Omron CX-Programmer project 新工程 (CX-Programmer 9.61)

# PLC XWD负压氦检: CJ2M CPU34
I/O table (CPU CJ2M-CPU34): rack 0 slot 11 CJ2M-EIP21

## Global symbols (name address type ; comment)
0.00 BOOL  ; #1扫码阻挡气缸缩回位
0.01 BOOL  ; #1扫码阻挡气缸伸出位
0.02 BOOL  ; #1隔离气缸缩回位
0.03 BOOL  ; 隔离气缸到位
0.04 BOOL  ; #2扫码阻挡气缸缩回位
0.05 BOOL  ; #2扫码阻挡气缸伸出位
0.06 BOOL  ; #2隔离气缸缩回位
0.08 BOOL  ; #1进料夹爪夹紧位
0.09 BOOL  ; #1进料夹爪松开位
0.10 BOOL  ; #2进料夹爪夹紧位
0.11 BOOL  ; #2进料夹爪松开位
0.12 BOOL  ; 进料夹爪变距气缸伸出位
0.13 BOOL  ; 进料夹爪变距气缸缩回位
0.14 BOOL  ; #1出料夹爪夹紧位
0.15 BOOL  ; #1出料夹爪松开位
10.00 BOOL  ; #1扫码阻挡气缸缩回
10.01 BOOL  ; #1扫码阻挡气缸伸出
10.02 BOOL  ; #1隔离气缸缩回
10.03 BOOL  ; #1隔离气缸伸出
10.04 BOOL  ; #2扫码阻挡气缸缩回
10.05 BOOL  ; #2扫码阻挡气缸伸出
10.06 BOOL  ; #2隔离气缸缩回
10.07 BOOL  ; #2隔离气缸伸出
10.08 BOOL  ; #1进料夹爪夹紧
10.09 BOOL  ; #1进料夹爪松开
10.10 BOOL  ; #2进料夹爪夹紧
10.11 BOOL  ; #2进料夹爪松开
10.12 BOOL  ; 进料夹爪变距气缸伸出
10.13 BOOL  ; 进料夹爪变距气缸缩回
10.14 BOOL  ; #1出料夹爪夹紧
10.15 BOOL  ; #1出料夹爪松开
11.00 BOOL  ; #2出料夹爪夹紧
11.01 BOOL  ; #2出料夹爪松开
11.02 BOOL  ; 出料夹爪变距气缸伸出
11.03 BOOL  ; 出料夹爪变距气缸缩回
11.04 BOOL  ; #1腔体平移一级气缸缩回
11.05 BOOL  ; #1腔体平移一级气缸伸出
11.06 BOOL  ; #1腔体平移二级气缸缩回
11.07 BOOL  ; #1腔体平移二级气缸伸出
11.08 BOOL  ; #1腔体顶伸气缸上升
11.09 BOOL  ; #1腔体顶伸气缸下降
11.10 BOOL  ; #1腔体氦检阀开
11.11 BOOL  ; 氦检仪真空阀开
11.12 BOOL  ; #1腔体抽真空阀开
11.13 BOOL  ; #1-1腔体阀开
11.14 BOOL  ; #1-2腔体阀开
11.15 BOOL  ; #1腔体破真空阀开
12.00 BOOL  ; #1腔体吹气阀开
12.01 BOOL  ; #2腔体平移一级气缸缩回
12.02 BOOL  ; #2腔体平移一级气缸伸出
12.03 BOOL  ; #2腔体平移二级气缸缩回
12.04 BOOL  ; #2腔体平移二级气缸伸出
12.05 BOOL  ; #2腔体顶伸气缸上升
12.06 BOOL  ; #2腔体顶伸气缸下降
12.07 BOOL  ; #2腔体氦检阀开
12.08 BOOL  ; 复检清洁阀开
12.09 BOOL  ; #2腔体抽真空阀开
12.10 BOOL  ; #2-1腔体阀开
12.11 BOOL  ; #2-2腔体阀开
12.12 BOOL  ; #2腔体破真空阀开
12.13 BOOL  ; #2腔体吹气阀开
12.14 BOOL  ; #3腔体平移一级气缸缩回
12.15 BOOL  ; #3腔体平移一级气缸伸出
13.00 BOOL  ; #3腔体平移二级气缸缩回
13.01 BOOL  ; #3腔体平移二级气缸伸出
13.02 BOOL  ; #3腔体顶伸气缸上升
13.03 BOOL  ; #3腔体顶伸气缸下降
13.04 BOOL  ; #3腔体氦检阀开
13.05 BOOL  ; 标漏阀开
13.06 BOOL  ; #3腔体抽真空阀开
13.07 BOOL  ; #3-1腔体阀开
13.08 BOOL  ; #3-2腔体阀开
13.09 BOOL  ; #3腔体破真空阀开
13.10 BOOL  ; #3腔体吹气阀开
13.11 BOOL  ; 进料伺服X轴使能
13.12 BOOL  ; 进料伺服X轴故障复位
13.13 BOOL  ; 进料伺服Z轴使能
13.14 BOOL  ; 进料伺服Z轴故障复位
13.15 BOOL  ; 进料伺服Z轴刹车
14.00 BOOL  ; 出料伺服X轴使能
14.01 BOOL  ; 出料伺服X轴故障复位
14.02 BOOL  ; 出料伺服Z轴使能
14.03 BOOL  ; 出料伺服Z轴故障复位
14.04 BOOL  ; 出料伺服Z轴刹车
14.05 BOOL  ; 腔体抽真空泵启动
14.07 BOOL  ; 氦检前置泵启动
14.08 BOOL  ; 氦检仪供电
14.09 BOOL  ; 启动按钮指示灯
14.10 BOOL  ; 停止按钮指示灯
14.11 BOOL  ; 复位按钮指示灯
14.12 BOOL  ; 蜂鸣器
14.13 BOOL  ; 三色灯（红）
14.14 BOOL  ; 三色灯（绿）
14.15 BOOL  ; 三色灯（黄）
1559.15 BOOL  ; SCU21_2Port#1 Protocol Macro Executing Flag
1569.15 BOOL  ; SCU21_2Port#2 Protocol Macro Executing Flag
15.00 BOOL  ; 进料拉带电机启动
15.01 BOOL  ; 扫码NG拉带电机启动
15.02 BOOL  ; 氦检NG拉带电机启动
15.03 BOOL  ; 进料对接输出
15.04 BOOL  ; 出料对接输出（TO下工站放料请求）
15.05 BOOL  ; 出料旋转气缸90度输出
15.06 BOOL  ; 出料旋转气缸0度输出
15.07 BOOL  ; 进料前段拉带输出
16.00 BOOL  ; #1-1电池抽真空阀开
16.01 BOOL  ; #1-2电池抽真空阀开
16.02 BOOL  ; #1-1电池注氦阀开
16.03 BOOL  ; #1-2电池注氦阀开
16.04 BOOL  ; #1-1电池破真空阀开
16.05 BOOL  ; #1-2电池破真空阀开
16.06 BOOL  ; #2-1电池抽真空阀开
16.07 BOOL  ; #2-2电池抽真空阀开
16.08 BOOL  ; #2-1电池注氦阀开
16.09 BOOL  ; #2-2电池注氦阀开
16.10 BOOL  ; #2-1电池破真空阀开
16.11 BOOL  ; #2-2电池破真空阀开
16.12 BOOL  ; #3-1电池抽真空阀开
16.13 BOOL  ; #3-2电池抽真空阀开
16.14 BOOL  ; #3-1电池注氦阀开
16.15 BOOL  ; #3-2电池注氦阀开
17.00 BOOL  ; #3-1电池破真空阀开
17.01 BOOL  ; #3-2电池破真空阀开
1.00 BOOL  ; #2出料夹爪夹紧位
1.01 BOOL  ; #2出料夹爪松开位
1.02 BOOL  ; 出料夹爪变距气缸伸出位
1.03 BOOL  ; 出料夹爪变距气缸缩回位
1.04 BOOL  ; #1腔体平移一级气缸缩回位
1.05 BOOL  ; #1腔体平移一级气缸伸出位
1.06 BOOL  ; #1腔体平移二级气缸缩回位
1.07 BOOL  ; #1腔体平移二级气缸伸出位
1.08 BOOL  ; #1腔体顶伸气缸上升位
1.09 BOOL  ; #1腔体顶伸气缸下降位
1.10 BOOL  ; #1腔体氦检阀开到位
1.11 BOOL  ; #1腔体氦检阀关到位
2001 CHANNEL  ; #1-1电池真空模拟量读数(AD081_1)
2002 CHANNEL  ; #1-2电池真空模拟量读数(AD081_2)
2003 CHANNEL  ; #2-1电池真空模拟量读数(AD081_3)
2004 CHANNEL  ; #2-2电池真空模拟量读数(AD081_4)
2005 CHANNEL  ; #3-1电池真空模拟量读数(AD081_5)
2006 CHANNEL  ; #3-2电池真空模拟量读数(AD081_6)
200.00 BOOL  ; PLC上电
200.01 BOOL  ; 紧急停止
200.01 BOOL  ; 急停按钮标志[0004.12]
200.02 BOOL  ; 自动启动
200.03 BOOL  ; 自动停止
200.04 BOOL  ; 报警清除
200.05 BOOL  ; 清料停止中
200.06 BOOL  ; 异常报警停止
200.08 BOOL  ; 设备待料状态（参考进料）
200.09 BOOL  ; 设备内有电池
200.10 BOOL  ; 机台有错误
200.11 BOOL  ; 报警中
200.12 BOOL  ; 三色灯-绿灯
200.13 BOOL  ; 三色灯-红灯
200.14 BOOL  ; 三色灯-黄灯
200.15 BOOL  ; 三色灯-蜂鸣器
2011 CHANNEL  ; #1腔体真空模拟量读数(AD041_1)
2012 CHANNEL  ; #2腔体真空模拟量读数(AD041_2)
2013 CHANNEL  ; #3腔体真空模拟量读数(AD041_3)
201.00 BOOL  ; 整机在初始位
205.00 BOOL  ; 整机停止中（Lamp）
205.01 BOOL  ; 清料停止中（Lamp）
205.02 BOOL  ; 整机复位（Lamp）
210.01 BOOL  ; PC系统通讯正常标志
210.02 BOOL  ; 整机机械手归零标志
210.03 BOOL  ; 安全门标志
210.04 BOOL  ; 氦检仪启动标志
221.00 BOOL  ; 整机复位（M）
221.01 BOOL  ; 进料拉带工站整机复位（M）
221.02 BOOL  ; 进料伺服工站整机复位（M）
221.03 BOOL  ; #1氦检工站整机复位（M）
221.04 BOOL  ; #2氦检工站整机复位（M）
221.05 BOOL  ; #3氦检工站整机复位（M）
221.06 BOOL  ; 出料伺服工站整机复位（M）
2960.02 BOOL  ; 进料伺服Z轴原点感应标志
2960.06 BOOL  ; 进料伺服X轴正极限
2960.07 BOOL  ; 进料伺服X轴负极限
2960.08 BOOL  ; 进料伺服Z轴正极限
2960.09 BOOL  ; 进料伺服Z轴负极限
2962.02 BOOL  ; 出料伺服Z轴原点感应标志
2962.06 BOOL  ; 出料伺服X轴正极限
2962.07 BOOL  ; 出料伺服X轴负极限
2962.08 BOOL  ; 出料伺服Z轴正极限
2962.09 BOOL  ; 出料伺服Z轴负极限
2.01 BOOL  ; #2腔体平移一级气缸缩回位
2.02 BOOL  ; #2腔体平移一级气缸伸出位
2.03 BOOL  ; #2腔体平移二级气缸缩回位
2.04 BOOL  ; #2腔体平移二级气缸伸出位
2.05 BOOL  ; #2腔体顶伸气缸上升位
2.06 BOOL  ; #2腔体顶伸气缸下降位
2.07 BOOL  ; #2腔体氦检阀开到位
2.08 BOOL  ; #2腔体氦检阀关到位
2.14 BOOL  ; #3腔体平移一级气缸缩回位
2.15 BOOL  ; #3腔体平移一级气缸伸出位
300.00 BOOL  ; #1扫码阻挡气缸缩回[Pls]
300.01 BOOL  ; #1扫码阻挡气缸伸出[Pls]
300.02 BOOL  ; #1隔离气缸缩回[Pls]
300.03 BOOL  ; #1隔离气缸伸出[Pls]
300.04 BOOL  ; #2扫码阻挡气缸缩回[Pls]
300.05 BOOL  ; #2扫码阻挡气缸伸出[Pls]
300.06 BOOL  ; #2隔离气缸缩回[Pls]
300.07 BOOL  ; #2隔离气缸伸出[Pls]
300.08 BOOL  ; #1进料夹爪夹紧[Pls]
300.09 BOOL  ; #1进料夹爪松开[Pls]
300.10 BOOL  ; #2进料夹爪夹紧[Pls]
300.11 BOOL  ; #2进料夹爪松开[Pls]
300.12 BOOL  ; 进料夹爪变距气缸伸出[Pls]
300.13 BOOL  ; 进料夹爪变距气缸缩回[Pls]
300.14 BOOL  ; #1出料夹爪夹紧[Pls]
300.15 BOOL  ; #1出料夹爪松开[Pls]
301.00 BOOL  ; #2出料夹爪夹紧[Pls]
301.01 BOOL  ; #2出料夹爪松开[Pls]
301.02 BOOL  ; 出料夹爪变距气缸伸出[Pls]
301.03 BOOL  ; 出料夹爪变距气缸缩回[Pls]
301.04 BOOL  ; #1腔体平移一级气缸缩回[Pls]
301.05 BOOL  ; #1腔体平移一级气缸伸出[Pls]
301.06 BOOL  ; #1腔体平移二级气缸缩回[Pls]
301.07 BOOL  ; #1腔体平移二级气缸伸出[Pls]
301.08 BOOL  ; #1腔体顶伸气缸上升[Pls]
301.09 BOOL  ; #1腔体顶伸气缸下降[Pls]
301.10 BOOL  ; #1腔体氦检阀开[Pls]
301.11 BOOL  ; 氦检仪真空阀开[Pls]
301.12 BOOL  ; #1腔体抽真空阀开[Pls]
301.13 BOOL  ; #1-1腔体阀开[Pls]
301.14 BOOL  ; #1-2腔体阀开[Pls]
301.15 BOOL  ; #1腔体破真空阀开[Pls]
302.00 BOOL  ; #1腔体吹气阀开[Pls]
302.01 BOOL  ; #2腔体平移一级气缸缩回[Pls]
302.02 BOOL  ; #2腔体平移一级气缸伸出[Pls]
302.03 BOOL  ; #2腔体平移二级气缸缩回[Pls]
302.04 BOOL  ; #2腔体平移二级气缸伸出[Pls]
302.05 BOOL  ; #2腔体顶伸气缸上升[Pls]
302.06 BOOL  ; #2腔体顶伸气缸下降[Pls]
302.07 BOOL  ; #2腔体氦检阀开[Pls]
302.08 BOOL  ; 复检清洁阀开[Pls]
302.09 BOOL  ; #2腔体抽真空阀开[Pls]
302.10 BOOL  ; #2-1腔体阀开[Pls]
302.11 BOOL  ; #2-2腔体阀开[Pls]
302.12 BOOL  ; #2腔体破真空阀开[Pls]
302.13 BOOL  ; #2腔体吹气阀开[Pls]
302.14 BOOL  ; #3腔体平移一级气缸缩回[Pls]
302.15 BOOL  ; #3腔体平移一级气缸伸出[Pls]
303.00 BOOL  ; #3腔体平移二级气缸缩回[Pls]
303.01 BOOL  ; #3腔体平移二级气缸伸出[Pls]
303.02 BOOL  ; #3腔体顶伸气缸上升[Pls]
303.03 BOOL  ; #3腔体顶伸气缸下降[Pls]
303.04 BOOL  ; #3腔体氦检阀开[Pls]
303.05 BOOL  ; 0[Pls]
303.06 BOOL  ; #3腔体抽真空阀开[Pls]
303.07 BOOL  ; #3-1腔体阀开[Pls]
303.08 BOOL  ; #3-2腔体阀开[Pls]
303.09 BOOL  ; #3腔体破真空阀开[Pls]
303.10 BOOL  ; #3腔体吹气阀开[Pls]
303.11 BOOL  ; 进料伺服X轴使能[Pls]
303.12 BOOL  ; 进料伺服X轴故障复位[Pls]
303.13 BOOL  ; 进料伺服Z轴使能[Pls]
303.14 BOOL  ; 进料伺服Z轴故障复位[Pls]
303.15 BOOL  ; 进料伺服Z轴刹车[Pls]
304.00 BOOL  ; 出料伺服X轴使能[Pls]
304.01 BOOL  ; 出料伺服X轴故障复位[Pls]
304.02 BOOL  ; 出料伺服Z轴使能[Pls]
304.03 BOOL  ; 出料伺服Z轴故障复位[Pls]
304.04 BOOL  ; 出料伺服Z轴刹车[Pls]
304.05 BOOL  ; 腔体抽真空泵启动[Pls]
304.06 BOOL  ; 0[Pls]
304.07 BOOL  ; 氦检前置泵启动[Pls]
304.08 BOOL  ; 氦检仪供电[Pls]
304.09 BOOL  ; 启动按钮指示灯[Pls]
304.10 BOOL  ; 停止按钮指示灯[Pls]
304.11 BOOL  ; 复位按钮指示灯[Pls]
304.12 BOOL  ; 蜂鸣器[Pls]
304.13 BOOL  ; 三色灯（红）[Pls]
304.14 BOOL  ; 三色灯（绿）[Pls]
304.15 BOOL  ; 三色灯（黄）[Pls]
305.00 BOOL  ; 进料拉带电机启动[Pls]
305.01 BOOL  ; 扫码NG拉带电机启动[Pls]
305.02 BOOL  ; 氦检NG拉带电机启动[Pls]
305.03 BOOL  ; 进料对接输出[Pls]
305.04 BOOL  ; 出料对接输出[Pls]
305.05 BOOL  ; 出料旋转气缸9O度位条件
305.06 BOOL  ; 出料旋转气缸O度位条件
305.07 BOOL  ; 0[Pls]
305.08 BOOL  ; 0[Pls]
305.09 BOOL  ; 0[Pls]
305.10 BOOL  ; 0[Pls]
305.11 BOOL  ; 0[Pls]
305.12 BOOL  ; 0[Pls]
305.13 BOOL  ; 0[Pls]
305.14 BOOL  ; 0[Pls]
305.15 BOOL  ; 0[Pls]
306.00 BOOL  ; #1-1电池抽真空阀开[Pls]
306.01 BOOL  ; #1-2电池抽真空阀开[Pls]
306.02 BOOL  ; #1-1电池注氦阀开[Pls]
306.03 BOOL  ; #1-2电池注氦阀开[Pls]
306.04 BOOL  ; #1-1电池破真空阀开[Pls]
306.05 BOOL  ; #1-2电池破真空阀开[Pls]
306.06 BOOL  ; #2-1电池抽真空阀开[Pls]
306.07 BOOL  ; #2-2电池抽真空阀开[Pls]
306.08 BOOL  ; #2-1电池注氦阀开[Pls]
306.09 BOOL  ; #2-2电池注氦阀开[Pls]
306.10 BOOL  ; #2-1电池破真空阀开[Pls]
306.11 BOOL  ; #2-2电池破真空阀开[Pls]
306.12 BOOL  ; #3-1电池抽真空阀开[Pls]
306.13 BOOL  ; #3-2电池抽真空阀开[Pls]
306.14 BOOL  ; #3-1电池注氦阀开[Pls]
306.15 BOOL  ; #3-2电池注氦阀开[Pls]
307.00 BOOL  ; #3-1电池破真空阀开[Pls]
307.01 BOOL  ; #3-2电池破真空阀开[Pls]
307.02 BOOL  ; 0[Pls]
307.03 BOOL  ; 0[Pls]
307.04 BOOL  ; 0[Pls]
307.05 BOOL  ; 0[Pls]
307.06 BOOL  ; 0[Pls]
307.07 BOOL  ; 0[Pls]
307.08 BOOL  ; 0[Pls]
307.09 BOOL  ; 0[Pls]
307.10 BOOL  ; 0[Pls]
307.11 BOOL  ; 0[Pls]
307.12 BOOL  ; 0[Pls]
307.13 BOOL  ; 0[Pls]
307.14 BOOL  ; 0[Pls]
307.15 BOOL  ; 0[Pls]
311.10 BOOL  ; #1腔体氦检阀关[Pls]
311.11 BOOL  ; 氦检仪真空阀关[Pls]
311.12 BOOL  ; #1腔体抽真空阀关[Pls]
311.13 BOOL  ; #1-1腔体阀关[Pls]
311.14 BOOL  ; #1-2腔体阀关[Pls]
311.15 BOOL  ; #1腔体破真空阀关[Pls]
312.00 BOOL  ; #1腔体吹气阀关[Pls]
312.01 BOOL  ; [Pls]
312.02 BOOL  ; [Pls]
312.03 BOOL  ; [Pls]
312.04 BOOL  ; [Pls]
312.05 BOOL  ; [Pls]
312.06 BOOL  ; [Pls]
312.07 BOOL  ; #2腔体氦检阀关[Pls]
312.08 BOOL  ; 复检清洁阀关[Pls]
312.09 BOOL  ; #2腔体抽真空阀关[Pls]
312.10 BOOL  ; #2-1腔体阀关[Pls]
312.11 BOOL  ; #2-2腔体阀关[Pls]
312.12 BOOL  ; #2腔体破真空阀关[Pls]
312.13 BOOL  ; #2腔体吹气阀关[Pls]
312.14 BOOL  ; 0[Pls]
312.15 BOOL  ; [Pls]
313.00 BOOL  ; [Pls]
313.01 BOOL  ; [Pls]
313.02 BOOL  ; [Pls]
313.03 BOOL  ; [Pls]
313.04 BOOL  ; #3腔体氦检阀关[Pls]
313.05 BOOL  ; 0[Pls]
313.06 BOOL  ; #3腔体抽真空阀关[Pls]
313.07 BOOL  ; #3-1腔体阀关[Pls]
313.08 BOOL  ; #3-2腔体阀关[Pls]
313.09 BOOL  ; #3腔体破真空阀关[Pls]
313.10 BOOL  ; #3腔体吹气阀关[Pls]
313.11 BOOL  ; [Pls]
313.12 BOOL  ; [Pls]
313.13 BOOL  ; [Pls]
313.14 BOOL  ; [Pls]
313.15 BOOL  ; [Pls]
314.00 BOOL  ; [Pls]
314.01 BOOL  ; [Pls]
314.02 BOOL  ; [Pls]
314.03 BOOL  ; [Pls]
314.04 BOOL  ; [Pls]
314.05 BOOL  ; 腔体抽真空泵停止[Pls]
314.06 BOOL  ; 0[Pls]
314.07 BOOL  ; 氦检前置泵停止[Pls]
314.08 BOOL  ; 氦检仪停电[Pls]
314.09 BOOL  ; [Pls]
314.10 BOOL  ; [Pls]
314.11 BOOL  ; [Pls]
314.12 BOOL  ; [Pls]
314.13 BOOL  ; [Pls]
314.14 BOOL  ; [Pls]
314.15 BOOL  ; [Pls]
315.00 BOOL  ; 进料拉带电机停止[Pls]
315.01 BOOL  ; 扫码NG拉带电机停止[Pls]
315.02 BOOL  ; 氦检NG拉带电机停止[Pls]
315.03 BOOL  ; 0[Pls]
315.04 BOOL  ; [Pls]
315.05 BOOL  ; [Pls]
315.06 BOOL  ; [Pls]
315.07 BOOL  ; [Pls]
315.08 BOOL  ; [Pls]
315.09 BOOL  ; [Pls]
315.10 BOOL  ; [Pls]
315.11 BOOL  ; [Pls]
315.12 BOOL  ; [Pls]
315.13 BOOL  ; [Pls]
315.14 BOOL  ; [Pls]
315.15 BOOL  ; [Pls]
316.00 BOOL  ; #1-1电池抽真空阀关[Pls]
316.01 BOOL  ; #1-2电池抽真空阀关[Pls]
316.02 BOOL  ; #1-1电池注氦阀关[Pls]
316.03 BOOL  ; #1-2电池注氦阀关[Pls]
316.04 BOOL  ; #1-1电池破真空阀关[Pls]
316.05 BOOL  ; #1-2电池破真空阀关[Pls]
316.06 BOOL  ; #2-1电池抽真空阀关[Pls]
316.07 BOOL  ; #2-2电池抽真空阀关[Pls]
316.08 BOOL  ; #2-1电池注氦阀关[Pls]
316.09 BOOL  ; #2-2电池注氦阀关[Pls]
316.10 BOOL  ; #2-1电池破真空阀关[Pls]
316.11 BOOL  ; #2-2电池破真空阀关[Pls]
316.12 BOOL  ; #3-1电池抽真空阀关[Pls]
316.13 BOOL  ; #3-2电池抽真空阀关[Pls]
316.14 BOOL  ; #3-1电池注氦阀关[Pls]
316.15 BOOL  ; #3-2电池注氦阀关[Pls]
317.00 BOOL  ; #3-1电池破真空阀关[Pls]
317.01 BOOL  ; #3-2电池破真空阀关[Pls]
3.00 BOOL  ; #3腔体平移二级气缸缩回位
3.01 BOOL  ; #3腔体平移二级气缸伸出位
3.02 BOOL  ; #3腔体顶伸气缸上升位
3.03 BOOL  ; #3腔体顶伸气缸下降位
3.04 BOOL  ; #3腔体氦检阀开到位
3.05 BOOL  ; #3腔体氦检阀关到位
3.06 BOOL  ; 氦检仪准备好了信号
3.07 BOOL  ; 氦检仪故障信号
3.11 BOOL  ; 进料伺服X轴准备好了信号
3.12 BOOL  ; 进料伺服X轴故障信号
3.13 BOOL  ; 进料伺服Z轴准备好了信号
3.14 BOOL  ; 进料伺服Z轴故障信号
400.00 BOOL  ; #1扫码阻挡气缸缩回[M]
400.01 BOOL  ; #1扫码阻挡气缸伸出[M]
400.02 BOOL  ; #1隔离气缸缩回[M]
400.03 BOOL  ; #1隔离气缸伸出[M]
400.04 BOOL  ; #2扫码阻挡气缸缩回[M]
400.05 BOOL  ; #2扫码阻挡气缸伸出[M]
400.06 BOOL  ; #2隔离气缸缩回[M]
400.07 BOOL  ; #2隔离气缸伸出[M]
400.08 BOOL  ; #1进料夹爪夹紧[M]
400.09 BOOL  ; #1进料夹爪松开[M]
400.10 BOOL  ; #2进料夹爪夹紧[M]
400.11 BOOL  ; #2进料夹爪松开[M]
400.12 BOOL  ; 进料夹爪变距气缸伸出[M]
400.13 BOOL  ; 进料夹爪变距气缸缩回[M]
400.14 BOOL  ; #1出料夹爪夹紧[M]
400.15 BOOL  ; #1出料夹爪松开[M]
401.00 BOOL  ; #2出料夹爪夹紧[M]
401.01 BOOL  ; #2出料夹爪松开[M]
401.02 BOOL  ; 出料夹爪变距气缸伸出[M]
401.03 BOOL  ; 出料夹爪变距气缸缩回[M]
401.04 BOOL  ; #1腔体平移一级气缸缩回[M]
401.05 BOOL  ; #1腔体平移一级气缸伸出[M]
401.06 BOOL  ; #1腔体平移二级气缸缩回[M]
401.07 BOOL  ; #1腔体平移二级气缸伸出[M]
401.08 BOOL  ; #1腔体顶伸气缸上升[M]
401.09 BOOL  ; #1腔体顶伸气缸下降[M]
401.10 BOOL  ; #1腔体氦检阀开[M]
401.11 BOOL  ; 氦检仪真空阀开[M]
401.12 BOOL  ; #1腔体抽真空阀开[M]
401.13 BOOL  ; #1-1腔体阀开[M]
401.14 BOOL  ; #1-2腔体阀开[M]
401.15 BOOL  ; #1腔体破真空阀开[M]
402.00 BOOL  ; #1腔体吹气阀开[M]
402.01 BOOL  ; #2腔体平移一级气缸缩回[M]
402.02 BOOL  ; #2腔体平移一级气缸伸出[M]
402.03 BOOL  ; #2腔体平移二级气缸缩回[M]
402.04 BOOL  ; #2腔体平移二级气缸伸出[M]
402.05 BOOL  ; #2腔体顶伸气缸上升[M]
402.06 BOOL  ; #2腔体顶伸气缸下降[M]
402.07 BOOL  ; #2腔体氦检阀开[M]
402.08 BOOL  ; 复检清洁阀开[M]
402.09 BOOL  ; #2腔体抽真空阀开[M]
402.10 BOOL  ; #2-1腔体阀开[M]
402.11 BOOL  ; #2-2腔体阀开[M]
402.12 BOOL  ; #2腔体破真空阀开[M]
402.13 BOOL  ; #2腔体吹气阀开[M]
402.14 BOOL  ; #3腔体平移一级气缸缩回[M]
402.15 BOOL  ; #3腔体平移一级气缸伸出[M]
403.00 BOOL  ; #3腔体平移二级气缸缩回[M]
403.01 BOOL  ; #3腔体平移二级气缸伸出[M]
403.02 BOOL  ; #3腔体顶伸气缸上升[M]
403.03 BOOL  ; #3腔体顶伸气缸下降[M]
403.04 BOOL  ; #3腔体氦检阀开[M]
403.05 BOOL  ; 0[M]
403.06 BOOL  ; #3腔体抽真空阀开[M]
403.07 BOOL  ; #3-1腔体阀开[M]
403.08 BOOL  ; #3-2腔体阀开[M]
403.09 BOOL  ; #3腔体破真空阀开[M]
403.10 BOOL  ; #3腔体吹气阀开[M]
403.11 BOOL  ; 进料伺服X轴使能[M]
403.12 BOOL  ; 进料伺服X轴故障复位[M]
403.13 BOOL  ; 进料伺服Z轴使能[M]
403.14 BOOL  ; 进料伺服Z轴故障复位[M]
403.15 BOOL  ; 进料伺服Z轴刹车[M]
404.00 BOOL  ; 出料伺服X轴使能[M]
404.01 BOOL  ; 出料伺服X轴故障复位[M]
404.02 BOOL  ; 出料伺服Z轴使能[M]
404.03 BOOL  ; 出料伺服Z轴故障复位[M]
404.04 BOOL  ; 出料伺服Z轴刹车[M]
404.05 BOOL  ; 腔体抽真空泵启动[M]
404.06 BOOL  ; 0[M]
404.07 BOOL  ; 氦检前置泵启动[M]
404.08 BOOL  ; 氦检仪供电[M]
404.09 BOOL  ; 启动按钮指示灯[M]
404.10 BOOL  ; 停止按钮指示灯[M]
404.11 BOOL  ; 复位按钮指示灯[M]
404.12 BOOL  ; 蜂鸣器[M]
404.13 BOOL  ; 三色灯（红）[M]
404.14 BOOL  ; 三色灯（绿）[M]
404.15 BOOL  ; 三色灯（黄）[M]
405.00 BOOL  ; 进料拉带电机启动[M]
405.01 BOOL  ; 扫码NG拉带电机启动[M]
405.02 BOOL  ; 氦检NG拉带电机启动[M]
405.03 BOOL  ; 进料对接输出[M]
405.04 BOOL  ; 出料对接输出[M]
405.05 BOOL  ; 出料旋转气缸90度输出[M]
405.06 BOOL  ; 出料旋转气缸0度输出[M]
405.07 BOOL  ; 0[M]
405.08 BOOL  ; 0[M]
405.09 BOOL  ; 0[M]
405.10 BOOL  ; 0[M]
405.11 BOOL  ; 0[M]
405.12 BOOL  ; 0[M]
405.13 BOOL  ; 0[M]
405.14 BOOL  ; 0[M]
405.15 BOOL  ; 0[M]
406.00 BOOL  ; #1-1电池抽真空阀开[M]
406.01 BOOL  ; #1-2电池抽真空阀开[M]
406.02 BOOL  ; #1-1电池注氦阀开[M]
406.03 BOOL  ; #1-2电池注氦阀开[M]
406.04 BOOL  ; #1-1电池破真空阀开[M]
406.05 BOOL  ; #1-2电池破真空阀开[M]
406.06 BOOL  ; #2-1电池抽真空阀开[M]
406.07 BOOL  ; #2-2电池抽真空阀开[M]
406.08 BOOL  ; #2-1电池注氦阀开[M]
406.09 BOOL  ; #2-2电池注氦阀开[M]
406.10 BOOL  ; #2-1电池破真空阀开[M]
406.11 BOOL  ; #2-2电池破真空阀开[M]
406.12 BOOL  ; #3-1电池抽真空阀开[M]
406.13 BOOL  ; #3-2电池抽真空阀开[M]
406.14 BOOL  ; #3-1电池注氦阀开[M]
406.15 BOOL  ; #3-2电池注氦阀开[M]
407.00 BOOL  ; #3-1电池破真空阀开[M]
407.01 BOOL  ; #3-2电池破真空阀开[M]
407.02 BOOL  ; 0[M]
407.03 BOOL  ; 0[M]
407.04 BOOL  ; 0[M]
407.05 BOOL  ; 0[M]
407.06 BOOL  ; 0[M]
407.07 BOOL  ; 0[M]
407.08 BOOL  ; 0[M]
407.09 BOOL  ; 0[M]
407.10 BOOL  ; 0[M]
407.11 BOOL  ; 0[M]
407.12 BOOL  ; 0[M]
407.13 BOOL  ; 0[M]
407.14 BOOL  ; 0[M]
407.15 BOOL  ; 0[M]
411.10 BOOL  ; #1腔体氦检阀关[M]
411.11 BOOL  ; 氦检仪真空阀关[M]
411.12 BOOL  ; #1腔体抽真空阀关[M]
411.13 BOOL  ; #1-1腔体阀关[M]
411.14 BOOL  ; #1-2腔体阀关[M]
411.15 BOOL  ; #1腔体破真空阀关[M]
412.00 BOOL  ; #1腔体吹气阀关[M]
412.01 BOOL  ; [M]
412.02 BOOL  ; [M]
412.03 BOOL  ; [M]
412.04 BOOL  ; [M]
412.05 BOOL  ; [M]
412.06 BOOL  ; [M]
412.07 BOOL  ; #2腔体氦检阀关[M]
412.08 BOOL  ; 复检清洁阀关[M]
412.09 BOOL  ; #2腔体抽真空阀关[M]
412.10 BOOL  ; #2-1腔体阀关[M]
412.11 BOOL  ; #2-2腔体阀关[M]
412.12 BOOL  ; #2腔体破真空阀关[M]
412.13 BOOL  ; #2腔体吹气阀关[M]
412.14 BOOL  ; 0[M]
412.15 BOOL  ; [M]
413.00 BOOL  ; [M]
413.01 BOOL  ; [M]
413.02 BOOL  ; [M]
413.03 BOOL  ; [M]
413.04 BOOL  ; #3腔体氦检阀关[M]
413.05 BOOL  ; 0[M]
413.06 BOOL  ; #3腔体抽真空阀关[M]
413.07 BOOL  ; #3-1腔体阀关[M]
413.08 BOOL  ; #3-2腔体阀关[M]
413.09 BOOL  ; #3腔体破真空阀关[M]
413.10 BOOL  ; #3腔体吹气阀关[M]
413.11 BOOL  ; [M]
413.12 BOOL  ; [M]
413.13 BOOL  ; [M]
413.14 BOOL  ; [M]
413.15 BOOL  ; [M]
414.00 BOOL  ; [M]
414.01 BOOL  ; [M]
414.02 BOOL  ; [M]
414.03 BOOL  ; [M]
414.04 BOOL  ; [M]
414.05 BOOL  ; 腔体抽真空泵停止[M]
414.06 BOOL  ; 0[M]
414.07 BOOL  ; 氦检前置泵停止[M]
414.08 BOOL  ; 氦检仪停电[M]
414.09 BOOL  ; [M]
414.10 BOOL  ; [M]
414.11 BOOL  ; [M]
414.12 BOOL  ; [M]
414.13 BOOL  ; [M]
414.14 BOOL  ; [M]
414.15 BOOL  ; [M]
415.00 BOOL  ; 进料拉带电机停止[M]
415.01 BOOL  ; 扫码NG拉带电机停止[M]
415.02 BOOL  ; 氦检NG拉带电机停止[M]
415.03 BOOL  ; 0[M]
415.04 BOOL  ; [M]
415.05 BOOL  ; [M]
415.06 BOOL  ; [M]
415.07 BOOL  ; [M]
415.08 BOOL  ; [M]
415.09 BOOL  ; [M]
415.10 BOOL  ; [M]
415.11 BOOL  ; [M]
415.12 BOOL  ; [M]
415.13 BOOL  ; [M]
415.14 BOOL  ; [M]
415.15 BOOL  ; [M]
416.00 BOOL  ; #1-1电池抽真空阀关[M]
416.01 BOOL  ; #1-2电池抽真空阀关[M]
416.02 BOOL  ; #1-1电池注氦阀关[M]
416.03 BOOL  ; #1-2电池注氦阀关[M]
416.04 BOOL  ; #1-1电池破真空阀关[M]
416.05 BOOL  ; #1-2电池破真空阀关[M]
416.06 BOOL  ; #2-1电池抽真空阀关[M]
416.07 BOOL  ; #2-2电池抽真空阀关[M]
416.08 BOOL  ; #2-1电池注氦阀关[M]
416.09 BOOL  ; #2-2电池注氦阀关[M]
416.10 BOOL  ; #2-1电池破真空阀关[M]
416.11 BOOL  ; #2-2电池破真空阀关[M]
416.12 BOOL  ; #3-1电池抽真空阀关[M]
416.13 BOOL  ; #3-2电池抽真空阀关[M]
416.14 BOOL  ; #3-1电池注氦阀关[M]
416.15 BOOL  ; #3-2电池注氦阀关[M]
417.00 BOOL  ; #3-1电池破真空阀关[M]
417.01 BOOL  ; #3-2电池破真空阀关[M]
449.00 BOOL  ; 进料#1扫码测试[M]
449.01 BOOL  ; 进料#2扫码测试[M]
450.00 BOOL  ; 进料伺服X轴JOG+[M]
450.01 BOOL  ; 进料伺服X轴JOG-[M]
450.02 BOOL  ; 进料伺服X轴回原点[M]
450.03 BOOL  ; 进料伺服X轴取料位[M]
450.04 BOOL  ; 进料伺服X轴#1腔放料位[M]
450.05 BOOL  ; 进料伺服X轴#2腔放料位[M]
450.06 BOOL  ; 进料伺服X轴#3腔放料位[M]
450.07 BOOL  ; 进料伺服X轴#1夹爪扫码NG放料位[M]
450.08 BOOL  ; 进料伺服X轴#2夹爪扫码NG放料位[M]
450.09 BOOL  ; 进料伺服X轴#1夹爪配对取放料位[M]
450.10 BOOL  ; 进料伺服X轴#2夹爪配对取放料位[M]
450.11 BOOL  ; 进料伺服X轴#1腔有料检测位[M]
450.12 BOOL  ; 进料伺服X轴#2腔有料检测位[M]
450.13 BOOL  ; 进料伺服X轴#3腔有料检测位[M]
450.14 BOOL  ; 0[M]
450.15 BOOL  ; 0[M]
451.00 BOOL  ; 进料伺服Z轴JOG+[M]
451.01 BOOL  ; 进料伺服Z轴JOG-[M]
451.02 BOOL  ; 进料伺服Z轴回原点[M]
451.03 BOOL  ; 进料伺服Z轴待机位[M]
451.04 BOOL  ; 进料伺服Z轴取料位[M]
451.05 BOOL  ; 进料伺服Z轴#1腔放料位[M]
451.06 BOOL  ; 进料伺服Z轴#2腔放料位[M]
451.07 BOOL  ; 进料伺服Z轴#3腔放料位[M]
451.08 BOOL  ; 进料伺服Z轴#1夹爪扫码NG放料位[M]
451.09 BOOL  ; 进料伺服Z轴#2夹爪扫码NG放料位[M]
451.10 BOOL  ; 进料伺服Z轴#1夹爪配对取放料位[M]
451.11 BOOL  ; 进料伺服Z轴#2夹爪配对取放料位[M]
451.12 BOOL  ; 0[M]
451.13 BOOL  ; 0[M]
451.14 BOOL  ; 0[M]
451.15 BOOL  ; 0[M]
452.00 BOOL  ; 出料伺服X轴JOG+[M]
452.01 BOOL  ; 出料伺服X轴JOG-[M]
452.02 BOOL  ; 出料伺服X轴回原点[M]
452.03 BOOL  ; 出料伺服X轴放料位[M]
452.04 BOOL  ; 出料伺服X轴#1腔取料位[M]
452.05 BOOL  ; 出料伺服X轴#2腔取料位[M]
452.06 BOOL  ; 出料伺服X轴#3腔取料位[M]
452.07 BOOL  ; 出料伺服X轴#1夹爪氦检NG放料位[M]
452.08 BOOL  ; 出料伺服X轴#2夹爪氦检NG放料位[M]
452.09 BOOL  ; 出料伺服X轴#1夹爪配对取放料位[M]
452.10 BOOL  ; 出料伺服X轴#2夹爪配对取放料位[M]
452.11 BOOL  ; 0[M]
452.12 BOOL  ; 0[M]
452.13 BOOL  ; 0[M]
452.14 BOOL  ; 0[M]
452.15 BOOL  ; 0[M]
453.00 BOOL  ; 出料伺服Z轴JOG+[M]
453.01 BOOL  ; 出料伺服Z轴JOG-[M]
453.02 BOOL  ; 出料伺服Z轴回原点[M]
453.03 BOOL  ; 出料伺服Z轴待机位[M]
453.04 BOOL  ; 出料伺服Z轴放料位[M]
453.05 BOOL  ; 出料伺服Z轴#1腔取料位[M]
453.06 BOOL  ; 出料伺服Z轴#2腔取料位[M]
453.07 BOOL  ; 出料伺服Z轴#3腔取料位[M]
453.08 BOOL  ; 出料伺服Z轴#1夹爪氦检NG放料位[M]
453.09 BOOL  ; 出料伺服Z轴#2夹爪氦检NG放料位[M]
453.10 BOOL  ; 出料伺服Z轴#1夹爪配对取放料位[M]
453.11 BOOL  ; 出料伺服Z轴#2夹爪配对取放料位[M]
480.00 BOOL  ; 进料伺服X轴定位目标位置设定OK
480.01 BOOL  ; 进料伺服X轴定位条件
480.10 BOOL  ; 进料伺服Z轴定位目标位置设定OK
480.11 BOOL  ; 进料伺服Z轴定位条件
481.00 BOOL  ; 进料伺服X轴手动定位触发（M）
481.01 BOOL  ; 进料伺服X轴单步/自动循环定位触发（A）
481.10 BOOL  ; 进料伺服Z轴手动定位触发（M）
481.11 BOOL  ; 进料伺服Z轴单步/自动循环定位触发（A）
4.00 BOOL  ; 出料伺服X轴准备好了信号
4.01 BOOL  ; 出料伺服X轴故障信号
4.02 BOOL  ; 出料伺服Z轴准备好了信号
4.03 BOOL  ; 出料伺服Z轴故障信号
4.05 BOOL  ; 腔体抽真空泵运行信号
4.06 BOOL  ; 腔体抽真空泵过载信号
4.07 BOOL  ; 氦检前置泵运行信号
4.08 BOOL  ; 氦检前置泵过载信号
4.09 BOOL  ; 启动按钮
4.10 BOOL  ; 停止按钮
4.11 BOOL  ; 复位按钮
4.12 BOOL  ; 急停按钮
4.13 BOOL  ; 手自动选择
4.14 BOOL  ; #1进料夹爪防下坠感应
4.15 BOOL  ; #2进料夹爪防下坠感应
500.00 BOOL  ; #1扫码阻挡气缸缩回条件
500.01 BOOL  ; #1扫码阻挡气缸伸出条件
500.02 BOOL  ; #1隔离气缸缩回条件
500.03 BOOL  ; #1隔离气缸伸出条件
500.04 BOOL  ; #2扫码阻挡气缸缩回条件
500.05 BOOL  ; #2扫码阻挡气缸伸出条件
500.06 BOOL  ; #2隔离气缸缩回条件
500.07 BOOL  ; #2隔离气缸伸出条件
500.08 BOOL  ; #1进料夹爪夹紧条件
500.09 BOOL  ; #1进料夹爪松开条件
500.10 BOOL  ; #2进料夹爪夹紧条件
500.11 BOOL  ; #2进料夹爪松开条件
500.12 BOOL  ; 进料夹爪变距气缸伸出条件
500.13 BOOL  ; 进料夹爪变距气缸缩回条件
500.14 BOOL  ; #1出料夹爪夹紧条件
500.15 BOOL  ; #1出料夹爪松开条件
501.00 BOOL  ; #2出料夹爪夹紧条件
501.01 BOOL  ; #2出料夹爪松开条件
501.02 BOOL  ; 出料夹爪变距气缸伸出条件
501.03 BOOL  ; 出料夹爪变距气缸缩回条件
501.04 BOOL  ; #1腔体平移一级气缸缩回条件
501.05 BOOL  ; #1腔体平移一级气缸伸出条件
501.06 BOOL  ; #1腔体平移二级气缸缩回条件
501.07 BOOL  ; #1腔体平移二级气缸伸出条件
501.08 BOOL  ; #1腔体顶伸气缸上升条件
501.09 BOOL  ; #1腔体顶伸气缸下降条件
501.10 BOOL  ; #1腔体氦检阀开条件
501.11 BOOL  ; 氦检仪真空阀开条件
501.12 BOOL  ; #1腔体抽真空阀开条件
501.13 BOOL  ; #1-1腔体阀开条件
501.14 BOOL  ; #1-2腔体阀开条件
501.15 BOOL  ; #1腔体破真空阀开条件
502.00 BOOL  ; #1腔体吹气阀开条件
502.01 BOOL  ; #2腔体平移一级气缸缩回条件
502.02 BOOL  ; #2腔体平移一级气缸伸出条件
502.03 BOOL  ; #2腔体平移二级气缸缩回条件
502.04 BOOL  ; #2腔体平移二级气缸伸出条件
502.05 BOOL  ; #2腔体顶伸气缸上升条件
502.06 BOOL  ; #2腔体顶伸气缸下降条件
502.07 BOOL  ; #2腔体氦检阀开条件
502.08 BOOL  ; 复检清洁阀开条件
502.09 BOOL  ; #2腔体抽真空阀开条件
502.10 BOOL  ; #2-1腔体阀开条件
502.11 BOOL  ; #2-2腔体阀开条件
502.12 BOOL  ; #2腔体破真空阀开条件
502.13 BOOL  ; #2腔体吹气阀开条件
502.14 BOOL  ; #3腔体平移一级气缸缩回条件
502.15 BOOL  ; #3腔体平移一级气缸伸出条件
503.00 BOOL  ; #3腔体平移二级气缸缩回条件
503.01 BOOL  ; #3腔体平移二级气缸伸出条件
503.02 BOOL  ; #3腔体顶伸气缸上升条件
503.03 BOOL  ; #3腔体顶伸气缸下降条件
503.04 BOOL  ; #3腔体氦检阀开条件
503.05 BOOL  ; 0条件
503.06 BOOL  ; #3腔体抽真空阀开条件
503.07 BOOL  ; #3-1腔体阀开条件
503.08 BOOL  ; #3-2腔体阀开条件
503.09 BOOL  ; #3腔体破真空阀开条件
503.10 BOOL  ; #3腔体吹气阀开条件
503.11 BOOL  ; 进料伺服X轴使能条件
503.12 BOOL  ; 进料伺服X轴故障复位条件
503.13 BOOL  ; 进料伺服Z轴使能条件
503.14 BOOL  ; 进料伺服Z轴故障复位条件
503.15 BOOL  ; 进料伺服Z轴刹车条件
504.00 BOOL  ; 出料伺服X轴使能条件
504.01 BOOL  ; 出料伺服X轴故障复位条件
504.02 BOOL  ; 出料伺服Z轴使能条件
504.03 BOOL  ; 出料伺服Z轴故障复位条件
504.04 BOOL  ; 出料伺服Z轴刹车条件
504.05 BOOL  ; 腔体抽真空泵启动条件
504.06 BOOL  ; 0条件
504.07 BOOL  ; 氦检前置泵启动条件
504.08 BOOL  ; 氦检仪供电条件
504.09 BOOL  ; 启动按钮指示灯条件
504.10 BOOL  ; 停止按钮指示灯条件
504.11 BOOL  ; 复位按钮指示灯条件
504.12 BOOL  ; 蜂鸣器条件
504.13 BOOL  ; 三色灯（红）条件
504.14 BOOL  ; 三色灯（绿）条件
504.15 BOOL  ; 三色灯（黄）条件
505.00 BOOL  ; 进料拉带电机启动条件
505.01 BOOL  ; 扫码NG拉带电机启动条件
505.02 BOOL  ; 氦检NG拉带电机启动条件
505.03 BOOL  ; 进料对接输出条件
505.04 BOOL  ; 出料对接输出条件
505.05 BOOL  ; 出料旋转气缸9O度位条件
505.06 BOOL  ; 出料旋转气缸O度位条件
505.07 BOOL  ; 0条件
505.08 BOOL  ; 0条件
505.09 BOOL  ; 0条件
505.10 BOOL  ; 0条件
505.11 BOOL  ; 0条件
505.12 BOOL  ; 0条件
505.13 BOOL  ; 0条件
505.14 BOOL  ; 0条件
505.15 BOOL  ; 0条件
506.00 BOOL  ; #1-1电池抽真空阀开条件
506.01 BOOL  ; #1-2电池抽真空阀开条件
506.02 BOOL  ; #1-1电池注氦阀开条件
506.03 BOOL  ; #1-2电池注氦阀开条件
506.04 BOOL  ; #1-1电池破真空阀开条件
506.05 BOOL  ; #1-2电池破真空阀开条件
506.06 BOOL  ; #2-1电池抽真空阀开条件
506.07 BOOL  ; #2-2电池抽真空阀开条件
506.08 BOOL  ; #2-1电池注氦阀开条件
506.09 BOOL  ; #2-2电池注氦阀开条件
506.10 BOOL  ; #2-1电池破真空阀开条件
506.11 BOOL  ; #2-2电池破真空阀开条件
506.12 BOOL  ; #3-1电池抽真空阀开条件
506.13 BOOL  ; #3-2电池抽真空阀开条件
506.14 BOOL  ; #3-1电池注氦阀开条件
506.15 BOOL  ; #3-2电池注氦阀开条件
507.00 BOOL  ; #3-1电池破真空阀开条件
507.01 BOOL  ; #3-2电池破真空阀开条件
507.02 BOOL  ; 0条件
507.03 BOOL  ; 0条件
507.04 BOOL  ; 0条件
507.05 BOOL  ; 0条件
507.06 BOOL  ; 0条件
507.07 BOOL  ; 0条件
507.08 BOOL  ; 0条件
507.09 BOOL  ; 0条件
507.10 BOOL  ; 0条件
507.11 BOOL  ; 0条件
507.12 BOOL  ; 0条件
507.13 BOOL  ; 0条件
507.14 BOOL  ; 0条件
507.15 BOOL  ; 0条件
511.10 BOOL  ; #1腔体氦检阀关条件
511.11 BOOL  ; 氦检仪真空阀关条件
511.12 BOOL  ; #1腔体抽真空阀关条件
511.13 BOOL  ; #1-1腔体阀关条件
511.14 BOOL  ; #1-2腔体阀关条件
511.15 BOOL  ; #1腔体破真空阀关条件
512.00 BOOL  ; #1腔体吹气阀关条件
512.01 BOOL  ; 条件
512.02 BOOL  ; 条件
512.03 BOOL  ; 条件
512.04 BOOL  ; 条件
512.05 BOOL  ; 条件
512.06 BOOL  ; 条件
512.07 BOOL  ; #2腔体氦检阀关条件
512.08 BOOL  ; 复检清洁阀关条件
512.09 BOOL  ; #2腔体抽真空阀关条件
512.10 BOOL  ; #2-1腔体阀关条件
512.11 BOOL  ; #2-2腔体阀关条件
512.12 BOOL  ; #2腔体破真空阀关条件
512.13 BOOL  ; #2腔体吹气阀关条件
512.14 BOOL  ; 0条件
512.15 BOOL  ; 条件
513.00 BOOL  ; 条件
513.01 BOOL  ; 条件
513.02 BOOL  ; 条件
513.03 BOOL  ; 条件
513.04 BOOL  ; #3腔体氦检阀关条件
513.05 BOOL  ; 0条件
513.06 BOOL  ; #3腔体抽真空阀关条件
513.07 BOOL  ; #3-1腔体阀关条件
513.08 BOOL  ; #3-2腔体阀关条件
513.09 BOOL  ; #3腔体破真空阀关条件
513.10 BOOL  ; #3腔体吹气阀关条件
513.11 BOOL  ; 条件
513.12 BOOL  ; 条件
513.13 BOOL  ; 条件
513.14 BOOL  ; 条件
513.15 BOOL  ; 条件
514.00 BOOL  ; 条件
514.01 BOOL  ; 条件
514.02 BOOL  ; 条件
514.03 BOOL  ; 条件
514.04 BOOL  ; 条件
514.05 BOOL  ; 腔体抽真空泵停止条件
514.06 BOOL  ; 0条件
514.07 BOOL  ; 氦检前置泵停止条件
514.08 BOOL  ; 氦检仪停电条件
514.09 BOOL  ; 条件
514.10 BOOL  ; 条件
514.11 BOOL  ; 条件
514.12 BOOL  ; 条件
514.13 BOOL  ; 条件
514.14 BOOL  ; 条件
514.15 BOOL  ; 条件
515.00 BOOL  ; 进料拉带电机停止条件
515.01 BOOL  ; 扫码NG拉带电机停止条件
515.02 BOOL  ; 氦检NG拉带电机停止条件
515.03 BOOL  ; 0条件
515.04 BOOL  ; 条件
515.05 BOOL  ; 条件
515.06 BOOL  ; 条件
515.07 BOOL  ; 条件
515.08 BOOL  ; 条件
515.09 BOOL  ; 条件
515.10 BOOL  ; 条件
515.11 BOOL  ; 条件
515.12 BOOL  ; 条件
515.13 BOOL  ; 条件
515.14 BOOL  ; 条件
515.15 BOOL  ; 条件
516.00 BOOL  ; #1-1电池抽真空阀关条件
516.01 BOOL  ; #1-2电池抽真空阀关条件
516.02 BOOL  ; #1-1电池注氦阀关条件
516.03 BOOL  ; #1-2电池注氦阀关条件
516.04 BOOL  ; #1-1电池破真空阀关条件
516.05 BOOL  ; #1-2电池破真空阀关条件
516.06 BOOL  ; #2-1电池抽真空阀关条件
516.07 BOOL  ; #2-2电池抽真空阀关条件
516.08 BOOL  ; #2-1电池注氦阀关条件
516.09 BOOL  ; #2-2电池注氦阀关条件
516.10 BOOL  ; #2-1电池破真空阀关条件
516.11 BOOL  ; #2-2电池破真空阀关条件
516.12 BOOL  ; #3-1电池抽真空阀关条件
516.13 BOOL  ; #3-2电池抽真空阀关条件
516.14 BOOL  ; #3-1电池注氦阀关条件
516.15 BOOL  ; #3-2电池注氦阀关条件
517.00 BOOL  ; #3-1电池破真空阀关条件
517.01 BOOL  ; #3-2电池破真空阀关条件
5.00 BOOL  ; #1出料夹爪防下坠感应
5.01 BOOL  ; #2出料夹爪防下坠感应
5.03 BOOL  ; 进料对接输入(停止)
5.04 BOOL  ; 出料对接输入
5.05 BOOL  ; $?St$Bk?_#[5] / 出料旋转气缸9O度位 / $?St$Bk?_#[5]
5.06 BOOL  ; $?St$Bk?_#[6] / 出料旋转气缸O度位 / $?St$Bk?_#[6]
5.07 BOOL  ; 设备总气压信号
5.08 BOOL  ; #1来料位有料感应
5.09 BOOL  ; #2来料位有料感应
5.10 BOOL  ; #1隔离位有料感应
5.11 BOOL  ; #2隔离位有料感应
5.12 BOOL  ; #1扫码位有料感应
5.13 BOOL  ; #2扫码位有料感应
5.14 BOOL  ; #1-1进料位有料感应（光电开关）
5.15 BOOL  ; #1-2进料位有料感应（接近开关）
600.00 BOOL  ; #1扫码阻挡气缸缩回[A]
600.01 BOOL  ; #1扫码阻挡气缸伸出[A]
600.02 BOOL  ; #1隔离气缸缩回[A]
600.03 BOOL  ; #1隔离气缸伸出[A]
600.04 BOOL  ; #2扫码阻挡气缸缩回[A]
600.05 BOOL  ; #2扫码阻挡气缸伸出[A]
600.06 BOOL  ; #2隔离气缸缩回[A]
600.07 BOOL  ; #2隔离气缸伸出[A]
600.08 BOOL  ; #1进料夹爪夹紧[A]
600.09 BOOL  ; #1进料夹爪松开[A]
600.10 BOOL  ; #2进料夹爪夹紧[A]
600.11 BOOL  ; #2进料夹爪松开[A]
600.12 BOOL  ; 进料夹爪变距气缸伸出[A]
600.13 BOOL  ; 进料夹爪变距气缸缩回[A]
600.14 BOOL  ; #1出料夹爪夹紧[A]
600.15 BOOL  ; #1出料夹爪松开[A]
601.00 BOOL  ; #2出料夹爪夹紧[A]
601.01 BOOL  ; #2出料夹爪松开[A]
601.02 BOOL  ; 出料夹爪变距气缸伸出[A]
601.03 BOOL  ; 出料夹爪变距气缸缩回[A]
601.04 BOOL  ; #1腔体平移一级气缸缩回[A]
601.05 BOOL  ; #1腔体平移一级气缸伸出[A]
601.06 BOOL  ; #1腔体平移二级气缸缩回[A]
601.07 BOOL  ; #1腔体平移二级气缸伸出[A]
601.08 BOOL  ; #1腔体顶伸气缸上升[A]
601.09 BOOL  ; #1腔体顶伸气缸下降[A]
601.10 BOOL  ; #1腔体氦检阀开[A]
601.11 BOOL  ; 氦检仪真空阀开[A]
601.12 BOOL  ; #1腔体抽真空阀开[A]
601.13 BOOL  ; #1-1腔体阀开[A]
601.14 BOOL  ; #1-2腔体阀开[A]
601.15 BOOL  ; #1腔体破真空阀开[A]
602.00 BOOL  ; #1腔体吹气阀开[A]
602.01 BOOL  ; #2腔体平移一级气缸缩回[A]
602.02 BOOL  ; #2腔体平移一级气缸伸出[A]
602.03 BOOL  ; #2腔体平移二级气缸缩回[A]
602.04 BOOL  ; #2腔体平移二级气缸伸出[A]
602.05 BOOL  ; #2腔体顶伸气缸上升[A]
602.06 BOOL  ; #2腔体顶伸气缸下降[A]
602.07 BOOL  ; #2腔体氦检阀开[A]
602.08 BOOL  ; 复检清洁阀开[A]
602.09 BOOL  ; #2腔体抽真空阀开[A]
602.10 BOOL  ; #2-1腔体阀开[A]
602.11 BOOL  ; #2-2腔体阀开[A]
602.12 BOOL  ; #2腔体破真空阀开[A]
602.13 BOOL  ; #2腔体吹气阀开[A]
602.14 BOOL  ; #3腔体平移一级气缸缩回[A]
602.15 BOOL  ; #3腔体平移一级气缸伸出[A]
603.00 BOOL  ; #3腔体平移二级气缸缩回[A]
603.01 BOOL  ; #3腔体平移二级气缸伸出[A]
603.02 BOOL  ; #3腔体顶伸气缸上升[A]
603.03 BOOL  ; #3腔体顶伸气缸下降[A]
603.04 BOOL  ; #3腔体氦检阀开[A]
603.05 BOOL  ; 0[A]
603.06 BOOL  ; #3腔体抽真空阀开[A]
603.07 BOOL  ; #3-1腔体阀开[A]
603.08 BOOL  ; #3-2腔体阀开[A]
603.09 BOOL  ; #3腔体破真空阀开[A]
603.10 BOOL  ; #3腔体吹气阀开[A]
603.11 BOOL  ; 进料伺服X轴使能[A]
603.12 BOOL  ; 进料伺服X轴故障复位[A]
603.13 BOOL  ; 进料伺服Z轴使能[A]
603.14 BOOL  ; 进料伺服Z轴故障复位[A]
603.15 BOOL  ; 进料伺服Z轴刹车[A]
604.00 BOOL  ; 出料伺服X轴使能[A]
604.01 BOOL  ; 出料伺服X轴故障复位[A]
604.02 BOOL  ; 出料伺服Z轴使能[A]
604.03 BOOL  ; 出料伺服Z轴故障复位[A]
604.04 BOOL  ; 出料伺服Z轴刹车[A]
604.05 BOOL  ; 腔体抽真空泵启动[A]
604.06 BOOL  ; 0[A]
604.07 BOOL  ; 氦检前置泵启动[A]
604.08 BOOL  ; 氦检仪供电[A]
604.09 BOOL  ; 启动按钮指示灯[A]
604.10 BOOL  ; 停止按钮指示灯[A]
604.11 BOOL  ; 复位按钮指示灯[A]
604.12 BOOL  ; 蜂鸣器[A]
604.13 BOOL  ; 三色灯（红）[A]
604.14 BOOL  ; 三色灯（绿）[A]
604.15 BOOL  ; 三色灯（黄）[A]
605.00 BOOL  ; 进料拉带电机启动[A]
605.01 BOOL  ; 扫码NG拉带电机启动[A]
605.02 BOOL  ; 氦检NG拉带电机启动[A]
605.03 BOOL  ; 进料对接输出[A]
605.04 BOOL  ; 出料对接输出[A]
605.05 BOOL  ; 出料旋转气缸9O度位条件
605.06 BOOL  ; 出料旋转气缸O度位条件
605.07 BOOL  ; 0[A]
605.08 BOOL  ; 0[A]
605.09 BOOL  ; 0[A]
605.10 BOOL  ; 0[A]
605.11 BOOL  ; 0[A]
605.12 BOOL  ; 0[A]
605.13 BOOL  ; 0[A]
605.14 BOOL  ; 0[A]
605.15 BOOL  ; 0[A]
606.00 BOOL  ; #1-1电池抽真空阀开[A]
606.01 BOOL  ; #1-2电池抽真空阀开[A]
606.02 BOOL  ; #1-1电池注氦阀开[A]
606.03 BOOL  ; #1-2电池注氦阀开[A]
606.04 BOOL  ; #1-1电池破真空阀开[A]
606.05 BOOL  ; #1-2电池破真空阀开[A]
606.06 BOOL  ; #2-1电池抽真空阀开[A]
606.07 BOOL  ; #2-2电池抽真空阀开[A]
606.08 BOOL  ; #2-1电池注氦阀开[A]
606.09 BOOL  ; #2-2电池注氦阀开[A]
606.10 BOOL  ; #2-1电池破真空阀开[A]
606.11 BOOL  ; #2-2电池破真空阀开[A]
606.12 BOOL  ; #3-1电池抽真空阀开[A]
606.13 BOOL  ; #3-2电池抽真空阀开[A]
606.14 BOOL  ; #3-1电池注氦阀开[A]
606.15 BOOL  ; #3-2电池注氦阀开[A]
607.00 BOOL  ; #3-1电池破真空阀开[A]
607.01 BOOL  ; #3-2电池破真空阀开[A]
607.02 BOOL  ; 0[A]
607.03 BOOL  ; 0[A]
607.04 BOOL  ; 0[A]
607.05 BOOL  ; 0[A]
607.06 BOOL  ; 0[A]
607.07 BOOL  ; 0[A]
607.08 BOOL  ; 0[A]
607.09 BOOL  ; 0[A]
607.10 BOOL  ; 0[A]
607.11 BOOL  ; 0[A]
607.12 BOOL  ; 0[A]
607.13 BOOL  ; 0[A]
607.14 BOOL  ; 0[A]
607.15 BOOL  ; 0[A]
6100.00 BOOL  ; 出料调试
6100.01 BOOL  ; 出料取料单步
6100.02 BOOL  ; 出料全NG单步
6100.14 BOOL  ; 全NG单步
611.10 BOOL  ; #1腔体氦检阀关[A]
611.11 BOOL  ; 氦检仪真空阀关[A]
611.12 BOOL  ; #1腔体抽真空阀关[A]
611.13 BOOL  ; #1-1腔体阀关[A]
611.14 BOOL  ; #1-2腔体阀关[A]
611.15 BOOL  ; #1腔体破真空阀关[A]
612.00 BOOL  ; #1腔体吹气阀关[A]
612.01 BOOL  ; [A]
612.02 BOOL  ; [A]
612.03 BOOL  ; [A]
612.04 BOOL  ; [A]
612.05 BOOL  ; [A]
612.06 BOOL  ; [A]
612.07 BOOL  ; #2腔体氦检阀关[A]
612.08 BOOL  ; 复检清洁阀关[A]
612.09 BOOL  ; #2腔体抽真空阀关[A]
612.10 BOOL  ; #2-1腔体阀关[A]
612.11 BOOL  ; #2-2腔体阀关[A]
612.12 BOOL  ; #2腔体破真空阀关[A]
612.13 BOOL  ; #2腔体吹气阀关[A]
612.14 BOOL  ; 0[A]
612.15 BOOL  ; [A]
613.00 BOOL  ; [A]
613.01 BOOL  ; [A]
613.02 BOOL  ; [A]
613.03 BOOL  ; [A]
613.04 BOOL  ; #3腔体氦检阀关[A]
613.05 BOOL  ; 0[A]
613.06 BOOL  ; #3腔体抽真空阀关[A]
613.07 BOOL  ; #3-1腔体阀关[A]
613.08 BOOL  ; #3-2腔体阀关[A]
613.09 BOOL  ; #3腔体破真空阀关[A]
613.10 BOOL  ; #3腔体吹气阀关[A]
613.11 BOOL  ; [A]
613.12 BOOL  ; [A]
613.13 BOOL  ; [A]
613.14 BOOL  ; [A]
613.15 BOOL  ; [A]
614.00 BOOL  ; [A]
614.01 BOOL  ; [A]
614.02 BOOL  ; [A]
614.03 BOOL  ; [A]
614.04 BOOL  ; [A]
614.05 BOOL  ; 腔体抽真空泵停止[A]
614.06 BOOL  ; 0[A]
614.07 BOOL  ; 氦检前置泵停止[A]
614.08 BOOL  ; 氦检仪停电[A]
614.09 BOOL  ; [A]
614.10 BOOL  ; [A]
614.11 BOOL  ; [A]
614.12 BOOL  ; [A]
614.13 BOOL  ; [A]
614.14 BOOL  ; [A]
614.15 BOOL  ; [A]
615.00 BOOL  ; 进料拉带电机停止[A]
615.01 BOOL  ; 扫码NG拉带电机停止[A]
615.02 BOOL  ; 氦检NG拉带电机停止[A]
615.03 BOOL  ; 0[A]
615.04 BOOL  ; [A]
615.05 BOOL  ; [A]
615.06 BOOL  ; [A]
615.07 BOOL  ; [A]
615.08 BOOL  ; [A]
615.09 BOOL  ; [A]
615.10 BOOL  ; [A]
615.11 BOOL  ; [A]
615.12 BOOL  ; [A]
615.13 BOOL  ; [A]
615.14 BOOL  ; [A]
615.15 BOOL  ; [A]
616.00 BOOL  ; #1-1电池抽真空阀关[A]
616.01 BOOL  ; #1-2电池抽真空阀关[A]
616.02 BOOL  ; #1-1电池注氦阀关[A]
616.03 BOOL  ; #1-2电池注氦阀关[A]
616.04 BOOL  ; #1-1电池破真空阀关[A]
616.05 BOOL  ; #1-2电池破真空阀关[A]
616.06 BOOL  ; #2-1电池抽真空阀关[A]
616.07 BOOL  ; #2-2电池抽真空阀关[A]
616.08 BOOL  ; #2-1电池注氦阀关[A]
616.09 BOOL  ; #2-2电池注氦阀关[A]
616.10 BOOL  ; #2-1电池破真空阀关[A]
616.11 BOOL  ; #2-2电池破真空阀关[A]
616.12 BOOL  ; #3-1电池抽真空阀关[A]
616.13 BOOL  ; #3-2电池抽真空阀关[A]
616.14 BOOL  ; #3-1电池注氦阀关[A]
616.15 BOOL  ; #3-2电池注氦阀关[A]
617.00 BOOL  ; #3-1电池破真空阀关[A]
617.01 BOOL  ; #3-2电池破真空阀关[A]
650.00 BOOL  ; 进料伺服X轴JOG+[A]
650.01 BOOL  ; 进料伺服X轴JOG-[A]
650.02 BOOL  ; 进料伺服X轴回原点[A]
650.03 BOOL  ; 进料伺服X轴取料位[A]
650.04 BOOL  ; 进料伺服X轴#1腔放料位[A]
650.05 BOOL  ; 进料伺服X轴#2腔放料位[A]
650.06 BOOL  ; 进料伺服X轴#3腔放料位[A]
650.07 BOOL  ; 进料伺服X轴#1夹爪扫码NG放料位[A]
650.08 BOOL  ; 进料伺服X轴#2夹爪扫码NG放料位[A]
650.09 BOOL  ; 进料伺服X轴#1夹爪配对取放料位[A]
650.10 BOOL  ; 进料伺服X轴#2夹爪配对取放料位[A]
650.11 BOOL  ; 进料伺服X轴#1腔有料检测位[A]
650.12 BOOL  ; 进料伺服X轴#2腔有料检测位[A]
650.13 BOOL  ; 进料伺服X轴#3腔有料检测位[A]
650.14 BOOL  ; 0[A]
650.15 BOOL  ; 0[A]
651.00 BOOL  ; 进料伺服Z轴JOG+[A]
651.01 BOOL  ; 进料伺服Z轴JOG-[A]
651.02 BOOL  ; 进料伺服Z轴回原点[A]
651.03 BOOL  ; 进料伺服Z轴待机位[A]
651.04 BOOL  ; 进料伺服Z轴取料位[A]
651.05 BOOL  ; 进料伺服Z轴#1腔放料位[A]
651.06 BOOL  ; 进料伺服Z轴#2腔放料位[A]
651.07 BOOL  ; 进料伺服Z轴#3腔放料位[A]
651.08 BOOL  ; 进料伺服Z轴#1夹爪扫码NG放料位[A]
651.09 BOOL  ; 进料伺服Z轴#2夹爪扫码NG放料位[A]
651.10 BOOL  ; 进料伺服Z轴#1夹爪配对取放料位[A]
651.11 BOOL  ; 进料伺服Z轴#2夹爪配对取放料位[A]
651.12 BOOL  ; 0[A]
651.13 BOOL  ; 0[A]
651.14 BOOL  ; 0[A]
651.15 BOOL  ; 0[A]
652.00 BOOL  ; 出料伺服X轴JOG+[A]
652.01 BOOL  ; 出料伺服X轴JOG-[A]
652.02 BOOL  ; 出料伺服X轴回原点[A]
652.03 BOOL  ; 出料伺服X轴放料位[A]
652.04 BOOL  ; 出料伺服X轴#1腔取料位[A]
652.05 BOOL  ; 出料伺服X轴#2腔取料位[A]
652.06 BOOL  ; 出料伺服X轴#3腔取料位[A]
652.07 BOOL  ; 出料伺服X轴#1夹爪氦检NG放料位[A]
652.08 BOOL  ; 出料伺服X轴#2夹爪氦检NG放料位[A]
652.09 BOOL  ; 出料伺服X轴#1夹爪配对取放料位[A]
652.10 BOOL  ; 出料伺服X轴#2夹爪配对取放料位[A]
652.11 BOOL  ; 0[A]
652.12 BOOL  ; 0[A]
652.13 BOOL  ; 0[A]
652.14 BOOL  ; 0[A]
652.15 BOOL  ; 0[A]
653.00 BOOL  ; 出料伺服Z轴JOG+[A]
653.01 BOOL  ; 出料伺服Z轴JOG-[A]
653.02 BOOL  ; 出料伺服Z轴回原点[A]
653.03 BOOL  ; 出料伺服Z轴待机位[A]
653.04 BOOL  ; 出料伺服Z轴放料位[A]
653.05 BOOL  ; 出料伺服Z轴#1腔取料位[A]
653.06 BOOL  ; 出料伺服Z轴#2腔取料位[A]
653.07 BOOL  ; 出料伺服Z轴#3腔取料位[A]
653.08 BOOL  ; 出料伺服Z轴#1夹爪氦检NG放料位[A]
653.09 BOOL  ; 出料伺服Z轴#2夹爪氦检NG放料位[A]
653.10 BOOL  ; 出料伺服Z轴#1夹爪配对取放料位[A]
653.11 BOOL  ; 出料伺服Z轴#2夹爪配对取放料位[A]
6.00 BOOL  ; #2-1进料位有料感应（光电开关）
6.01 BOOL  ; #2-2进料位有料感应（接近开关）
6.02 BOOL  ; 进料夹爪柔性感应
6.03 BOOL  ; 出料夹爪柔性感应
6.04 BOOL  ; #1进料夹爪对应腔体有料感应
6.05 BOOL  ; #2进料夹爪对应腔体有料感应
6.06 BOOL  ; 扫码NG放料#1位有料感应
6.07 BOOL  ; 扫码NG放料#2位有料感应
6.08 BOOL  ; 扫码NG料满位有料感应
6.09 BOOL  ; 进料配对位有料感应
6.10 BOOL  ; 出料配对位有料感应
6.11 BOOL  ; 氦检NG放料#1位有料感应
6.12 BOOL  ; 氦检NG放料#2位有料感应
6.13 BOOL  ; 氦检NG料满位有料感应
6.14 BOOL  ; #1-1出料位有料感应
6.15 BOOL  ; #1-2出料位有料感应
700 CHANNEL  ; 手动按钮操作字
700.00 BOOL  ; #1扫码阻挡气缸缩回[SW]
700.01 BOOL  ; #1扫码阻挡气缸伸出[SW]
700.02 BOOL  ; #1隔离气缸缩回[SW]
700.03 BOOL  ; #1隔离气缸伸出[SW]
700.04 BOOL  ; #2扫码阻挡气缸缩回[SW]
700.05 BOOL  ; #2扫码阻挡气缸伸出[SW]
700.06 BOOL  ; #2隔离气缸缩回[SW]
700.07 BOOL  ; #2隔离气缸伸出[SW]
700.08 BOOL  ; #1进料夹爪夹紧[SW]
700.09 BOOL  ; #1进料夹爪松开[SW]
700.10 BOOL  ; #2进料夹爪夹紧[SW]
700.11 BOOL  ; #2进料夹爪松开[SW]
700.12 BOOL  ; 进料夹爪变距气缸伸出[SW]
700.13 BOOL  ; 进料夹爪变距气缸缩回[SW]
700.14 BOOL  ; #1出料夹爪夹紧[SW]
700.15 BOOL  ; #1出料夹爪松开[SW]
701.00 BOOL  ; #2出料夹爪夹紧[SW]
701.01 BOOL  ; #2出料夹爪松开[SW]
701.02 BOOL  ; 出料夹爪变距气缸伸出[SW]
701.03 BOOL  ; 出料夹爪变距气缸缩回[SW]
701.04 BOOL  ; #1腔体平移一级气缸缩回[SW]
701.05 BOOL  ; #1腔体平移一级气缸伸出[SW]
701.06 BOOL  ; #1腔体平移二级气缸缩回[SW]
701.07 BOOL  ; #1腔体平移二级气缸伸出[SW]
701.08 BOOL  ; #1腔体顶伸气缸上升[SW]
701.09 BOOL  ; #1腔体顶伸气缸下降[SW]
701.10 BOOL  ; #1腔体氦检阀开[SW]
701.11 BOOL  ; 氦检仪真空阀开[SW]
701.12 BOOL  ; #1腔体抽真空阀开[SW]
701.13 BOOL  ; #1-1腔体阀开[SW]
701.14 BOOL  ; #1-2腔体阀开[SW]
701.15 BOOL  ; #1腔体破真空阀开[SW]
702.00 BOOL  ; #1腔体吹气阀开[SW]
702.01 BOOL  ; #2腔体平移一级气缸缩回[SW]
702.02 BOOL  ; #2腔体平移一级气缸伸出[SW]
702.03 BOOL  ; #2腔体平移二级气缸缩回[SW]
702.04 BOOL  ; #2腔体平移二级气缸伸出[SW]
702.05 BOOL  ; #2腔体顶伸气缸上升[SW]
702.06 BOOL  ; #2腔体顶伸气缸下降[SW]
702.07 BOOL  ; #2腔体氦检阀开[SW]
702.08 BOOL  ; 复检清洁阀开[SW]
702.09 BOOL  ; #2腔体抽真空阀开[SW]
702.10 BOOL  ; #2-1腔体阀开[SW]
702.11 BOOL  ; #2-2腔体阀开[SW]
702.12 BOOL  ; #2腔体破真空阀开[SW]
702.13 BOOL  ; #2腔体吹气阀开[SW]
702.14 BOOL  ; #3腔体平移一级气缸缩回[SW]
702.15 BOOL  ; #3腔体平移一级气缸伸出[SW]
703.00 BOOL  ; #3腔体平移二级气缸缩回[SW]
703.01 BOOL  ; #3腔体平移二级气缸伸出[SW]
703.02 BOOL  ; #3腔体顶伸气缸上升[SW]
703.03 BOOL  ; #3腔体顶伸气缸下降[SW]
703.04 BOOL  ; #3腔体氦检阀开[SW]
703.05 BOOL  ; 0[SW]
703.06 BOOL  ; #3腔体抽真空阀开[SW]
703.07 BOOL  ; #3-1腔体阀开[SW]
703.08 BOOL  ; #3-2腔体阀开[SW]
703.09 BOOL  ; #3腔体破真空阀开[SW]
703.10 BOOL  ; #3腔体吹气阀开[SW]
703.11 BOOL  ; 进料伺服X轴使能[SW]
703.12 BOOL  ; 进料伺服X轴故障复位[SW]
703.13 BOOL  ; 进料伺服Z轴使能[SW]
703.14 BOOL  ; 进料伺服Z轴故障复位[SW]
703.15 BOOL  ; 进料伺服Z轴刹车[SW]
704.00 BOOL  ; 出料伺服X轴使能[SW]
704.01 BOOL  ; 出料伺服X轴故障复位[SW]
704.02 BOOL  ; 出料伺服Z轴使能[SW]
704.03 BOOL  ; 出料伺服Z轴故障复位[SW]
704.04 BOOL  ; 出料伺服Z轴刹车[SW]
704.05 BOOL  ; 腔体抽真空泵启动[SW]
704.06 BOOL  ; 0[SW]
704.07 BOOL  ; 氦检前置泵启动[SW]
704.08 BOOL  ; 氦检仪供电[SW]
704.09 BOOL  ; 启动按钮指示灯[SW]
704.10 BOOL  ; 停止按钮指示灯[SW]
704.11 BOOL  ; 复位按钮指示灯[SW]
704.12 BOOL  ; 蜂鸣器[SW]
704.13 BOOL  ; 三色灯（红）[SW]
704.14 BOOL  ; 三色灯（绿）[SW]
704.15 BOOL  ; 三色灯（黄）[SW]
705 CHANNEL  ; 手动按钮操作字
705.00 BOOL  ; 进料拉带电机启动[SW]
705.01 BOOL  ; 扫码NG拉带电机启动[SW]
705.02 BOOL  ; 氦检NG拉带电机启动[SW]
705.03 BOOL  ; 进料对接输出[SW]
705.04 BOOL  ; 出料对接输出[SW]
705.05 BOOL  ; 出料旋转气缸9O度位条件
705.06 BOOL  ; 出料旋转气缸O度位条件
705.07 BOOL  ; 0[SW]
705.08 BOOL  ; 0[SW]
705.09 BOOL  ; 0[SW]
705.10 BOOL  ; 0[SW]
705.11 BOOL  ; 0[SW]
705.12 BOOL  ; 0[SW]
705.13 BOOL  ; 0[SW]
705.14 BOOL  ; 0[SW]
705.15 BOOL  ; 0[SW]
706 CHANNEL  ; 手动按钮操作字
706.00 BOOL  ; #1-1电池抽真空阀开[SW]
706.01 BOOL  ; #1-2电池抽真空阀开[SW]
706.02 BOOL  ; #1-1电池注氦阀开[SW]
706.03 BOOL  ; #1-2电池注氦阀开[SW]
706.04 BOOL  ; #1-1电池破真空阀开[SW]
706.05 BOOL  ; #1-2电池破真空阀开[SW]
706.06 BOOL  ; #2-1电池抽真空阀开[SW]
706.07 BOOL  ; #2-2电池抽真空阀开[SW]
706.08 BOOL  ; #2-1电池注氦阀开[SW]
706.09 BOOL  ; #2-2电池注氦阀开[SW]
706.10 BOOL  ; #2-1电池破真空阀开[SW]
706.11 BOOL  ; #2-2电池破真空阀开[SW]
706.12 BOOL  ; #3-1电池抽真空阀开[SW]
706.13 BOOL  ; #3-2电池抽真空阀开[SW]
706.14 BOOL  ; #3-1电池注氦阀开[SW]
706.15 BOOL  ; #3-2电池注氦阀开[SW]
707.00 BOOL  ; #3-1电池破真空阀开[SW]
707.01 BOOL  ; #3-2电池破真空阀开[SW]
707.02 BOOL  ; 0[SW]
707.03 BOOL  ; 0[SW]
707.04 BOOL  ; 0[SW]
707.05 BOOL  ; 0[SW]
707.06 BOOL  ; 0[SW]
707.07 BOOL  ; 0[SW]
707.08 BOOL  ; 0[SW]
707.09 BOOL  ; 0[SW]
707.10 BOOL  ; 0[SW]
707.11 BOOL  ; 0[SW]
707.12 BOOL  ; 0[SW]
707.13 BOOL  ; 0[SW]
707.14 BOOL  ; 0[SW]
707.15 BOOL  ; 0[SW]
711 CHANNEL  ; 手动按钮操作字
711.10 BOOL  ; #1腔体氦检阀关[SW]
711.11 BOOL  ; 氦检仪真空阀关[SW]
711.12 BOOL  ; #1腔体抽真空阀关[SW]
711.13 BOOL  ; #1-1腔体阀关[SW]
711.14 BOOL  ; #1-2腔体阀关[SW]
711.15 BOOL  ; #1腔体破真空阀关[SW]
712.00 BOOL  ; #1腔体吹气阀关[SW]
712.01 BOOL  ; [SW]
712.02 BOOL  ; [SW]
712.03 BOOL  ; [SW]
712.04 BOOL  ; [SW]
712.05 BOOL  ; [SW]
712.06 BOOL  ; [SW]
712.07 BOOL  ; #2腔体氦检阀关[SW]
712.08 BOOL  ; 复检清洁阀关[SW]
712.09 BOOL  ; #2腔体抽真空阀关[SW]
712.10 BOOL  ; #2-1腔体阀关[SW]
712.11 BOOL  ; #2-2腔体阀关[SW]
712.12 BOOL  ; #2腔体破真空阀关[SW]
712.13 BOOL  ; #2腔体吹气阀关[SW]
712.14 BOOL  ; 0[SW]
712.15 BOOL  ; [SW]
713.00 BOOL  ; [SW]
713.01 BOOL  ; [SW]
713.02 BOOL  ; [SW]
713.03 BOOL  ; [SW]
713.04 BOOL  ; #3腔体氦检阀关[SW]
713.05 BOOL  ; 0[SW]
713.06 BOOL  ; #3腔体抽真空阀关[SW]
713.07 BOOL  ; #3-1腔体阀关[SW]
713.08 BOOL  ; #3-2腔体阀关[SW]
713.09 BOOL  ; #3腔体破真空阀关[SW]
713.10 BOOL  ; #3腔体吹气阀关[SW]
713.11 BOOL  ; [SW]
713.12 BOOL  ; [SW]
713.13 BOOL  ; [SW]
713.14 BOOL  ; [SW]
713.15 BOOL  ; [SW]
714.00 BOOL  ; [SW]
714.01 BOOL  ; [SW]
714.02 BOOL  ; [SW]
714.03 BOOL  ; [SW]
714.04 BOOL  ; [SW]
714.05 BOOL  ; 腔体抽真空泵停止[SW]
714.06 BOOL  ; 0[SW]
714.07 BOOL  ; 氦检前置泵停止[SW]
714.08 BOOL  ; 氦检仪停电[SW]
714.09 BOOL  ; [SW]
714.10 BOOL  ; [SW]
714.11 BOOL  ; [SW]
714.12 BOOL  ; [SW]
714.13 BOOL  ; [SW]
714.14 BOOL  ; [SW]
714.15 BOOL  ; [SW]
715 CHANNEL  ; 手动按钮操作字
715.00 BOOL  ; 进料拉带电机停止[SW]
715.01 BOOL  ; 扫码NG拉带电机停止[SW]
715.02 BOOL  ; 氦检NG拉带电机停止[SW]
715.03 BOOL  ; 0[SW]
715.04 BOOL  ; [SW]
715.05 BOOL  ; [SW]
715.06 BOOL  ; [SW]
715.07 BOOL  ; [SW]
715.08 BOOL  ; [SW]
715.09 BOOL  ; [SW]
715.10 BOOL  ; [SW]
715.11 BOOL  ; [SW]
715.12 BOOL  ; [SW]
715.13 BOOL  ; [SW]
715.14 BOOL  ; [SW]
715.15 BOOL  ; [SW]
716 CHANNEL  ; 手动按钮操作字
716.00 BOOL  ; #1-1电池抽真空阀关[SW]
716.01 BOOL  ; #1-2电池抽真空阀关[SW]
716.02 BOOL  ; #1-1电池注氦阀关[SW]
716.03 BOOL  ; #1-2电池注氦阀关[SW]
716.04 BOOL  ; #1-1电池破真空阀关[SW]
716.05 BOOL  ; #1-2电池破真空阀关[SW]
716.06 BOOL  ; #2-1电池抽真空阀关[SW]
716.07 BOOL  ; #2-2电池抽真空阀关[SW]
716.08 BOOL  ; #2-1电池注氦阀关[SW]
716.09 BOOL  ; #2-2电池注氦阀关[SW]
716.10 BOOL  ; #2-1电池破真空阀关[SW]
716.11 BOOL  ; #2-2电池破真空阀关[SW]
716.12 BOOL  ; #3-1电池抽真空阀关[SW]
716.13 BOOL  ; #3-2电池抽真空阀关[SW]
716.14 BOOL  ; #3-1电池注氦阀关[SW]
716.15 BOOL  ; #3-2电池注氦阀关[SW]
717.00 BOOL  ; #3-1电池破真空阀关[SW]
717.01 BOOL  ; #3-2电池破真空阀关[SW]
750.00 BOOL  ; 进料伺服X轴JOG+[SW]
750.01 BOOL  ; 进料伺服X轴JOG-[SW]
750.02 BOOL  ; 进料伺服X轴回原点[SW]
750.03 BOOL  ; 进料伺服X轴取料位[SW]
750.04 BOOL  ; 进料伺服X轴#1腔放料位[SW]
750.05 BOOL  ; 进料伺服X轴#2腔放料位[SW]
750.06 BOOL  ; 进料伺服X轴#3腔放料位[SW]
750.07 BOOL  ; 进料伺服X轴#1夹爪扫码NG放料位[SW]
750.08 BOOL  ; 进料伺服X轴#2夹爪扫码NG放料位[SW]
750.09 BOOL  ; 进料伺服X轴#1夹爪配对取放料位[SW]
750.10 BOOL  ; 进料伺服X轴#2夹爪配对取放料位[SW]
750.11 BOOL  ; 进料伺服X轴#1腔有料检测位[SW]
750.12 BOOL  ; 进料伺服X轴#2腔有料检测位[SW]
750.13 BOOL  ; 进料伺服X轴#3腔有料检测位[SW]
750.14 BOOL  ; 0[SW]
750.15 BOOL  ; 0[SW]
751.00 BOOL  ; 进料伺服Z轴JOG+[SW]
751.01 BOOL  ; 进料伺服Z轴JOG-[SW]
751.02 BOOL  ; 进料伺服Z轴回原点[SW]
751.03 BOOL  ; 进料伺服Z轴待机位[SW]
751.04 BOOL  ; 进料伺服Z轴取料位[SW]
751.05 BOOL  ; 进料伺服Z轴#1腔放料位[SW]
751.06 BOOL  ; 进料伺服Z轴#2腔放料位[SW]
751.07 BOOL  ; 进料伺服Z轴#3腔放料位[SW]
751.08 BOOL  ; 进料伺服Z轴#1夹爪扫码NG放料位[SW]
751.09 BOOL  ; 进料伺服Z轴#2夹爪扫码NG放料位[SW]
751.10 BOOL  ; 进料伺服Z轴#1夹爪配对取放料位[SW]
751.11 BOOL  ; 进料伺服Z轴#2夹爪配对取放料位[SW]
751.12 BOOL  ; 0[SW]
751.13 BOOL  ; 0[SW]
751.14 BOOL  ; 0[SW]
751.15 BOOL  ; 进料伺服Z轴跟踪开选择（跟踪=1）[SW]
752 CHANNEL  ; 出料模组X/Z联动需求
752.00 BOOL  ; 出料伺服X轴JOG+[SW]
752.01 BOOL  ; 出料伺服X轴JOG-[SW]
752.02 BOOL  ; 出料伺服X轴回原点[SW]
752.03 BOOL  ; 出料伺服X轴放料位[SW]
752.04 BOOL  ; 出料伺服X轴#1腔取料位[SW]
752.05 BOOL  ; 出料伺服X轴#2腔取料位[SW]
752.06 BOOL  ; 出料伺服X轴#3腔取料位[SW]
752.07 BOOL  ; 出料伺服X轴#1夹爪氦检NG放料位[SW]
752.08 BOOL  ; 出料伺服X轴#2夹爪氦检NG放料位[SW]
752.09 BOOL  ; 出料伺服X轴#1夹爪配对取放料位[SW]
752.10 BOOL  ; 出料伺服X轴#2夹爪配对取放料位[SW]
752.11 BOOL  ; 0[SW]
752.12 BOOL  ; 0[SW]
752.13 BOOL  ; 0[SW]
752.14 BOOL  ; 0[SW]
752.15 BOOL  ; 0[SW]
753.00 BOOL  ; 出料伺服Z轴JOG+[SW]
753.01 BOOL  ; 出料伺服Z轴JOG-[SW]
753.02 BOOL  ; 出料伺服Z轴回原点[SW]
753.03 BOOL  ; 出料伺服Z轴待机位[SW]
753.04 BOOL  ; 出料伺服Z轴放料位[SW]
753.05 BOOL  ; 出料伺服Z轴#1腔取料位[SW]
753.06 BOOL  ; 出料伺服Z轴#2腔取料位[SW]
753.07 BOOL  ; 出料伺服Z轴#3腔取料位[SW]
753.08 BOOL  ; 出料伺服Z轴#1夹爪氦检NG放料位[SW]
753.09 BOOL  ; 出料伺服Z轴#2夹爪氦检NG放料位[SW]
753.10 BOOL  ; 出料伺服Z轴#1夹爪配对取放料位[SW]
753.11 BOOL  ; 出料伺服Z轴#2夹爪配对取放料位[SW]
753.15 BOOL  ; 出料伺服Z轴跟踪开选择[SW]
7.00 BOOL  ; #2-1出料位有料感应
7.01 BOOL  ; #2-2出料位有料感应
7.02 BOOL  ; #1门磁开关
7.03 BOOL  ; #2门磁开关
7.04 BOOL  ; #3门磁开关
7.05 BOOL  ; #4门磁开关
7.06 BOOL  ; #5门磁开关
7.07 BOOL  ; #6门磁开关
7.08 BOOL  ; #7门磁开关
7.09 BOOL  ; #8门磁开关
7.10 BOOL  ; #9门磁开关
7.11 BOOL  ; #10门磁开关
7.12 BOOL  ; #11门磁开关
7.13 BOOL  ; 设备真空压力信号
7.14 BOOL  ; 设备氦气压力信号
7.15 BOOL  ; 精密调压阀信号
800.00 BOOL  ; #1扫码阻挡气缸缩回位标志[0000.00]
800.01 BOOL  ; #1扫码阻挡气缸伸出位标志[0000.01]
800.02 BOOL  ; #1隔离气缸缩回位标志[0000.02]
800.03 BOOL  ; 0标志[0000.03]
800.04 BOOL  ; #2扫码阻挡气缸缩回位标志[0000.04]
800.05 BOOL  ; #2扫码阻挡气缸伸出位标志[0000.05]
800.06 BOOL  ; #2隔离气缸缩回位标志[0000.06]
800.07 BOOL  ; 0标志[0000.07]
800.08 BOOL  ; #1进料夹爪夹紧位标志[0000.08]
800.09 BOOL  ; #1进料夹爪松开位标志[0000.09]
800.10 BOOL  ; #2进料夹爪夹紧位标志[0000.10]
800.11 BOOL  ; #2进料夹爪松开位标志[0000.11]
800.12 BOOL  ; 进料夹爪变距气缸伸出位标志[0000.12]
800.13 BOOL  ; 进料夹爪变距气缸缩回位标志[0000.13]
800.14 BOOL  ; #1出料夹爪夹紧位标志[0000.14]
800.15 BOOL  ; #1出料夹爪松开位标志[0000.15]
801.00 BOOL  ; #2出料夹爪夹紧位标志[0001.00]
801.01 BOOL  ; #2出料夹爪松开位标志[0001.01]
801.02 BOOL  ; 出料夹爪变距气缸伸出位标志[0001.02]
801.03 BOOL  ; 出料夹爪变距气缸缩回位标志[0001.03]
801.04 BOOL  ; #1腔体平移一级气缸缩回位标志[0001.04]
801.05 BOOL  ; #1腔体平移一级气缸伸出位标志[0001.05]
801.06 BOOL  ; #1腔体平移二级气缸缩回位标志[0001.06]
801.07 BOOL  ; #1腔体平移二级气缸伸出位标志[0001.07]
801.08 BOOL  ; #1腔体顶伸气缸上升位标志[0001.08]
801.09 BOOL  ; #1腔体顶伸气缸下降位标志[0001.09]
801.10 BOOL  ; #1腔体氦检阀开到位标志[0001.10]
801.11 BOOL  ; #1腔体氦检阀关到位标志[0001.11]
801.12 BOOL  ; 0标志[0001.12]
801.13 BOOL  ; 0标志[0001.13]
801.14 BOOL  ; 0标志[0001.14]
801.15 BOOL  ; 0标志[0001.15]
802.00 BOOL  ; 0标志[0002.00]
802.01 BOOL  ; #2腔体平移一级气缸缩回位标志[0002.01]
802.02 BOOL  ; #2腔体平移一级气缸伸出位标志[0002.02]
802.03 BOOL  ; #2腔体平移二级气缸缩回位标志[0002.03]
802.04 BOOL  ; #2腔体平移二级气缸伸出位标志[0002.04]
802.05 BOOL  ; #2腔体顶伸气缸上升位标志[0002.05]
802.06 BOOL  ; #2腔体顶伸气缸下降位标志[0002.06]
802.07 BOOL  ; #2腔体氦检阀开到位标志[0002.07]
802.08 BOOL  ; #2腔体氦检阀关到位标志[0002.08]
802.09 BOOL  ; 0标志[0002.09]
802.10 BOOL  ; 0标志[0002.10]
802.11 BOOL  ; 0标志[0002.11]
802.12 BOOL  ; 0标志[0002.12]
802.13 BOOL  ; 0标志[0002.13]
802.14 BOOL  ; #3腔体平移一级气缸缩回位标志[0002.14]
802.15 BOOL  ; #3腔体平移一级气缸伸出位标志[0002.15]
803.00 BOOL  ; #3腔体平移二级气缸缩回位标志[0003.00]
803.01 BOOL  ; #3腔体平移二级气缸伸出位标志[0003.01]
803.02 BOOL  ; #3腔体顶伸气缸上升位标志[0003.02]
803.03 BOOL  ; #3腔体顶伸气缸下降位标志[0003.03]
803.04 BOOL  ; #3腔体氦检阀开到位标志[0003.04]
803.05 BOOL  ; #3腔体氦检阀关到位标志[0003.05]
803.06 BOOL  ; 氦检仪准备好了信号标志[0003.06]
803.07 BOOL  ; 氦检仪故障信号标志[0003.07]
803.08 BOOL  ; 0标志[0003.08]
803.09 BOOL  ; 0标志[0003.09]
803.10 BOOL  ; 0标志[0003.10]
803.11 BOOL  ; 进料伺服X轴准备好了信号标志[0003.11]
803.12 BOOL  ; 进料伺服X轴故障信号标志[0003.12]
803.13 BOOL  ; 进料伺服Z轴准备好了信号标志[0003.13]
803.14 BOOL  ; 进料伺服Z轴故障信号标志[0003.14]
803.15 BOOL  ; 0标志[0003.15]
804.00 BOOL  ; 出料伺服X轴准备好了信号标志[0004.00]
804.01 BOOL  ; 出料伺服X轴故障信号标志[0004.01]
804.02 BOOL  ; 出料伺服Z轴准备好了信号标志[0004.02]
804.03 BOOL  ; 出料伺服Z轴故障信号标志[0004.03]
804.04 BOOL  ; 0标志[0004.04]
804.05 BOOL  ; 腔体抽真空泵运行信号标志[0004.05]
804.06 BOOL  ; 腔体抽真空泵过载信号标志[0004.06]
804.07 BOOL  ; 氦检前置泵运行信号标志[0004.07]
804.08 BOOL  ; 氦检前置泵过载信号标志[0004.08]
804.09 BOOL  ; 启动按钮标志[0004.09]
804.10 BOOL  ; 停止按钮标志[0004.10]
804.11 BOOL  ; 复位按钮标志[0004.11]
804.12 BOOL  ; $?St$Bk?_#[7] / 急停按钮标志[0004.12] / $?St$Bk?_#[7]
804.13 BOOL  ; 手自动选择标志[0004.13]
804.14 BOOL  ; #1进料夹爪防下坠感应标志[0004.14]
804.15 BOOL  ; #2进料夹爪防下坠感应标志[0004.15]
805.00 BOOL  ; #1出料夹爪防下坠感应标志[0005.00]
805.01 BOOL  ; #2出料夹爪防下坠感应标志[0005.01]
805.02 BOOL  ; 0标志[0005.02]
805.03 BOOL  ; 进料对接输入(停止)标志[0005.03]
805.04 BOOL  ; 出料对接输入标志（1-允许放料）[0005.04]
805.05 BOOL  ; 出料旋转气缸9O度位条件
805.06 BOOL  ; 出料旋转气缸O度位条件
805.07 BOOL  ; 设备总气压信号标志[0005.07]
805.08 BOOL  ; #1来料位有料感应标志[0005.08]
805.09 BOOL  ; #2来料位有料感应标志[0005.09]
805.10 BOOL  ; #1隔离位有料感应标志[0005.10]
805.11 BOOL  ; #2隔离位有料感应标志[0005.11]
805.12 BOOL  ; #1扫码位有料感应标志[0005.12]
805.13 BOOL  ; #2扫码位有料感应标志[0005.13]
805.14 BOOL  ; #1-1进料位有料感应标志[0005.14]
805.15 BOOL  ; #1-2进料位有料感应标志[0005.15]
806.00 BOOL  ; #2-1进料位有料感应标志[0006.00]
806.01 BOOL  ; #2-2进料位有料感应标志[0006.01]
806.02 BOOL  ; 进料夹爪柔性感应标志[0006.02]
806.03 BOOL  ; 出料夹爪柔性感应标志[0006.03]
806.04 BOOL  ; #1进料夹爪对应腔体有料感应标志[0006.04]
806.05 BOOL  ; #2进料夹爪对应腔体有料感应标志[0006.05]
806.06 BOOL  ; 扫码NG放料#1位有料感应标志[0006.06]
806.07 BOOL  ; 扫码NG放料#2位有料感应标志[0006.07]
806.08 BOOL  ; 扫码NG料满位有料感应标志[0006.08]
806.09 BOOL  ; 进料配对位有料感应标志[0006.09]
806.10 BOOL  ; 出料配对位有料感应标志[0006.10]
806.11 BOOL  ; 氦检NG放料#1位有料感应标志[0006.11]
806.12 BOOL  ; 氦检NG放料#2位有料感应标志[0006.12]
806.13 BOOL  ; 氦检NG料满位有料感应标志[0006.13]
806.14 BOOL  ; #1-1出料位有料感应标志[0006.14]
806.15 BOOL  ; #1-2出料位有料感应标志[0006.15]
807.00 BOOL  ; #2-1出料位有料感应标志[0007.00]
807.01 BOOL  ; #2-2出料位有料感应标志[0007.01]
807.02 BOOL  ; #1门磁开关标志[0007.02]
807.03 BOOL  ; #2门磁开关标志[0007.03]
807.04 BOOL  ; #3门磁开关标志[0007.04]
807.05 BOOL  ; #4门磁开关标志[0007.05]
807.06 BOOL  ; #5门磁开关标志[0007.06]
807.07 BOOL  ; #6门磁开关标志[0007.07]
807.08 BOOL  ; #7门磁开关标志[0007.08]
807.09 BOOL  ; #8门磁开关标志[0007.09]
807.10 BOOL  ; #9门磁开关标志[0007.10]
807.11 BOOL  ; #10门磁开关标志[0007.11]
807.12 BOOL  ; #11门磁开关标志[0007.12]
807.13 BOOL  ; 设备真空压力信号标志[0007.13]
807.14 BOOL  ; 设备氦气压力信号标志[0007.14]
807.15 BOOL  ; 精密调压阀信号标志[0007.15]
810.03 BOOL  ; $?St$Bk?_#[8] / #1隔离气缸伸出位标志 / $?St$Bk?_#[8]
810.07 BOOL  ; $?St$Bk?_#[9] / #2隔离气缸伸出位标志 / $?St$Bk?_#[9]
820.08 BOOL  ; $?St$Bk?_#[10] / 标漏阀开到位标志 / $?St$Bk?_#[10]
820.09 BOOL  ; $?St$Bk?_#[11] / 标漏阀关到位标志 / $?St$Bk?_#[11]
820.10 BOOL  ; 氦检仪真空阀开到位标志
820.11 BOOL  ; 氦检仪真空阀关到位标志
820.12 BOOL  ; 复检清洁阀开到位标志
820.13 BOOL  ; 复检清洁阀关到位标志
820.14 BOOL  ; #1腔体抽真空阀开到位标志
820.15 BOOL  ; #1腔体抽真空阀关到位标志
821.00 BOOL  ; #1-1腔体阀开到位标志
821.01 BOOL  ; #1-1腔体阀关到位标志
821.02 BOOL  ; #1-2腔体阀开到位标志
821.03 BOOL  ; #1-2腔体阀关到位标志
821.04 BOOL  ; #1腔体破真空阀开到位标志
821.05 BOOL  ; #1腔体破真空阀关到位标志
821.06 BOOL  ; #1腔体吹气阀开到位标志
821.07 BOOL  ; #1腔体吹气阀关到位标志
821.08 BOOL  ; #2腔体抽真空阀开到位标志
821.09 BOOL  ; #2腔体抽真空阀关到位标志
821.10 BOOL  ; #2-1腔体阀开到位标志
821.11 BOOL  ; #2-1腔体阀关到位标志
821.12 BOOL  ; #2-2腔体阀开到位标志
821.13 BOOL  ; #2-2腔体阀关到位标志
821.14 BOOL  ; #2腔体破真空阀开到位标志
821.15 BOOL  ; #2腔体破真空阀关到位标志
822.00 BOOL  ; #2腔体吹气阀开到位标志
822.01 BOOL  ; #2腔体吹气阀关到位标志
822.02 BOOL  ; #3腔体抽真空阀开到位标志
822.03 BOOL  ; #3腔体抽真空阀关到位标志
822.04 BOOL  ; #3-1腔体阀开到位标志
822.05 BOOL  ; #3-1腔体阀关到位标志
822.06 BOOL  ; #3-2腔体阀开到位标志
822.07 BOOL  ; #3-2腔体阀关到位标志
822.08 BOOL  ; #3腔体破真空阀开到位标志
822.09 BOOL  ; #3腔体破真空阀关到位标志
822.10 BOOL  ; #3腔体吹气阀开到位标志
822.11 BOOL  ; #3腔体吹气阀关到位标志
822.12 BOOL  ; #1-1电池抽真空阀开到位标志
822.13 BOOL  ; #1-1电池抽真空阀关到位标志
822.14 BOOL  ; #1-2电池抽真空阀开到位标志
822.15 BOOL  ; #1-2电池抽真空阀关到位标志
823.00 BOOL  ; #1-1电池注氦阀开到位标志
823.01 BOOL  ; #1-1电池注氦阀关到位标志
823.02 BOOL  ; #1-2电池注氦阀开到位标志
823.03 BOOL  ; #1-2电池注氦阀关到位标志
823.04 BOOL  ; #1-1电池破真空阀开到位标志
823.05 BOOL  ; #1-1电池破真空阀关到位标志
823.06 BOOL  ; #1-2电池破真空阀开到位标志
823.07 BOOL  ; #1-2电池破真空阀关到位标志
823.08 BOOL  ; #2-1电池抽真空阀开到位标志
823.09 BOOL  ; #2-1电池抽真空阀关到位标志
823.10 BOOL  ; #2-2电池抽真空阀开到位标志
823.11 BOOL  ; #2-2电池抽真空阀关到位标志
823.12 BOOL  ; #2-1电池注氦阀开到位标志
823.13 BOOL  ; #2-1电池注氦阀关到位标志
823.14 BOOL  ; #2-2电池注氦阀开到位标志
823.15 BOOL  ; #2-2电池注氦阀关到位标志
824.00 BOOL  ; #2-1电池破真空阀开到位标志
824.01 BOOL  ; #2-1电池破真空阀关到位标志
824.02 BOOL  ; #2-2电池破真空阀开到位标志
824.03 BOOL  ; #2-2电池破真空阀关到位标志
824.04 BOOL  ; #3-1电池抽真空阀开到位标志
824.05 BOOL  ; #3-1电池抽真空阀关到位标志
824.06 BOOL  ; #3-2电池抽真空阀开到位标志
824.07 BOOL  ; #3-2电池抽真空阀关到位标志
824.08 BOOL  ; #3-1电池注氦阀开到位标志
824.09 BOOL  ; #3-1电池注氦阀关到位标志
824.10 BOOL  ; #3-2电池注氦阀开到位标志
824.11 BOOL  ; #3-2电池注氦阀关到位标志
824.12 BOOL  ; #3-1电池破真空阀开到位标志
824.13 BOOL  ; #3-1电池破真空阀关到位标志
824.14 BOOL  ; #3-2电池破真空阀开到位标志
824.15 BOOL  ; #3-2电池破真空阀关到位标志
850.00 BOOL  ; 进料伺服X轴JOG+标志
850.01 BOOL  ; 进料伺服X轴JOG-标志
850.02 BOOL  ; 进料伺服X轴回原点标志
850.03 BOOL  ; 进料伺服X轴取料位标志
850.04 BOOL  ; 进料伺服X轴#1腔放料位标志
850.05 BOOL  ; 进料伺服X轴#2腔放料位标志
850.06 BOOL  ; 进料伺服X轴#3腔放料位标志
850.07 BOOL  ; 进料伺服X轴#1夹爪扫码NG放料位标志
850.08 BOOL  ; 进料伺服X轴#2夹爪扫码NG放料位标志
850.09 BOOL  ; 进料伺服X轴#1夹爪配对取放料位标志
850.10 BOOL  ; 进料伺服X轴#2夹爪配对取放料位标志
850.11 BOOL  ; 进料伺服X轴#1腔有料检测位标志
850.12 BOOL  ; 进料伺服X轴#2腔有料检测位标志
850.13 BOOL  ; 进料伺服X轴#3腔有料检测位标志
850.14 BOOL  ; 0标志
850.15 BOOL  ; 0标志
851.00 BOOL  ; 进料伺服Z轴JOG+标志
851.01 BOOL  ; 进料伺服Z轴JOG-标志
851.02 BOOL  ; 进料伺服Z轴回原点标志
851.03 BOOL  ; 进料伺服Z轴待机位标志
851.04 BOOL  ; 进料伺服Z轴取料位标志
851.05 BOOL  ; 进料伺服Z轴#1腔放料位标志
851.06 BOOL  ; 进料伺服Z轴#2腔放料位标志
851.07 BOOL  ; 进料伺服Z轴#3腔放料位标志
851.08 BOOL  ; 进料伺服Z轴#1夹爪扫码NG放料位标志
851.09 BOOL  ; 进料伺服Z轴#2夹爪扫码NG放料位标志
851.10 BOOL  ; 进料伺服Z轴#1夹爪配对取放料位标志
851.11 BOOL  ; 进料伺服Z轴#2夹爪配对取放料位标志
851.12 BOOL  ; 0标志
851.13 BOOL  ; 0标志
851.14 BOOL  ; 0标志
851.15 BOOL  ; 0标志
852.00 BOOL  ; 出料伺服X轴JOG+标志
852.01 BOOL  ; 出料伺服X轴JOG-标志
852.02 BOOL  ; 出料伺服X轴回原点标志
852.03 BOOL  ; 出料伺服X轴放料位标志
852.04 BOOL  ; 出料伺服X轴#1腔取料位标志
852.05 BOOL  ; 出料伺服X轴#2腔取料位标志
852.06 BOOL  ; 出料伺服X轴#3腔取料位标志
852.07 BOOL  ; 出料伺服X轴#1夹爪氦检NG放料位标志
852.08 BOOL  ; 出料伺服X轴#2夹爪氦检NG放料位标志
852.09 BOOL  ; 出料伺服X轴#1夹爪配对取放料位标志
852.10 BOOL  ; 出料伺服X轴#2夹爪配对取放料位标志
852.11 BOOL  ; 0标志
852.12 BOOL  ; 0标志
852.13 BOOL  ; 0标志
852.14 BOOL  ; 0标志
852.15 BOOL  ; 0标志
853.00 BOOL  ; 出料伺服Z轴JOG+标志
853.01 BOOL  ; 出料伺服Z轴JOG-标志
853.02 BOOL  ; 出料伺服Z轴回原点标志
853.03 BOOL  ; 出料伺服Z轴待机位标志
853.04 BOOL  ; 出料伺服Z轴放料位标志
853.05 BOOL  ; 出料伺服Z轴#1腔取料位标志
853.06 BOOL  ; 出料伺服Z轴#2腔取料位标志
853.07 BOOL  ; 出料伺服Z轴#3腔取料位标志
853.08 BOOL  ; 出料伺服Z轴#1夹爪氦检NG放料位标志
853.09 BOOL  ; 出料伺服Z轴#2夹爪氦检NG放料位标志
853.10 BOOL  ; 出料伺服Z轴#1夹爪配对取放料位标志
853.11 BOOL  ; 出料伺服Z轴#2夹爪配对取放料位标志
900.00 BOOL  ; #1扫码阻挡气缸缩回位[lamp]
900.01 BOOL  ; #1扫码阻挡气缸伸出位[lamp]
900.02 BOOL  ; #1隔离气缸缩回位[lamp]
900.03 BOOL  ; 0[lamp]
900.04 BOOL  ; #2扫码阻挡气缸缩回位[lamp]
900.05 BOOL  ; #2扫码阻挡气缸伸出位[lamp]
900.06 BOOL  ; #2隔离气缸缩回位[lamp]
900.07 BOOL  ; 0[lamp]
900.08 BOOL  ; #1进料夹爪夹紧位[lamp]
900.09 BOOL  ; #1进料夹爪松开位[lamp]
900.10 BOOL  ; #2进料夹爪夹紧位[lamp]
900.11 BOOL  ; #2进料夹爪松开位[lamp]
900.12 BOOL  ; 进料夹爪变距气缸伸出位[lamp]
900.13 BOOL  ; 进料夹爪变距气缸缩回位[lamp]
900.14 BOOL  ; #1出料夹爪夹紧位[lamp]
900.15 BOOL  ; #1出料夹爪松开位[lamp]
901.00 BOOL  ; #2出料夹爪夹紧位[lamp]
901.01 BOOL  ; #2出料夹爪松开位[lamp]
901.02 BOOL  ; 出料夹爪变距气缸伸出位[lamp]
901.03 BOOL  ; 出料夹爪变距气缸缩回位[lamp]
901.04 BOOL  ; #1腔体平移一级气缸缩回位[lamp]
901.05 BOOL  ; #1腔体平移一级气缸伸出位[lamp]
901.06 BOOL  ; #1腔体平移二级气缸缩回位[lamp]
901.07 BOOL  ; #1腔体平移二级气缸伸出位[lamp]
901.08 BOOL  ; #1腔体顶伸气缸上升位[lamp]
901.09 BOOL  ; #1腔体顶伸气缸下降位[lamp]
901.10 BOOL  ; #1腔体氦检阀开到位[lamp]
901.11 BOOL  ; #1腔体氦检阀关到位[lamp]
901.12 BOOL  ; 0[lamp]
901.13 BOOL  ; 0[lamp]
901.14 BOOL  ; 0[lamp]
901.15 BOOL  ; 0[lamp]
902.00 BOOL  ; 0[lamp]
902.01 BOOL  ; #2腔体平移一级气缸缩回位[lamp]
902.02 BOOL  ; #2腔体平移一级气缸伸出位[lamp]
902.03 BOOL  ; #2腔体平移二级气缸缩回位[lamp]
902.04 BOOL  ; #2腔体平移二级气缸伸出位[lamp]
902.05 BOOL  ; #2腔体顶伸气缸上升位[lamp]
902.06 BOOL  ; #2腔体顶伸气缸下降位[lamp]
902.07 BOOL  ; #2腔体氦检阀开到位[lamp]
902.08 BOOL  ; #2腔体氦检阀关到位[lamp]
902.09 BOOL  ; 0[lamp]
902.10 BOOL  ; 0[lamp]
902.11 BOOL  ; 0[lamp]
902.12 BOOL  ; 0[lamp]
902.13 BOOL  ; 0[lamp]
902.14 BOOL  ; #3腔体平移一级气缸缩回位[lamp]
902.15 BOOL  ; #3腔体平移一级气缸伸出位[lamp]
903.00 BOOL  ; #3腔体平移二级气缸缩回位[lamp]
903.01 BOOL  ; #3腔体平移二级气缸伸出位[lamp]
903.02 BOOL  ; #3腔体顶伸气缸上升位[lamp]
903.03 BOOL  ; #3腔体顶伸气缸下降位[lamp]
903.04 BOOL  ; #3腔体氦检阀开到位[lamp]
903.05 BOOL  ; #3腔体氦检阀关到位[lamp]
903.06 BOOL  ; 氦检仪准备好了信号[lamp]
903.07 BOOL  ; 氦检仪故障信号[lamp]
903.08 BOOL  ; 0[lamp]
903.09 BOOL  ; 0[lamp]
903.10 BOOL  ; 0[lamp]
903.11 BOOL  ; 进料伺服X轴准备好了信号[lamp]
903.12 BOOL  ; 进料伺服X轴故障信号[lamp]
903.13 BOOL  ; 进料伺服Z轴准备好了信号[lamp]
903.14 BOOL  ; 进料伺服Z轴故障信号[lamp]
903.15 BOOL  ; 进料伺服Z轴刹车[lamp]
904.00 BOOL  ; 出料伺服X轴准备好了信号[lamp]
904.01 BOOL  ; 出料伺服X轴故障信号[lamp]
904.02 BOOL  ; 出料伺服Z轴准备好了信号[lamp]
904.03 BOOL  ; 出料伺服Z轴故障信号[lamp]
904.04 BOOL  ; 0[lamp]
904.05 BOOL  ; 腔体抽真空泵运行信号[lamp]
904.06 BOOL  ; 腔体抽真空泵过载信号[lamp]
904.07 BOOL  ; 氦检前置泵运行信号[lamp]
904.08 BOOL  ; 氦检前置泵过载信号[lamp]
904.09 BOOL  ; 启动按钮[lamp]
904.10 BOOL  ; 停止按钮[lamp]
904.11 BOOL  ; 复位按钮[lamp]
904.12 BOOL  ; 急停按钮[lamp]
904.13 BOOL  ; 手自动选择[lamp]
904.14 BOOL  ; #1进料夹爪防下坠感应[lamp]
904.15 BOOL  ; #2进料夹爪防下坠感应[lamp]
905.00 BOOL  ; #1出料夹爪防下坠感应[lamp]
905.01 BOOL  ; #2出料夹爪防下坠感应[lamp]
905.02 BOOL  ; 0[lamp]
905.03 BOOL  ; 进料对接输入[lamp]
905.04 BOOL  ; 出料对接输入[lamp]
905.05 BOOL  ; 出料旋转气缸9O度位条件
905.06 BOOL  ; 出料旋转气缸O度位条件
905.07 BOOL  ; 设备总气压信号[lamp]
905.08 BOOL  ; #1来料位有料感应[lamp]
905.09 BOOL  ; #2来料位有料感应[lamp]
905.10 BOOL  ; #1隔离位有料感应[lamp]
905.11 BOOL  ; #2隔离位有料感应[lamp]
905.12 BOOL  ; #1扫码位有料感应[lamp]
905.13 BOOL  ; #2扫码位有料感应[lamp]
905.14 BOOL  ; #1-1进料位有料感应[lamp]
905.15 BOOL  ; #1-2进料位有料感应[lamp]
906.00 BOOL  ; #2-1进料位有料感应[lamp]
906.01 BOOL  ; #2-2进料位有料感应[lamp]
906.02 BOOL  ; 进料夹爪柔性感应[lamp]
906.03 BOOL  ; 出料夹爪柔性感应[lamp]
906.04 BOOL  ; #1进料夹爪对应腔体有料感应[lamp]
906.05 BOOL  ; #2进料夹爪对应腔体有料感应[lamp]
906.06 BOOL  ; 扫码NG放料#1位有料感应[lamp]
906.07 BOOL  ; 扫码NG放料#2位有料感应[lamp]
906.08 BOOL  ; 扫码NG料满位有料感应[lamp]
906.09 BOOL  ; 进料配对位有料感应[lamp]
906.10 BOOL  ; 出料配对位有料感应[lamp]
906.11 BOOL  ; 氦检NG放料#1位有料感应[lamp]
906.12 BOOL  ; 氦检NG放料#2位有料感应[lamp]
906.13 BOOL  ; 氦检NG料满位有料感应[lamp]
906.14 BOOL  ; #1-1出料位有料感应[lamp]
906.15 BOOL  ; #1-2出料位有料感应[lamp]
907.00 BOOL  ; #2-1出料位有料感应[lamp]
907.01 BOOL  ; #2-2出料位有料感应[lamp]
907.02 BOOL  ; #1门磁开关[lamp]
907.03 BOOL  ; #2门磁开关[lamp]
907.04 BOOL  ; #3门磁开关[lamp]
907.05 BOOL  ; #4门磁开关[lamp]
907.06 BOOL  ; #5门磁开关[lamp]
907.07 BOOL  ; #6门磁开关[lamp]
907.08 BOOL  ; #7门磁开关[lamp]
907.09 BOOL  ; #8门磁开关[lamp]
907.10 BOOL  ; #9门磁开关[lamp]
907.11 BOOL  ; #10门磁开关[lamp]
907.12 BOOL  ; #11门磁开关[lamp]
907.13 BOOL  ; 设备真空压力信号[lamp]
907.14 BOOL  ; 设备氦气压力信号[lamp]
907.15 BOOL  ; 精密调压阀信号[lamp]
910.03 BOOL  ; $?St$Bk?_#[12] / #1隔离气缸伸出位[lamp] / $?St$Bk?_#[12]
910.07 BOOL  ; $?St$Bk?_#[13] / #2隔离气缸伸出位[lamp] / $?St$Bk?_#[13]
920.14 BOOL  ; #1腔体抽真空阀开到位[lamp]
920.15 BOOL  ; #1腔体抽真空阀关到位[lamp]
921.00 BOOL  ; #1-1腔体阀开到位[lamp]
921.01 BOOL  ; #1-1腔体阀关到位[lamp]
921.02 BOOL  ; #1-2腔体阀开到位[lamp]
921.03 BOOL  ; #1-2腔体阀关到位[lamp]
921.04 BOOL  ; #1腔体破真空阀开到位[lamp]
921.05 BOOL  ; #1腔体破真空阀关到位[lamp]
921.06 BOOL  ; #1腔体吹气阀开到位[lamp]
921.07 BOOL  ; #1腔体吹气阀关到位[lamp]
921.08 BOOL  ; #2腔体抽真空阀开到位[lamp]
921.09 BOOL  ; #2腔体抽真空阀关到位[lamp]
921.10 BOOL  ; #2-1腔体阀开到位[lamp]
921.11 BOOL  ; #2-1腔体阀关到位[lamp]
921.12 BOOL  ; #2-2腔体阀开到位[lamp]
921.13 BOOL  ; #2-2腔体阀关到位[lamp]
921.14 BOOL  ; #2腔体破真空阀开到位[lamp]
921.15 BOOL  ; #2腔体破真空阀关到位[lamp]
922.00 BOOL  ; #2腔体吹气阀开到位[lamp]
922.01 BOOL  ; #2腔体吹气阀关到位[lamp]
922.02 BOOL  ; #3腔体抽真空阀开到位[lamp]
922.03 BOOL  ; #3腔体抽真空阀关到位[lamp]
922.04 BOOL  ; #3-1腔体阀开到位[lamp]
922.05 BOOL  ; #3-1腔体阀关到位[lamp]
922.06 BOOL  ; #3-2腔体阀开到位[lamp]
922.07 BOOL  ; #3-2腔体阀关到位[lamp]
922.08 BOOL  ; #3腔体破真空阀开到位[lamp]
922.09 BOOL  ; #3腔体破真空阀关到位[lamp]
922.10 BOOL  ; #3腔体吹气阀开到位[lamp]
922.11 BOOL  ; #3腔体吹气阀关到位[lamp]
922.12 BOOL  ; #1-1电池抽真空阀开到位[lamp]
922.13 BOOL  ; #1-1电池抽真空阀关到位[lamp]
922.14 BOOL  ; #1-2电池抽真空阀开到位[lamp]
922.15 BOOL  ; #1-2电池抽真空阀关到位[lamp]
923.00 BOOL  ; #1-1电池注氦阀开到位[lamp]
923.01 BOOL  ; #1-1电池注氦阀关到位[lamp]
923.02 BOOL  ; #1-2电池注氦阀开到位[lamp]
923.03 BOOL  ; #1-2电池注氦阀关到位[lamp]
923.04 BOOL  ; #1-1电池破真空阀开到位[lamp]
923.05 BOOL  ; #1-1电池破真空阀关到位[lamp]
923.06 BOOL  ; #1-2电池破真空阀开到位[lamp]
923.07 BOOL  ; #1-2电池破真空阀关到位[lamp]
923.08 BOOL  ; #2-1电池抽真空阀开到位[lamp]
923.09 BOOL  ; #2-1电池抽真空阀关到位[lamp]
923.10 BOOL  ; #2-2电池抽真空阀开到位[lamp]
923.11 BOOL  ; #2-2电池抽真空阀关到位[lamp]
923.12 BOOL  ; #2-1电池注氦阀开到位[lamp]
923.13 BOOL  ; #2-1电池注氦阀关到位[lamp]
923.14 BOOL  ; #2-2电池注氦阀开到位[lamp]
923.15 BOOL  ; #2-2电池注氦阀关到位[lamp]
924.00 BOOL  ; #2-1电池破真空阀开到位[lamp]
924.01 BOOL  ; #2-1电池破真空阀关到位[lamp]
924.02 BOOL  ; #2-2电池破真空阀开到位[lamp]
924.03 BOOL  ; #2-2电池破真空阀关到位[lamp]
924.04 BOOL  ; #3-1电池抽真空阀开到位[lamp]
924.05 BOOL  ; #3-1电池抽真空阀关到位[lamp]
924.06 BOOL  ; #3-2电池抽真空阀开到位[lamp]
924.07 BOOL  ; #3-2电池抽真空阀关到位[lamp]
924.08 BOOL  ; #3-1电池注氦阀开到位[lamp]
924.09 BOOL  ; #3-1电池注氦阀关到位[lamp]
924.10 BOOL  ; #3-2电池注氦阀开到位[lamp]
924.11 BOOL  ; #3-2电池注氦阀关到位[lamp]
924.12 BOOL  ; #3-1电池破真空阀开到位[lamp]
924.13 BOOL  ; #3-1电池破真空阀关到位[lamp]
924.14 BOOL  ; #3-2电池破真空阀开到位[lamp]
924.15 BOOL  ; #3-2电池破真空阀关到位[lamp]
950.00 BOOL  ; 进料伺服X轴JOG+[lamp]
950.01 BOOL  ; 进料伺服X轴JOG-[lamp]
950.02 BOOL  ; 进料伺服X轴回原点[lamp]
950.03 BOOL  ; 进料伺服X轴取料位[lamp]
950.04 BOOL  ; 进料伺服X轴#1腔放料位[lamp]
950.05 BOOL  ; 进料伺服X轴#2腔放料位[lamp]
950.06 BOOL  ; 进料伺服X轴#3腔放料位[lamp]
950.07 BOOL  ; 进料伺服X轴#1夹爪扫码NG放料位[lamp]
950.08 BOOL  ; 进料伺服X轴#2夹爪扫码NG放料位[lamp]
950.09 BOOL  ; 进料伺服X轴#1夹爪配对取放料位[lamp]
950.10 BOOL  ; 进料伺服X轴#2夹爪配对取放料位[lamp]
950.11 BOOL  ; 进料伺服X轴#1腔有料检测位[lamp]
950.12 BOOL  ; 进料伺服X轴#2腔有料检测位[lamp]
950.13 BOOL  ; 进料伺服X轴#3腔有料检测位[lamp]
950.14 BOOL  ; 0[lamp]
950.15 BOOL  ; 0[lamp]
951.00 BOOL  ; 进料伺服Z轴JOG+[lamp]
951.01 BOOL  ; 进料伺服Z轴JOG-[lamp]
951.02 BOOL  ; 进料伺服Z轴回原点[lamp]
951.03 BOOL  ; 进料伺服Z轴待机位[lamp]
951.04 BOOL  ; 进料伺服Z轴取料位[lamp]
951.05 BOOL  ; 进料伺服Z轴#1腔放料位[lamp]
951.06 BOOL  ; 进料伺服Z轴#2腔放料位[lamp]
951.07 BOOL  ; 进料伺服Z轴#3腔放料位[lamp]
951.08 BOOL  ; 进料伺服Z轴#1夹爪扫码NG放料位[lamp]
951.09 BOOL  ; 进料伺服Z轴#2夹爪扫码NG放料位[lamp]
951.10 BOOL  ; 进料伺服Z轴#1夹爪配对取放料位[lamp]
951.11 BOOL  ; 进料伺服Z轴#2夹爪配对取放料位[lamp]
951.12 BOOL  ; 0[lamp]
951.13 BOOL  ; 0[lamp]
951.14 BOOL  ; 0[lamp]
951.15 BOOL  ; 0[lamp]
952.00 BOOL  ; 出料伺服X轴JOG+[lamp]
952.01 BOOL  ; 出料伺服X轴JOG-[lamp]
952.02 BOOL  ; 出料伺服X轴回原点[lamp]
952.03 BOOL  ; 出料伺服X轴放料位[lamp]
952.04 BOOL  ; 出料伺服X轴#1腔取料位[lamp]
952.05 BOOL  ; 出料伺服X轴#2腔取料位[lamp]
952.06 BOOL  ; 出料伺服X轴#3腔取料位[lamp]
952.07 BOOL  ; 出料伺服X轴#1夹爪氦检NG放料位[lamp]
952.08 BOOL  ; 出料伺服X轴#2夹爪氦检NG放料位[lamp]
952.09 BOOL  ; 出料伺服X轴#1夹爪配对取放料位[lamp]
952.10 BOOL  ; 出料伺服X轴#2夹爪配对取放料位[lamp]
952.11 BOOL  ; 0[lamp]
952.12 BOOL  ; 0[lamp]
952.13 BOOL  ; 0[lamp]
952.14 BOOL  ; 0[lamp]
952.15 BOOL  ; 0[lamp]
953.00 BOOL  ; 出料伺服Z轴JOG+[lamp]
953.01 BOOL  ; 出料伺服Z轴JOG-[lamp]
953.02 BOOL  ; 出料伺服Z轴回原点[lamp]
953.03 BOOL  ; 出料伺服Z轴待机位[lamp]
953.04 BOOL  ; 出料伺服Z轴放料位[lamp]
953.05 BOOL  ; 出料伺服Z轴#1腔取料位[lamp]
953.06 BOOL  ; 出料伺服Z轴#2腔取料位[lamp]
953.07 BOOL  ; 出料伺服Z轴#3腔取料位[lamp]
953.08 BOOL  ; 出料伺服Z轴#1夹爪氦检NG放料位[lamp]
953.09 BOOL  ; 出料伺服Z轴#2夹爪氦检NG放料位[lamp]
953.10 BOOL  ; 出料伺服Z轴#1夹爪配对取放料位[lamp]
953.11 BOOL  ; 出料伺服Z轴#2夹爪配对取放料位[lamp]
A201.01 BOOL  ; SCU21_2 Port#2 端口1允许标志
A202.01 BOOL  ; SCU21_2 Port#2 端口1允许标志
A202.05 BOOL  ; SCU21_2 Port#1 端口5允许标志
A276 CHANNEL  ; 脉冲输出0当前值
A278 CHANNEL  ; 脉冲输出1当前值
A280.04 BOOL  ; 进料伺服X轴脉冲输出中标志(0：停止中,1：输出中)
A280.05 BOOL  ; 进料伺服X轴无原点标志(0：原点确定,1：原点未确定)
A280.07 BOOL  ; 脉冲输出0输出停止异常标志
A281.04 BOOL  ; 进料伺服Z轴脉冲输出中标志(0：停止中,1：输出中)
A281.05 BOOL  ; 进料伺服Z轴无原点标志(0：原点确定,1：原点未确定)
A281.07 BOOL  ; 脉冲输出1输出停止异常标志
A326.04 BOOL  ; 出料伺服X轴脉冲输出中标志(0：停止中,1：输出中)
A326.05 BOOL  ; 出料伺服X轴无原点标志(0：原点确定,1：原点未确定)
A327.04 BOOL  ; 出料伺服Z轴脉冲输出中标志(0：停止中,1：输出中)
A327.05 BOOL  ; 出料伺服Z轴无原点标志(0：原点确定,1：原点未确定)
A392.04 BOOL  ; 内置RS232串行端口错误标志
A392.05 BOOL  ; 内置串行端口发送就绪
A392.06 BOOL  ; 内置串口接收就绪
A392.07 BOOL  ; 串行端口 1接收超限标志
A393 CHANNEL  ; 内置串口接收数据长度
A526.00 BOOL  ; 内置RS232串行端口重启标志
A540.08 BOOL  ; 脉冲输出0 CW限位输入信号标志
A540.09 BOOL  ; 脉冲输出0 CCW限位输入信号标志
A541.08 BOOL  ; 脉冲输出1 CW限位输入信号标志
A541.09 BOOL  ; 脉冲输出1 CCW限位输入信号标志
A542.08 BOOL  ; 出料X轴定位轴CW
A542.09 BOOL  ; 出料X轴定位轴CCW
A543.08 BOOL  ; 出料Z轴定位轴CW
A543.09 BOOL  ; 出料Z轴定位轴CCW
A622.01 BOOL  ; #2unit#1port restar
A622.02 BOOL  ; #2unit#2port restar
C0050 BOOL  ; 进料拉带机构扫码NG后重复次数计数
D1 CHANNEL  ; #1腔体读取设定时间
D10 CHANNEL  ; PLC&PC数据交互超时报警延时设定
D100 CHANNEL  ; 腔体测试设定真空阈值（Pa_Float）
D1000.00 BOOL  ; 进料拉带机构扫码初始位
D1000.05 BOOL  ; 进料扫码停止标志
D1000.06 BOOL  ; 进料扫码清料完成标志
D1000.07 BOOL  ; 进料拉带机构异常标志
D1001.00 BOOL  ; 进料拉带机构扫码运行条件
D1001.01 BOOL  ; 进料拉带隔离气缸允许放料条件
D1001.02 BOOL  ; 进料拉带扫码阻挡气缸允许放料条件
D1003.00 BOOL  ; 进料拉带机构单步/自动循环运行中（总）
D1003.10 BOOL  ; 进料拉带工站记忆显示（Lamp）
D1003.11 BOOL  ; 进料拉带工站初始化显示（Lamp）
D1003.13 BOOL  ; 进料拉带机构记忆清除（SW）
D1003.14 BOOL  ; 进料拉带机构复位按钮（SW）
D1003.15 BOOL  ; 进料拉带机构单步（SW）
D1004.00 BOOL  ; 进料拉带机构单步运行中
D1004.01 BOOL  ; 进料拉带机构单步/自动循环运行中
D1004.10 BOOL  ; 进料拉带机构单步运行条件
D1005.00 BOOL  ; 进料拉带机构开始运行条件
D1005.01 BOOL  ; 进料拉带机构步进条件
D1005.15 BOOL  ; 进料拉带机构步进
D1006 CHANNEL  ; 进料拉带机构步序
D1006.00 BOOL  ; 进料拉带机构自动开始（步）
D1006.01 BOOL  ; 进料拉带机构扫码数据初始化（步）
D1006.02 BOOL  ; 预留
D1006.03 BOOL  ; 进料拉带机构扫码触发前延时（步）
D1006.04 BOOL  ; 进料拉带机构扫码触发（步）
D1006.05 BOOL  ; 进料拉带机构扫码结果（步）
D1006.06 BOOL  ; 进料拉带机构扫码MES入站校验结果（步）
D1006.07 BOOL  ; 预留
D1006.08 BOOL  ; 进料拉带机构扫码阻挡气缸缩回&进料拉带电机启动（步）
D1006.09 BOOL  ; 进料拉带机构扫码阻挡气缸伸出（步）
D1006.10 BOOL  ; 预留
D1006.11 BOOL  ; 进料拉带机构循环完成
D1017.00 BOOL  ; 进料拉带机构复位（M）
D1017.01 BOOL  ; #1隔离气缸伸出（复位）
D1017.02 BOOL  ; #2隔离气缸伸出（复位）
D1017.03 BOOL  ; #1扫码阻挡气缸伸出（复位）
D1017.04 BOOL  ; #2扫码阻挡气缸伸出（复位）
D1017.05 BOOL  ; #1隔离气缸缩回（复位）
D1017.06 BOOL  ; #2隔离气缸缩回（复位）
D1017.07 BOOL  ; #1扫码阻挡气缸缩回（复位）
D1017.08 BOOL  ; #2扫码阻挡气缸缩回（复位）
D1019 CHANNEL  ; 进料拉带机构扫码步序号
D102 CHANNEL  ; 腔体测试设定抽真空时间上限（S_UInt）
D1023.13 BOOL  ; NG缓存机构记忆清除（SW）
D104 CHANNEL  ; 腔体测试设定清氦压力（Pa_Float）
D1040.00 BOOL  ; 进料伺服机构初始位
D1040.05 BOOL  ; 进料伺服机构停止标志
D1040.06 BOOL  ; 进料伺服机构清料完成标志
D1040.07 BOOL  ; 进料伺服机构异常标志
D1041.00 BOOL  ; 进料伺服机构运行条件（公共）
D1041.01 BOOL  ; 进料伺服机构运行条件1（进料拉带取料）
D1041.02 BOOL  ; 进料伺服机构运行条件2（扫码NG放料）
D1041.03 BOOL  ; 进料伺服机构运行条件3（扫码配对取/放料）
D1041.04 BOOL  ; 进料伺服机构运行条件4（腔体放料）
D1043.00 BOOL  ; 进料伺服机构单步/自动循环运行中（总）
D1043.10 BOOL  ; 进料伺服工站记忆显示（Lamp）
D1043.11 BOOL  ; 进料伺服工站初始化显示（Lamp）
D1043.13 BOOL  ; 进料伺服机构记忆清除（SW）
D1043.14 BOOL  ; 进料伺服机构复位按钮（SW）
D1043.15 BOOL  ; 进料伺服机构单步（SW）
D1044.00 BOOL  ; 进料伺服机构单步运行中1（进料拉带取料）
D1044.01 BOOL  ; 进料伺服机构单步/自动循环运行中1（进料拉带取料）
D1044.02 BOOL  ; 进料伺服机构单步运行中2（扫码NG放料）
D1044.03 BOOL  ; 进料伺服机构单步/自动循环运行中2（扫码NG放料）
D1044.04 BOOL  ; 进料伺服机构单步运行中3（扫码配对取/放料）
D1044.05 BOOL  ; 进料伺服机构单步/自动循环运行中3（扫码配对取/放料）
D1044.06 BOOL  ; 进料伺服机构单步运行中4（腔体放料）
D1044.07 BOOL  ; 进料伺服机构单步/自动循环运行中4（腔体放料）
D1044.10 BOOL  ; 进料伺服机构单步运行条件1（进料拉带取料）
D1044.11 BOOL  ; 进料伺服机构单步运行条件2（扫码NG放料）
D1044.12 BOOL  ; 进料伺服机构单步运行条件3（扫码配对取/放料）
D1044.13 BOOL  ; 进料伺服机构单步运行条件4（腔体放料）
D1045.00 BOOL  ; 进料伺服机构开始运行条件1（进料拉带取料）
D1045.01 BOOL  ; 进料伺服机构步进条件1（进料拉带取料）
D1045.15 BOOL  ; 进料伺服机构步进1（进料拉带取料）
D1046 CHANNEL  ; 进料伺服机构步序1（进料拉带取料）
D1046.00 BOOL  ; 进料伺服机构自动开始1（步）
D1046.01 BOOL  ; 进料伺服机构X轴取料位&变距气缸缩回1（步）
D1046.02 BOOL  ; 进料伺服机构Z轴取料位1（步）
D1046.03 BOOL  ; 进料伺服机构夹爪夹紧1（步）
D1046.04 BOOL  ; 进料伺服机构Z轴待料位1（步）
D1046.05 BOOL  ; 预留
D1046.06 BOOL  ; 进料伺服机构循环完成1（步）
D1048.00 BOOL  ; 进料伺服机构开始运行条件2（扫码NG放料）
D1048.01 BOOL  ; 进料伺服机构步进条件2（扫码NG放料）
D1048.15 BOOL  ; 进料伺服机构步进2（扫码NG放料）
D1049 CHANNEL  ; 进料伺服机构步序2（扫码NG放料）
D1049.00 BOOL  ; 进料伺服机构自动开始2（步）
D1049.01 BOOL  ; 进料伺服机构X轴#1|2夹爪扫码NG放料位&变距气缸伸出2（步）
D1049.02 BOOL  ; 进料伺服机构Z轴#1|2夹爪扫码NG放料位2（步）
D1049.03 BOOL  ; 进料伺服机构#1|2夹爪松开2（步）
D1049.04 BOOL  ; 进料伺服机构Z轴待料位2（步）
D1049.05 BOOL  ; 预留
D1049.06 BOOL  ; 预留
D1049.07 BOOL  ; 预留
D1049.08 BOOL  ; 预留
D1049.09 BOOL  ; 进料伺服机构X轴取料位&变距气缸缩回2（步）
D1049.10 BOOL  ; 进料伺服机构循环完成2（步）
D1051.00 BOOL  ; 进料伺服机构开始运行条件3（扫码配对取/放料）
D1051.01 BOOL  ; 进料伺服机构步进条件3（扫码配对取/放料）
D1051.15 BOOL  ; 进料伺服机构步进3（扫码配对取/放料）
D1052 CHANNEL  ; 进料伺服机构步序3（扫码配对取/放料）
D1052.00 BOOL  ; 进料伺服机构自动开始3（步）
D1052.01 BOOL  ; 进料伺服机构X轴#1|2夹爪配对取放料位&变距气缸缩回3（步）
D1052.02 BOOL  ; 进料伺服机构Z轴#1|2夹爪配对取放料位3（步）
D1052.03 BOOL  ; 进料伺服机构#1|2夹爪松开|夹紧3（步）
D1052.04 BOOL  ; 进料伺服机构Z轴待料位3（步）
D1052.05 BOOL  ; 预留
D1052.06 BOOL  ; 进料伺服机构X轴取料位&变距气缸缩回3（步）
D1052.07 BOOL  ; 进料伺服机构循环完成3（步）
D1054.00 BOOL  ; 进料伺服机构开始运行条件4（腔体放料）
D1054.01 BOOL  ; 进料伺服机构步进条件4（腔体放料）
D1054.15 BOOL  ; 进料伺服机构步进4（腔体放料）
D1055 CHANNEL  ; 进料伺服机构步序4（腔体放料）
D1055.00 BOOL  ; 进料伺服机构自动开始4（步）
D1055.01 BOOL  ; 进料伺服机构X轴#1|2|3腔放料位&变距气缸伸出4（步）
D1055.02 BOOL  ; 预留
D1055.03 BOOL  ; 进料伺服机构Z轴#1|2|3腔放料位4（步）
D1055.04 BOOL  ; 进料伺服机构#1&2夹爪松开4（步）
D1055.05 BOOL  ; 进料伺服机构Z轴待料位4（步）
D1055.05 BOOL  ; 预留
D1055.06 BOOL  ; 进料伺服机构X轴取料位&变距气缸缩回4（步）
D1055.07 BOOL  ; 进料伺服机构循环完成4（步）
D1057.00 BOOL  ; 进料伺服工站复位（M）
D1057.01 BOOL  ; #1进料夹爪松开（复位）
D1057.02 BOOL  ; #2进料夹爪松开（复位）
D1057.03 BOOL  ; 进料夹爪变距气缸缩回（复位）
D1057.04 BOOL  ; #1进料夹爪夹紧（复位）
D1057.05 BOOL  ; #2进料夹爪夹紧（复位）
D1057.06 BOOL  ; 进料伺服Z轴回原点（复位）
D1057.07 BOOL  ; 进料伺服Z轴待机位（复位）
D1057.08 BOOL  ; 进料伺服X轴回原点（复位）
D1057.09 BOOL  ; 进料伺服X轴取料位（复位）
D1059 CHANNEL  ; 进料伺服机构步序号
D106 CHANNEL  ; 腔体测试设定氦检安全阈值（Pa_Float）
D1060.00 BOOL  ; #1氦检机构初始位
D1060.05 BOOL  ; #1氦检机构停止标志
D1060.06 BOOL  ; #1氦检机构清料完成标志
D1060.07 BOOL  ; #1氦检机构异常标志
D1061.00 BOOL  ; #1腔体机构运行条件（自动步）
D1061.01 BOOL  ; #1腔体机构运行条件（自动单检步）
D1061.02 BOOL  ; #1腔体机构运行条件（清氦步）
D1062.00 BOOL  ; #1腔体机构平移气缸安全移动条件
D1062.12 BOOL  ; #1腔体机构腔体抽真空需求（测试）
D1062.13 BOOL  ; #1腔体机构正常清氦需求（正压测试）
D1062.14 BOOL  ; #1腔体氦检阀打开允许条件
D1062.15 BOOL  ; #1腔体机构腔体抽气阀打开允许
D1063.00 BOOL  ; #1腔体机构单步/自动循环运行中（总）
D1063.10 BOOL  ; $?St$Bk?_#[14] / #1腔体机构记忆清除(SW) / $?St$Bk?_#[14]
D1063.11 BOOL  ; #1腔体标漏(SW)
D1063.12 BOOL  ; #1腔体自检启动(SW)
D1063.13 BOOL  ; #1腔体自检停止(SW)
D1063.14 BOOL  ; #1腔体机构复位按钮（SW）
D1063.15 BOOL  ; #1腔体机构单步（SW）
D1064.00 BOOL  ; #1腔体机构单步运行中
D1064.01 BOOL  ; #1腔体机构单步/自动循环运行中（自动步）
D1064.02 BOOL  ; #1腔体机构自动循环运行中（自动单检步）
D1064.03 BOOL  ; #1腔体机构自动循环运行中（清氦步）
D1064.04 BOOL  ; #1-1腔体单腔自检（SW）
D1064.05 BOOL  ; #1-2腔体单腔自检(SW)
D1064.06 BOOL  ; #1腔体自检运行中
D1065.00 BOOL  ; #1腔体机构开始运行条件（自动步）
D1065.01 BOOL  ; #1腔体机构步进条件（自动步）
D1065.02 BOOL  ; #1腔体机构开始运行条件（自动单检步）
D1065.03 BOOL  ; #1腔体机构步进条件（自动单检步）
D1065.04 BOOL  ; #1腔体机构开始运行条件（清氦步）
D1065.05 BOOL  ; #1腔体机构步进条件（清氦步）
D1065.13 BOOL  ; #1腔体机构步进（清氦步）
D1065.14 BOOL  ; #1腔体机构步进（自动单检步）
D1065.15 BOOL  ; #1腔体机构步进（自动步）
D1066 CHANNEL  ; #1腔体机构自动步序号
D1066.00 BOOL  ; #1腔体机构自动开始（自动步）
D1066.01 BOOL  ; #1腔体机构平移气缸到氦检位/数据初始化（自动步）
D1066.02 BOOL  ; #1腔体机构腔体顶升气缸上升（自动步）
D1066.03 BOOL  ; #1腔体机构等待氦检阀打开条件及腔体抽气阀打开条件/开腔体阀（自动步）
D1066.04 BOOL  ; #1腔体机构（自动步）
D1066.05 BOOL  ; #1腔体机构腔体抽气阀打开/延时开电池抽气阀（自动步）
D1066.06 BOOL  ; #1腔体机构关电池抽气阀（自动步）
D1066.07 BOOL  ; #1腔体机构开电池注氦阀（自动步）
D1066.08 BOOL  ; #1腔体机构关电池注氦阀（自动步）
D1066.09 BOOL  ; #1腔体机构（自动步）
D1066.10 BOOL  ; #1腔体机构开腔体氦检阀/延时关腔体抽气阀（自动步）
D1066.11 BOOL  ; #1腔体机构（自动步）
D1066.12 BOOL  ; #1腔体机构关腔体氦检阀（自动步）
D1066.13 BOOL  ; #1腔体机构（自动步）
D1066.14 BOOL  ; #1腔体机构开腔体#1-1腔体阀/开腔体#1-2腔体阀（自动步）
D1066.15 BOOL  ; #1腔体机构开腔体抽真空阀/开电池抽真空阀（自动步）
D1067.00 BOOL  ; #1腔体机构关腔体抽真空阀/关电池抽真空阀/开腔体阀（自动步）
D1067.01 BOOL  ; #1腔体机构清氦需求判定（自动步）
D1067.02 BOOL  ; #1腔体机构开腔体破真空阀/开电池破真空阀（自动步）
D1067.03 BOOL  ; #1腔体机构关腔体破真空阀/关电池破真空阀（自动步）
D1067.04 BOOL  ; #1腔体机构复测需求判定（自动步）
D1067.05 BOOL  ; #1腔体机构（自动步）
D1067.06 BOOL  ; #1腔体机构腔体顶升气缸下降（自动步）
D1067.07 BOOL  ; #1腔体机构（自动步）
D1067.08 BOOL  ; #1腔体机构腔体平移气缸到出料位（自动步）
D1067.09 BOOL  ; #1腔体机构腔体等待取料完成信号（自动步）
D1067.10 BOOL  ; #1腔体机构（自动步）
D1067.11 BOOL  ; #1腔体机构平移气缸到上料位（自动步）
D1067.12 BOOL  ; #1腔体机构（自动步）
D1067.13 BOOL  ; #1腔体机构（自动步）
D1067.14 BOOL  ; #1腔体机构（自动步）
D1067.15 BOOL  ; #1腔体机构循环结束（自动步）
D1070 CHANNEL  ; #1腔体机构单检步序号
D1070.00 BOOL  ; #1腔体机构自动开始（自动单检步）
D1070.01 BOOL  ; #1腔体机构平移气缸到氦检位/数据初始化（自动单检步）
D1070.02 BOOL  ; #1腔体机构腔体顶升气缸上升（自动单检步）
D1070.03 BOOL  ; #1腔体机构关闭#1-2腔体阀（自动单检步）
D1070.04 BOOL  ; #1腔体机构腔体抽气阀打开/延时开#1-1电池抽气阀（自动单检步）
D1070.05 BOOL  ; #1腔体机构关#1-1电池抽气阀（自动单检步）
D1070.06 BOOL  ; #1腔体机构开#1-1电池注氦阀（自动单检步）
D1070.07 BOOL  ; #1腔体机构关#1-1电池注氦阀（自动单检步）
D1070.08 BOOL  ; #1腔体机构（自动单检步）
D1070.09 BOOL  ; #1腔体机构开腔体氦检阀/延时关腔体抽气阀（自动单检步）
D1070.10 BOOL  ; #1腔体机构关腔体氦检阀/关腔体抽气阀/关#1-1电池抽气阀（自动单检步）
D1070.11 BOOL  ; #1腔体机构关闭#1-1腔体阀/清氦判定（自动单检步）
D1070.12 BOOL  ; #1腔体机构打开#1-2腔体阀（自动单检步）
D1070.13 BOOL  ; #1腔体机构腔体抽气阀打开/延时开#1-2电池抽气阀（自动单检步）
D1070.14 BOOL  ; #1腔体机构关#1-2电池抽气阀（自动单检步）
D1070.15 BOOL  ; #1腔体机构开#1-2电池注氦阀（自动单检步）
D1071.00 BOOL  ; #1腔体机构关#1-2电池注氦阀（自动单检步）
D1071.01 BOOL  ; #1腔体机构（自动单检步）
D1071.02 BOOL  ; #1腔体机构开腔体氦检阀/延时关腔体抽气阀（自动单检步）
D1071.03 BOOL  ; #1腔体机构关腔体氦检阀（自动单检步）
D1071.04 BOOL  ; #1腔体机构开腔体#1-1阀（自动单检步）
D1071.05 BOOL  ; #1腔体机构开腔体抽真空阀/开电池抽真空阀（自动单检步）
D1071.06 BOOL  ; #1腔体机构关腔体抽真空阀/关电池抽真空阀（自动单检步）
D1071.07 BOOL  ; #1腔体机构清氦需求判定（自动单检步）
D1071.08 BOOL  ; #1腔体机构开腔体破真空阀/开电池破真空阀（自动单检步）
D1071.09 BOOL  ; #1腔体机构关腔体破真空阀/关电池破真空阀（自动单检步）
D1071.10 BOOL  ; #1腔体机构腔体顶升气缸下降（自动单检步）
D1071.11 BOOL  ; #1腔体机构腔体平移气缸到出料位（自动单检步）
D1071.12 BOOL  ; $?St$Bk?_#[15] / #1腔体机构腔体等待取料完成信号（自动单检步） / $?St$Bk?_#[15]
D1071.13 BOOL  ; #1腔体机构腔体平移气缸到上料位（自动单检步）
D1071.14 BOOL  ; #1腔体机构（自动单检步）
D1071.15 BOOL  ; #1腔体机构循环结束（自动单检步）
D1074 CHANNEL  ; #1腔体机构清氦步序号
D1074.00 BOOL  ; #1腔体机构自动开始（清氦步）
D1074.01 BOOL  ; #1腔体机构平移气缸到氦检位/数据初始化（清氦步）
D1074.02 BOOL  ; #1腔体机构腔体顶升气缸上升（清氦步）
D1074.03 BOOL  ; #1腔体机构氦检仪真空阀关闭（清氦步）
D1074.04 BOOL  ; #1腔体机构正压开腔体阀/负压关腔体阀/氦检阀打开
D1074.05 BOOL  ; #1腔体机构（清氦步）
D1074.06 BOOL  ; #1腔体机构腔体抽气阀打开/电池抽气阀打开（清氦步）
D1074.07 BOOL  ; #1腔体机构腔体抽气阀关闭/电池抽气阀关闭（清氦步）
D1074.08 BOOL  ; #1腔体机构（清氦步）
D1074.09 BOOL  ; #1腔体机构氦检清洁阀打开/电池破真空阀打开（清氦步）
D1074.10 BOOL  ; #1腔体机构氦检清洁阀关闭/电池破真空阀关闭（清氦步）
D1074.11 BOOL  ; #1腔体机构（清氦步）
D1074.12 BOOL  ; #1腔体机构清氦次数判定（清氦步）
D1074.13 BOOL  ; #1腔体机构（清氦步）
D1074.14 BOOL  ; #1腔体机构腔体抽气阀打开/电池抽气阀打开（清氦步）
D1074.15 BOOL  ; #1腔体机构关闭电池抽气阀（清氦步）
D1075.00 BOOL  ; #1腔体机构腔体氦检阀仪真空阀打开/延时关腔体抽气阀（清氦步）
D1075.01 BOOL  ; #1腔体机构（清氦步）
D1075.02 BOOL  ; #1腔体机构腔体氦检阀关闭（清氦步）
D1075.03 BOOL  ; #1腔体机构腔体抽气阀关闭/电池抽气阀关闭（清氦步）
D1075.04 BOOL  ; #1腔体机构是否需要重新清氦判定（清氦步）
D1075.05 BOOL  ; #1腔体机构（清氦步）
D1075.06 BOOL  ; #1腔体机构开腔体破真空阀/开电池破真空阀/开腔体阀（清氦步）
D1075.07 BOOL  ; #1腔体机构关腔体破真空阀/关电池破真空阀（清氦步）
D1075.08 BOOL  ; #1腔体机构（清氦步）
D1075.09 BOOL  ; #1腔体机构清氦完成标志（清氦步）
D1075.10 BOOL  ; #1腔体机构（清氦步）
D1075.11 BOOL  ; #1腔体机构腔体顶升气缸下降（清氦步）
D1075.12 BOOL  ; #1腔体机构腔体平移气缸到初始位（清氦步）
D1075.13 BOOL  ; #1腔体机构（清氦步）
D1075.14 BOOL  ; #1腔体机构（清氦步）
D1075.15 BOOL  ; #1腔体机构循环结束（清氦步）
D1077.00 BOOL  ; #1腔体机构复位（M）
D1077.01 BOOL  ; #1腔体关闭除破真空阀以外全部阀门（复位）
D1077.02 BOOL  ; #1腔体打开腔体阀门（复位）
D1077.03 BOOL  ; #1腔体破真空值未到达开破真空阀（复位）
D1077.04 BOOL  ; #1腔体破真空值到达关破真空阀（复位）
D1077.05 BOOL  ; #1腔体腔体顶升气缸下降（复位）
D1077.06 BOOL  ; #1腔体腔体平移气缸伸出（复位）
D108 CHANNEL  ; 腔体测试设定破真空阈值（Pa_Float）
D1085.00 BOOL  ; #1腔体抽气阀打开允许（自检）
D1085.01 BOOL  ; #1腔体抽气阀打开需求（自检）
D1085.02 BOOL  ; #1腔体平移气缸在初始位（自检）
D1085.03 BOOL  ; #1腔体平移气缸在氦检位（自检）
D1085.04 BOOL  ; #1腔体真空泵开（自检）
D1085.05 BOOL  ; #1腔体平移气缸到初始位（自检）
D1085.06 BOOL  ; #1腔体平移气缸到氦检位（自检）
D1085.07 BOOL  ; #1腔体顶升气缸下降（自检）
D1085.08 BOOL  ; #1腔体顶升气缸上升（自检）
D1085.09 BOOL  ; #1腔体开抽真空阀（自检）
D1085.10 BOOL  ; #1腔体关抽真空阀（自检）
D1085.11 BOOL  ; #1腔体开破真空阀（自检）
D1085.12 BOOL  ; #1腔体关破真空阀（自检）
D1085.13 BOOL  ; #1腔体破真空阀状态（自检）
D1085.14 BOOL  ; #1腔体抽真空阀状态（自检）
D1086 CHANNEL  ; 标漏状态
D1087.00 BOOL  ; #1腔体机构标漏运行条件
D1087.01 BOOL  ; #1腔体机构标漏开始运行条件
D1087.02 BOOL  ; #1腔体机构标漏步进条件
D1087.15 BOOL  ; #1腔体机构标漏步进
D1088 CHANNEL  ; #1腔体标漏步序号
D1088.00 BOOL  ; #1腔体机构自动开始（标漏步）
D1088.01 BOOL  ; #1腔体机构关闭所有腔体阀门（标漏步）
D1088.02 BOOL  ; #1腔体机构所有腔体平移气缸到氦检位（标漏步）
D1088.03 BOOL  ; #1腔体机构所有腔体顶升气缸上升（标漏步）
D1088.04 BOOL  ; #1腔体机构关闭氦检仪真空阀/开氦检仪真空泵/腔体真空泵（标漏步）
D1088.05 BOOL  ; #1腔体机构开标漏阀（标漏步）
D1088.06 BOOL  ; #1腔体机构开#1腔体氦检阀（标漏步）
D1088.07 BOOL  ; #1腔体机构开#1-1腔体阀（标漏步）
D1088.08 BOOL  ; #1腔体机构开#1腔抽气阀（标漏步）
D1088.09 BOOL  ; #1腔体机构关#1腔体抽气阀（标漏步）
D1088.10 BOOL  ; #1腔体机构（标漏步）
D1088.11 BOOL  ; #1腔体机构（标漏步）
D1088.12 BOOL  ; #1腔体机构开始#1-1氦检（标漏步）
D1088.13 BOOL  ; #1腔体机构关#1腔体氦检阀（标漏步）
D1088.14 BOOL  ; #1腔体机构关#1-1腔体阀（标漏步）
D1088.15 BOOL  ; #1腔体机构开#1-2腔体阀（标漏步）
D1089.00 BOOL  ; #1腔体机构开#1腔抽真空阀（标漏步）
D1089.01 BOOL  ; #1腔体机构关#1腔抽真空阀（标漏步）
D1089.02 BOOL  ; #1腔体机构（标漏步）
D1089.03 BOOL  ; #1腔体机构（标漏步）
D1089.04 BOOL  ; #1腔体机构开始#1-2氦检（标漏步）
D1089.05 BOOL  ; #1腔体机构关#1腔体氦检阀（标漏步）
D1089.06 BOOL  ; #1腔体机构关#1-2腔体阀（标漏步）
D1089.07 BOOL  ; #1腔体机构（标漏步）
D1089.08 BOOL  ; #1腔体机构（标漏步）
D1089.09 BOOL  ; #1腔体机构（标漏步）
D1089.10 BOOL  ; #1腔体机构（标漏步）
D1089.11 BOOL  ; #1腔体机构（标漏步）
D1089.12 BOOL  ; #1腔体机构（标漏步）
D1089.13 BOOL  ; #1腔体机构（标漏步）
D1089.14 BOOL  ; #1腔体机构跳转至#2腔标漏步（标漏步）
D1089.15 BOOL  ; #1腔体机构循环结束（标漏步）
D1090.00 BOOL  ; #2氦检机构初始位
D1090.05 BOOL  ; #2氦检机构停止标志
D1090.06 BOOL  ; #2氦检机构清料完成标志
D1090.07 BOOL  ; #2氦检机构异常标志
D1091.00 BOOL  ; #2腔体机构运行条件（自动步）
D1091.01 BOOL  ; #2腔体机构运行条件（自动单检步）
D1091.02 BOOL  ; #2腔体机构运行条件（清氦步）
D1092.00 BOOL  ; #2腔体机构平移气缸安全移动条件
D1092.12 BOOL  ; #2腔体机构腔体抽真空需求（测试）
D1092.13 BOOL  ; #2腔体机构正常清氦需求（正压测试）
D1092.14 BOOL  ; #2腔体氦检阀打开允许条件
D1092.15 BOOL  ; #2腔体机构腔体抽气阀打开允许
D1093.00 BOOL  ; #2腔体机构单步/自动循环运行中（总）
D1093.10 BOOL  ; $?St$Bk?_#[16] / #2腔体机构记忆清除(SW) / $?St$Bk?_#[16]
D1093.12 BOOL  ; #2腔体自检启动(SW)
D1093.13 BOOL  ; #2腔体自检停止(SW)
D1093.14 BOOL  ; #2腔体机构复位按钮（SW）
D1093.15 BOOL  ; #2腔体机构单步（SW）
D1094.00 BOOL  ; #2腔体机构单步运行中
D1094.01 BOOL  ; #2腔体机构单步/自动循环运行中（自动步）
D1094.02 BOOL  ; #2腔体机构自动循环运行中（自动单检步）
D1094.03 BOOL  ; #2腔体机构自动循环运行中（清氦步）
D1094.04 BOOL  ; #2-1腔体单腔自检(SW)
D1094.05 BOOL  ; #2-2腔体单腔自检(SW)
D1094.06 BOOL  ; #2腔体自检运行中
D1095.00 BOOL  ; #2腔体机构开始运行条件（自动步）
D1095.01 BOOL  ; #2腔体机构步进条件（自动步）
D1095.02 BOOL  ; #2腔体机构开始运行条件（自动单检步）
D1095.03 BOOL  ; #2腔体机构步进条件（自动单检步）
D1095.04 BOOL  ; #2腔体机构开始运行条件（清氦步）
D1095.05 BOOL  ; #2腔体机构步进条件（清氦步）
D1095.13 BOOL  ; #2腔体机构步进（清氦步）
D1095.14 BOOL  ; #2腔体机构步进（自动单检步）
D1095.15 BOOL  ; #2腔体机构步进（自动步）
D1096 CHANNEL  ; #2腔体机构自动步序号
D1096.00 BOOL  ; #2腔体机构自动开始（自动步）
D1096.01 BOOL  ; #2腔体机构平移气缸到氦检位/数据初始化（自动步）
D1096.02 BOOL  ; #2腔体机构腔体顶升气缸上升（自动步）
D1096.03 BOOL  ; #2腔体机构等待氦检阀打开条件及腔体抽气阀打开条件/开腔体阀（自动步）
D1096.04 BOOL  ; #2腔体机构（自动步）
D1096.05 BOOL  ; #2腔体机构腔体抽气阀打开/延时开电池抽气阀（自动步）
D1096.06 BOOL  ; #2腔体机构关电池抽气阀（自动步）
D1096.07 BOOL  ; #2腔体机构开电池注氦阀（自动步）
D1096.08 BOOL  ; #2腔体机构关电池注氦阀（自动步）
D1096.09 BOOL  ; #2腔体机构（自动步）
D1096.10 BOOL  ; #2腔体机构开腔体氦检阀/延时关腔体抽气阀（自动步）
D1096.11 BOOL  ; #2腔体机构（自动步）
D1096.12 BOOL  ; #2腔体机构关腔体氦检阀（自动步）
D1096.13 BOOL  ; #2腔体机构（自动步）
D1096.14 BOOL  ; #2腔体机构开腔体#2-1腔体阀/开腔体#2-2腔体阀（自动步）
D1096.15 BOOL  ; #2腔体机构开腔体抽真空阀/开电池抽真空阀（自动步）
D1097.00 BOOL  ; #2腔体机构关腔体抽真空阀/关电池抽真空阀/开腔体阀（自动步）
D1097.01 BOOL  ; #2腔体机构清氦需求判定（自动步）
D1097.02 BOOL  ; #2腔体机构开腔体破真空阀/开电池破真空阀（自动步）
D1097.03 BOOL  ; #2腔体机构关腔体破真空阀/关电池破真空阀（自动步）
D1097.04 BOOL  ; #2腔体机构复测需求判定（自动步）
D1097.05 BOOL  ; #2腔体机构（自动步）
D1097.06 BOOL  ; #2腔体机构腔体顶升气缸下降（自动步）
D1097.07 BOOL  ; #2腔体机构（自动步）
D1097.08 BOOL  ; #2腔体机构腔体平移气缸到出料位（自动步）
D1097.09 BOOL  ; #2腔体机构腔体等待取料完成信号（自动步）
D1097.10 BOOL  ; #2腔体机构（自动步）
D1097.11 BOOL  ; #2腔体机构平移气缸到上料位（自动步）
D1097.12 BOOL  ; #2腔体机构（自动步）
D1097.13 BOOL  ; #2腔体机构（自动步）
D1097.14 BOOL  ; #2腔体机构（自动步）
D1097.15 BOOL  ; #2腔体机构循环结束（自动步）
D110 CHANNEL  ; 腔体测试设定氦检时间（S_UInt）
D1100 CHANNEL  ; #2腔体机构单检步序号
D1100.00 BOOL  ; #2腔体机构自动开始（自动单检步）
D1100.01 BOOL  ; #2腔体机构平移气缸到氦检位/数据初始化（自动单检步）
D1100.02 BOOL  ; #2腔体机构腔体顶升气缸上升（自动单检步）
D1100.03 BOOL  ; #2腔体机构关闭#2-2腔体阀（自动单检步）
D1100.04 BOOL  ; #2腔体机构腔体抽气阀打开/延时开#2-1电池抽气阀（自动单检步）
D1100.05 BOOL  ; #2腔体机构关#2-1电池抽气阀（自动单检步）
D1100.06 BOOL  ; #2腔体机构开#2-1电池注氦阀（自动单检步）
D1100.07 BOOL  ; #2腔体机构关#2-1电池注氦阀（自动单检步）
D1100.08 BOOL  ; #2腔体机构（自动单检步）
D1100.09 BOOL  ; #2腔体机构开腔体氦检阀/延时关腔体抽气阀（自动单检步）
D1100.10 BOOL  ; #2腔体机构关腔体氦检阀/关腔体抽气阀/关#2-1电池抽气阀（自动单检步）
D1100.11 BOOL  ; #2腔体机构关闭#2-1腔体阀/清氦判定（自动单检步）
D1100.12 BOOL  ; #2腔体机构打开#2-2腔体阀（自动单检步）
D1100.13 BOOL  ; #2腔体机构腔体抽气阀打开/延时开#2-2电池抽气阀（自动单检步）
D1100.14 BOOL  ; #2腔体机构关#2-2电池抽气阀（自动单检步）
D1100.15 BOOL  ; #2腔体机构开#2-2电池注氦阀（自动单检步）
D1101.00 BOOL  ; #2腔体机构关#2-2电池注氦阀（自动单检步）
D1101.01 BOOL  ; #2腔体机构（自动单检步）
D1101.02 BOOL  ; #2腔体机构开腔体氦检阀/延时关腔体抽气阀（自动单检步）
D1101.03 BOOL  ; #2腔体机构关腔体氦检阀（自动单检步）
D1101.04 BOOL  ; #2腔体机构开腔体#2-1阀（自动单检步）
D1101.05 BOOL  ; #2腔体机构开腔体抽真空阀/开电池抽真空阀（自动单检步）
D1101.06 BOOL  ; #2腔体机构关腔体抽真空阀/关电池抽真空阀（自动单检步）
D1101.07 BOOL  ; #2腔体机构清氦需求判定（自动单检步）
D1101.08 BOOL  ; #2腔体机构开腔体破真空阀/开电池破真空阀（自动单检步）
D1101.09 BOOL  ; #2腔体机构关腔体破真空阀/关电池破真空阀（自动单检步）
D1101.10 BOOL  ; #2腔体机构腔体顶升气缸下降（自动单检步）
D1101.11 BOOL  ; #2腔体机构腔体平移气缸到出料位（自动单检步）
D1101.12 BOOL  ; #2腔体机构腔体等待取料完成信号（自动单检步）
D1101.13 BOOL  ; #2腔体机构腔体平移气缸到上料位（自动单检步）
D1101.14 BOOL  ; #2腔体机构（自动单检步）
D1101.15 BOOL  ; #2腔体机构循环结束（自动单检步）
D1104 CHANNEL  ; #2腔体机构清氦步序号
D1104.00 BOOL  ; #2腔体机构自动开始（清氦步）
D1104.01 BOOL  ; #2腔体机构平移气缸到氦检位/数据初始化（清氦步）
D1104.02 BOOL  ; #2腔体机构腔体顶升气缸上升（清氦步）
D1104.03 BOOL  ; #2腔体机构氦检仪真空阀关闭（清氦步）
D1104.04 BOOL  ; #2腔体机构正压开腔体阀/负压关腔体阀/氦检阀打开
D1104.05 BOOL  ; #2腔体机构（清氦步）
D1104.06 BOOL  ; #2腔体机构腔体抽气阀打开/电池抽气阀打开（清氦步）
D1104.07 BOOL  ; #2腔体机构腔体抽气阀关闭/电池抽气阀关闭（清氦步）
D1104.08 BOOL  ; #2腔体机构（清氦步）
D1104.09 BOOL  ; #2腔体机构氦检清洁阀打开/电池破真空阀打开（清氦步）
D1104.10 BOOL  ; #2腔体机构氦检清洁阀关闭/电池破真空阀关闭（清氦步）
D1104.11 BOOL  ; #2腔体机构（清氦步）
D1104.12 BOOL  ; #2腔体机构清氦次数判定（清氦步）
D1104.13 BOOL  ; #2腔体机构（清氦步）
D1104.14 BOOL  ; #2腔体机构腔体抽气阀打开/电池抽气阀打开（清氦步）
D1104.15 BOOL  ; #2腔体机构关闭电池抽气阀（清氦步）
D1105.00 BOOL  ; #2腔体机构腔体氦检阀仪真空阀打开/延时关腔体抽气阀（清氦步）
D1105.01 BOOL  ; #2腔体机构（清氦步）
D1105.02 BOOL  ; #2腔体机构腔体氦检阀关闭（清氦步）
D1105.03 BOOL  ; #2腔体机构腔体抽气阀关闭/电池抽气阀关闭（清氦步）
D1105.04 BOOL  ; #2腔体机构是否需要重新清氦判定（清氦步）
D1105.05 BOOL  ; #2腔体机构（清氦步）
D1105.06 BOOL  ; #2腔体机构开腔体破真空阀/开电池破真空阀/开腔体阀（清氦步）
D1105.07 BOOL  ; #2腔体机构关腔体破真空阀/关电池破真空阀（清氦步）
D1105.08 BOOL  ; #2腔体机构（清氦步）
D1105.09 BOOL  ; #2腔体机构清氦完成标志（清氦步）
D1105.10 BOOL  ; #2腔体机构（清氦步）
D1105.11 BOOL  ; #2腔体机构腔体顶升气缸下降（清氦步）
D1105.12 BOOL  ; #2腔体机构腔体平移气缸到初始位（清氦步）
D1105.13 BOOL  ; #2腔体机构（清氦步）
D1105.14 BOOL  ; #2腔体机构（清氦步）
D1105.15 BOOL  ; #2腔体机构循环结束（清氦步）
D1107.00 BOOL  ; #2腔体机构复位（M）
D1107.01 BOOL  ; #2腔体关闭除破真空阀以外全部阀门（复位）
D1107.02 BOOL  ; #2腔体打开腔体阀门（复位）
D1107.03 BOOL  ; #2腔体破真空值未到达开破真空阀（复位）
D1107.04 BOOL  ; #2腔体破真空值到达关破真空阀（复位）
D1107.05 BOOL  ; #2腔体腔体顶升气缸下降（复位）
D1107.06 BOOL  ; #2腔体腔体平移气缸伸出（复位）
D1115.00 BOOL  ; #2腔体抽气阀打开允许（自检）
D1115.01 BOOL  ; #2腔体抽气阀打开需求（自检）
D1115.02 BOOL  ; #2腔体平移气缸在初始位（自检）
D1115.03 BOOL  ; #2腔体平移气缸在氦检位（自检）
D1115.04 BOOL  ; #2腔体真空泵开（自检）
D1115.05 BOOL  ; #2腔体平移气缸到初始位（自检）
D1115.06 BOOL  ; #2腔体平移气缸到氦检位（自检）
D1115.07 BOOL  ; #2腔体顶升气缸下降（自检）
D1115.08 BOOL  ; #2腔体顶升气缸上升（自检）
D1115.09 BOOL  ; #2腔体开抽真空阀（自检）
D1115.10 BOOL  ; #2腔体关抽真空阀（自检）
D1115.11 BOOL  ; #2腔体开破真空阀（自检）
D1115.12 BOOL  ; #2腔体关破真空阀（自检）
D1115.13 BOOL  ; #2腔体破真空阀状态（自检）
D1115.14 BOOL  ; #2腔体抽真空阀状态（自检）
D1117.00 BOOL  ; #2腔体机构标漏运行条件
D1117.01 BOOL  ; #2腔体机构标漏开始运行条件
D1117.02 BOOL  ; #2腔体机构标漏步进条件
D1117.15 BOOL  ; #2腔体机构标漏步进
D1118 CHANNEL  ; #2腔体标漏步序号
D1118.00 BOOL  ; #2腔体机构自动开始（标漏步）
D1118.01 BOOL  ; #2腔体机构（标漏步）
D1118.02 BOOL  ; #2腔体机构（标漏步）
D1118.03 BOOL  ; #2腔体机构（标漏步）
D1118.04 BOOL  ; #2腔体机构（标漏步）
D1118.05 BOOL  ; #2腔体机构（标漏步）
D1118.06 BOOL  ; #2腔体机构（标漏步）
D1118.07 BOOL  ; #2腔体机构开#2-1腔体阀（标漏步）
D1118.08 BOOL  ; #2腔体机构开#2腔抽气阀（标漏步）
D1118.09 BOOL  ; #2腔体机构关#2腔体抽气阀（标漏步）
D1118.10 BOOL  ; #2腔体机构（标漏步）
D1118.11 BOOL  ; #2腔体机构（标漏步）
D1118.12 BOOL  ; #2腔体机构开始#2-1氦检（标漏步）
D1118.13 BOOL  ; #2腔体机构关#2腔体氦检阀（标漏步）
D1118.14 BOOL  ; #2腔体机构关#2-1腔体阀（标漏步）
D1118.15 BOOL  ; #2腔体机构开#2-2腔体阀（标漏步）
D1119.00 BOOL  ; #2腔体机构开#2腔抽真空阀（标漏步）
D1119.01 BOOL  ; #2腔体机构关#2腔抽真空阀（标漏步）
D1119.02 BOOL  ; #2腔体机构（标漏步）
D1119.03 BOOL  ; #2腔体机构（标漏步）
D1119.04 BOOL  ; #2腔体机构开始#2-2氦检（标漏步）
D1119.05 BOOL  ; #2腔体机构关#2腔体氦检阀（标漏步）
D1119.06 BOOL  ; #2腔体机构关#2-2腔体阀（标漏步）
D1119.07 BOOL  ; #2腔体机构（标漏步）
D1119.08 BOOL  ; #2腔体机构（标漏步）
D1119.09 BOOL  ; #2腔体机构（标漏步）
D1119.10 BOOL  ; #2腔体机构（标漏步）
D1119.11 BOOL  ; #2腔体机构（标漏步）
D1119.12 BOOL  ; #2腔体机构（标漏步）
D1119.13 BOOL  ; #2腔体机构（标漏步）
D1119.14 BOOL  ; #2腔体机构跳转至#3腔标漏步（标漏步）
D1119.15 BOOL  ; #2腔体机构循环结束（标漏步）
D112 CHANNEL  ; 泄漏率（Pa.m3/s_Float）
D1120.00 BOOL  ; #3氦检机构初始位
D1120.05 BOOL  ; #3氦检机构停止标志
D1120.06 BOOL  ; #3氦检机构清料完成标志
D1120.07 BOOL  ; #3腔体机构异常标志
D1121.00 BOOL  ; #3腔体机构运行条件（自动步）
D1121.01 BOOL  ; #3腔体机构运行条件（自动单检步）
D1121.02 BOOL  ; #3腔体机构运行条件（清氦步）
D1122.00 BOOL  ; #3腔体机构平移气缸安全移动条件
D1122.12 BOOL  ; #3腔体机构腔体抽真空需求（测试）
D1122.13 BOOL  ; #3腔体机构正常清氦需求（正压测试）
D1122.14 BOOL  ; #3腔体氦检阀打开允许条件
D1122.15 BOOL  ; #3腔体机构腔体抽气阀打开允许
D1123.00 BOOL  ; #3腔体机构单步/自动循环运行中（总）
D1123.10 BOOL  ; $?St$Bk?_#[17] / #3腔体机构记忆清除(SW) / $?St$Bk?_#[17]
D1123.12 BOOL  ; #3腔体自检启动(SW)
D1123.13 BOOL  ; #3腔体自检停止(SW)
D1123.14 BOOL  ; #3腔体机构复位按钮（SW）
D1123.15 BOOL  ; #3腔体机构单步（SW）
D1124.00 BOOL  ; #3腔体机构单步运行中
D1124.01 BOOL  ; #3腔体机构单步/自动循环运行中（自动步）
D1124.02 BOOL  ; #3腔体机构自动循环运行中（自动单检步）
D1124.03 BOOL  ; #3腔体机构自动循环运行中（清氦步）
D1124.04 BOOL  ; #3-1腔体单腔自检(SW)
D1124.05 BOOL  ; #3-2腔体单腔自检(SW)
D1124.06 BOOL  ; #3腔体自检运行中
D1125.00 BOOL  ; #3腔体机构开始运行条件（自动步）
D1125.01 BOOL  ; #3腔体机构步进条件（自动步）
D1125.02 BOOL  ; #3腔体机构开始运行条件（自动单检步）
D1125.03 BOOL  ; #3腔体机构步进条件（自动单检步）
D1125.04 BOOL  ; #3腔体机构开始运行条件（清氦步）
D1125.05 BOOL  ; #3腔体机构步进条件（清氦步）
D1125.13 BOOL  ; #3腔体机构步进（清氦步）
D1125.14 BOOL  ; #3腔体机构步进（自动单检步）
D1125.15 BOOL  ; #3腔体机构步进（自动步）
D1126 CHANNEL  ; #3腔体机构自动步序号
D1126.00 BOOL  ; #3腔体机构自动开始（自动步）
D1126.01 BOOL  ; #3腔体机构平移气缸到氦检位/数据初始化（自动步）
D1126.02 BOOL  ; #3腔体机构腔体顶升气缸上升（自动步）
D1126.03 BOOL  ; #3腔体机构等待氦检阀打开条件及腔体抽气阀打开条件/开腔体阀（自动步）
D1126.04 BOOL  ; #3腔体机构（自动步）
D1126.05 BOOL  ; #3腔体机构腔体抽气阀打开/延时开电池抽气阀（自动步）
D1126.06 BOOL  ; #3腔体机构关电池抽气阀（自动步）
D1126.07 BOOL  ; #3腔体机构开电池注氦阀（自动步）
D1126.08 BOOL  ; #3腔体机构关电池注氦阀（自动步）
D1126.09 BOOL  ; #3腔体机构（自动步）
D1126.10 BOOL  ; #3腔体机构开腔体氦检阀/延时关腔体抽气阀（自动步）
D1126.11 BOOL  ; #3腔体机构（自动步）
D1126.12 BOOL  ; #3腔体机构关腔体氦检阀（自动步）
D1126.13 BOOL  ; #3腔体机构（自动步）
D1126.14 BOOL  ; #3腔体机构开腔体#3-1腔体阀/开腔体#3-2腔体阀（自动步）
D1126.15 BOOL  ; #3腔体机构开腔体抽真空阀/开电池抽真空阀（自动步）
D1127.00 BOOL  ; #3腔体机构关腔体抽真空阀/关电池抽真空阀/开腔体阀（自动步）
D1127.01 BOOL  ; #3腔体机构清氦需求判定（自动步）
D1127.02 BOOL  ; #3腔体机构开腔体破真空阀/开电池破真空阀（自动步）
D1127.03 BOOL  ; #3腔体机构关腔体破真空阀/关电池破真空阀（自动步）
D1127.04 BOOL  ; #3腔体机构复测需求判定（自动步）
D1127.05 BOOL  ; #3腔体机构（自动步）
D1127.06 BOOL  ; #3腔体机构腔体顶升气缸下降（自动步）
D1127.07 BOOL  ; #3腔体机构（自动步）
D1127.08 BOOL  ; #3腔体机构腔体平移气缸到出料位（自动步）
D1127.09 BOOL  ; #3腔体机构腔体等待取料完成信号（自动步）
D1127.10 BOOL  ; #3腔体机构（自动步）
D1127.11 BOOL  ; #3腔体机构平移气缸到上料位（自动步）
D1127.12 BOOL  ; #3腔体机构（自动步）
D1127.13 BOOL  ; #3腔体机构（自动步）
D1127.14 BOOL  ; #3腔体机构（自动步）
D1127.15 BOOL  ; #3腔体机构循环结束（自动步）
D1130 CHANNEL  ; #3腔体机构单检步序号
D1130.00 BOOL  ; #3腔体机构自动开始（自动单检步）
D1130.01 BOOL  ; #3腔体机构平移气缸到氦检位/数据初始化（自动单检步）
D1130.02 BOOL  ; #3腔体机构腔体顶升气缸上升（自动单检步）
D1130.03 BOOL  ; #3腔体机构关闭#3-2腔体阀（自动单检步）
D1130.04 BOOL  ; #3腔体机构腔体抽气阀打开/延时开#3-1电池抽气阀（自动单检步）
D1130.05 BOOL  ; #3腔体机构关#3-1电池抽气阀（自动单检步）
D1130.06 BOOL  ; #3腔体机构开#3-1电池注氦阀（自动单检步）
D1130.07 BOOL  ; #3腔体机构关#3-1电池注氦阀（自动单检步）
D1130.08 BOOL  ; #3腔体机构（自动单检步）
D1130.09 BOOL  ; #3腔体机构开腔体氦检阀/延时关腔体抽气阀（自动单检步）
D1130.10 BOOL  ; #3腔体机构关腔体氦检阀/关腔体抽气阀/关#3-1电池抽气阀（自动单检步）
D1130.11 BOOL  ; #3腔体机构关闭#3-1腔体阀/清氦判定（自动单检步）
D1130.12 BOOL  ; #3腔体机构打开#3-2腔体阀（自动单检步）
D1130.13 BOOL  ; #3腔体机构腔体抽气阀打开/延时开#3-2电池抽气阀（自动单检步）
D1130.14 BOOL  ; #3腔体机构关#3-2电池抽气阀（自动单检步）
D1130.15 BOOL  ; #3腔体机构开#3-2电池注氦阀（自动单检步）
D1131.00 BOOL  ; #3腔体机构关#3-2电池注氦阀（自动单检步）
D1131.01 BOOL  ; #3腔体机构（自动单检步）
D1131.02 BOOL  ; #3腔体机构开腔体氦检阀/延时关腔体抽气阀（自动单检步）
D1131.03 BOOL  ; #3腔体机构关腔体氦检阀（自动单检步）
D1131.04 BOOL  ; #3腔体机构开腔体#3-1阀（自动单检步）
D1131.05 BOOL  ; #3腔体机构开腔体抽真空阀/开电池抽真空阀（自动单检步）
D1131.06 BOOL  ; #3腔体机构关腔体抽真空阀/关电池抽真空阀（自动单检步）
D1131.07 BOOL  ; #3腔体机构清氦需求判定（自动单检步）
D1131.08 BOOL  ; #3腔体机构开腔体破真空阀/开电池破真空阀（自动单检步）
D1131.09 BOOL  ; #3腔体机构关腔体破真空阀/关电池破真空阀（自动单检步）
D1131.10 BOOL  ; #3腔体机构腔体顶升气缸下降（自动单检步）
D1131.11 BOOL  ; #3腔体机构腔体平移气缸到出料位（自动单检步）
D1131.12 BOOL  ; #3腔体机构腔体等待取料完成信号（自动单检步）
D1131.13 BOOL  ; #3腔体机构腔体平移气缸到上料位（自动单检步）
D1131.14 BOOL  ; #3腔体机构（自动单检步）
D1131.15 BOOL  ; #3腔体机构循环结束（自动单检步）
D1134 CHANNEL  ; #3腔体机构清氦步序号
D1134.00 BOOL  ; #3腔体机构自动开始（清氦步）
D1134.01 BOOL  ; #3腔体机构平移气缸到氦检位/数据初始化（清氦步）
D1134.02 BOOL  ; #3腔体机构腔体顶升气缸上升（清氦步）
D1134.03 BOOL  ; #3腔体机构氦检仪真空阀关闭（清氦步）
D1134.04 BOOL  ; #3腔体机构正压开腔体阀/负压关腔体阀/氦检阀打开
D1134.05 BOOL  ; #3腔体机构（清氦步）
D1134.06 BOOL  ; #3腔体机构腔体抽气阀打开/电池抽气阀打开（清氦步）
D1134.07 BOOL  ; #3腔体机构腔体抽气阀关闭/电池抽气阀关闭（清氦步）
D1134.08 BOOL  ; #3腔体机构（清氦步）
D1134.09 BOOL  ; #3腔体机构氦检清洁阀打开/电池破真空阀打开（清氦步）
D1134.10 BOOL  ; #3腔体机构氦检清洁阀关闭/电池破真空阀关闭（清氦步）
D1134.11 BOOL  ; #3腔体机构（清氦步）
D1134.12 BOOL  ; #3腔体机构清氦次数判定（清氦步）
D1134.13 BOOL  ; #3腔体机构（清氦步）
D1134.14 BOOL  ; #3腔体机构腔体抽气阀打开/电池抽气阀打开（清氦步）
D1134.15 BOOL  ; #3腔体机构关闭电池抽气阀（清氦步）
D1135.00 BOOL  ; #3腔体机构腔体氦检阀仪真空阀打开/延时关腔体抽气阀（清氦步）
D1135.01 BOOL  ; #3腔体机构（清氦步）
D1135.02 BOOL  ; #3腔体机构腔体氦检阀关闭（清氦步）
D1135.03 BOOL  ; #3腔体机构腔体抽气阀关闭/电池抽气阀关闭（清氦步）
D1135.04 BOOL  ; #3腔体机构是否需要重新清氦判定（清氦步）
D1135.05 BOOL  ; #3腔体机构（清氦步）
D1135.06 BOOL  ; #3腔体机构开腔体破真空阀/开电池破真空阀/开腔体阀（清氦步）
D1135.07 BOOL  ; #3腔体机构关腔体破真空阀/关电池破真空阀（清氦步）
D1135.08 BOOL  ; #3腔体机构（清氦步）
D1135.09 BOOL  ; #3腔体机构清氦完成标志（清氦步）
D1135.10 BOOL  ; #3腔体机构（清氦步）
D1135.11 BOOL  ; #3腔体机构腔体顶升气缸下降（清氦步）
D1135.12 BOOL  ; #3腔体机构腔体平移气缸到初始位（清氦步）
D1135.13 BOOL  ; #3腔体机构（清氦步）
D1135.14 BOOL  ; #3腔体机构（清氦步）
D1135.15 BOOL  ; #3腔体机构循环结束（清氦步）
D1137.00 BOOL  ; #3腔体机构复位（M）
D1137.01 BOOL  ; #3腔体关闭除破真空阀以外全部阀门（复位）
D1137.02 BOOL  ; #3腔体打开腔体阀门（复位）
D1137.03 BOOL  ; #3腔体破真空值未到达开破真空阀（复位）
D1137.04 BOOL  ; #3腔体破真空值到达关破真空阀（复位）
D1137.05 BOOL  ; #3腔体腔体顶升气缸下降（复位）
D1137.06 BOOL  ; #3腔体腔体平移气缸伸出（复位）
D114 CHANNEL  ; 泄漏率（Pa.m3/s_Float_指数）
D1145.00 BOOL  ; #3腔体抽气阀打开允许（自检）
D1145.01 BOOL  ; #3腔体抽气阀打开需求（自检）
D1145.02 BOOL  ; #3腔体平移气缸在初始位（自检）
D1145.03 BOOL  ; #3腔体平移气缸在氦检位（自检）
D1145.04 BOOL  ; #3腔体真空泵开（自检）
D1145.05 BOOL  ; #3腔体平移气缸到初始位（自检）
D1145.06 BOOL  ; #3腔体平移气缸到氦检位（自检）
D1145.07 BOOL  ; #3腔体顶升气缸下降（自检）
D1145.08 BOOL  ; #3腔体顶升气缸上升（自检）
D1145.09 BOOL  ; #3腔体开抽真空阀（自检）
D1145.10 BOOL  ; #3腔体关抽真空阀（自检）
D1145.11 BOOL  ; #3腔体开破真空阀（自检）
D1145.12 BOOL  ; #3腔体关破真空阀（自检）
D1145.13 BOOL  ; #3腔体破真空阀状态（自检）
D1145.14 BOOL  ; #3腔体抽真空阀状态（自检）
D1147.00 BOOL  ; #3腔体机构标漏运行条件
D1147.01 BOOL  ; #3腔体机构标漏开始运行条件
D1147.02 BOOL  ; #3腔体机构标漏步进条件
D1147.15 BOOL  ; #3腔体机构标漏步进
D1148 CHANNEL  ; #3腔体标漏步序号
D1148.00 BOOL  ; #3腔体机构自动开始（标漏步）
D1148.01 BOOL  ; #3腔体机构（标漏步）
D1148.02 BOOL  ; #3腔体机构（标漏步）
D1148.03 BOOL  ; #3腔体机构（标漏步）
D1148.04 BOOL  ; #3腔体机构（标漏步）
D1148.05 BOOL  ; #3腔体机构（标漏步）
D1148.06 BOOL  ; #3腔体机构（标漏步）
D1148.07 BOOL  ; #3腔体机构开#3-1腔体阀（标漏步）
D1148.08 BOOL  ; #3腔体机构开#3腔抽气阀（标漏步）
D1148.09 BOOL  ; #3腔体机构关#3腔体抽气阀（标漏步）
D1148.10 BOOL  ; #3腔体机构（标漏步）
D1148.11 BOOL  ; #3腔体机构（标漏步）
D1148.12 BOOL  ; #3腔体机构开始#3-1氦检（标漏步）
D1148.13 BOOL  ; #3腔体机构关#3腔体氦检阀（标漏步）
D1148.14 BOOL  ; #3腔体机构关#3-1腔体阀（标漏步）
D1148.15 BOOL  ; #3腔体机构开#3-2腔体阀（标漏步）
D1149.00 BOOL  ; #3腔体机构开#3腔抽真空阀（标漏步）
D1149.01 BOOL  ; #3腔体机构关#3腔抽真空阀（标漏步）
D1149.02 BOOL  ; #3腔体机构（标漏步）
D1149.03 BOOL  ; #3腔体机构（标漏步）
D1149.04 BOOL  ; #3腔体机构开始#3-2氦检（标漏步）
D1149.05 BOOL  ; #3腔体机构关#3腔体氦检阀（标漏步）
D1149.06 BOOL  ; #3腔体机构关#3-2腔体阀（标漏步）
D1149.07 BOOL  ; #3腔体机构开所有腔体总阀（标漏步）
D1149.08 BOOL  ; #3腔体机构开所有腔体破真空阀（标漏步）
D1149.09 BOOL  ; #3腔体机构关所有腔体破真空阀（标漏步）
D1149.10 BOOL  ; #3腔体机构所有顶升气缸下降（标漏步）
D1149.11 BOOL  ; #3腔体机构所有腔体平移气缸回初始位（标漏步）
D1149.12 BOOL  ; #3腔体机构关标漏阀（标漏步）
D1149.13 BOOL  ; #3腔体机构（标漏步）
D1149.14 BOOL  ; #3腔体机构（标漏步）
D1149.15 BOOL  ; #3腔体机构循环结束（标漏步）
D1150.00 BOOL  ; 出料伺服机构初始位
D1150.05 BOOL  ; 出料伺服机构停止标志
D1150.06 BOOL  ; 出料伺服机构清料完成标志
D1150.07 BOOL  ; 出料伺服机构异常标志
D1153.14 BOOL  ; 出料伺服机构复位按钮（SW）
D1156 CHANNEL  ; 下料模组自动流程
D1156.00 BOOL  ; 下料模组运行前检测
D1156.01 BOOL  ; 下料模组运行备用
D1156.02 BOOL  ; 下料x模组运行到对应下料位
D1156.03 BOOL  ; 下料Z模组运行前检测
D1156.04 BOOL  ; 下料Z模组运行
D1156.05 BOOL  ; 下料模组夹爪夹紧
D1156.06 BOOL  ; 下料模组运行备用
D1156.07 BOOL  ; 下料Z模组到待机位
D1156.08 BOOL  ; 下料模组取料完成记忆
D1156.09 BOOL  ; 下料模组是否放全OK料检测
D1156.10 BOOL  ; 下料X模组到OK下料位/旋转气缸到90度(负压)
D1156.11 BOOL  ; 下料Z模组OK下降检测
D1156.12 BOOL  ; 下料Z模组到OK下料位
D1156.13 BOOL  ; 下料模组放全OK料开夹爪
D1156.14 BOOL  ; 下料Z模组到待机位/旋转气缸到0度(负压)
D1156.15 BOOL  ; *下料模组去腔体取料流程&全OK下料结束
D1158 CHANNEL  ; 下料模组全NG流程
D1158.00 BOOL  ; 下料模组全OK/NG料流程准备
D1158.01 BOOL  ; 下料X模组到2#爪放料位
D1158.02 BOOL  ; 下料模组放2#NG安全检测
D1158.03 BOOL  ; 下料模组放2#NG Z轴下降
D1158.04 BOOL  ; 下料模组开2#NG夹爪
D1158.05 BOOL  ; 下料Z模组放完2#NG回待机位
D1158.06 BOOL  ; 下料X模组到1#爪放料位
D1158.07 BOOL  ; 下料模组放1#NG安全检测
D1158.08 BOOL  ; 下料模组放1#NG Z轴下降
D1158.09 BOOL  ; 下料模组开1#NG夹爪
D1158.10 BOOL  ; 下料Z模组放完1#NG回待机位
D1158.11 BOOL  ; 下料模组放双NG备用
D1158.12 BOOL  ; 下料模组放双NG备用
D1158.13 BOOL  ; 下料模组放双NG备用
D1158.14 BOOL  ; 下料模组放双NG备用
D1158.15 BOOL  ; 下料模组放双NG结束
D116 CHANNEL  ; 检漏口压力（Pa_Float）
D1160 CHANNEL  ; 下料模组（取）放1OK/1NG流程
D1160.00 BOOL  ; *下料模组（取）放1OK/1NG流程运行前检测
D1160.01 BOOL  ; 下料X模组到达对应X位置
D1160.02 BOOL  ; 下料Z模组下降前检测
D1160.03 BOOL  ; 下料Z模组下降放NG料
D1160.04 BOOL  ; 下料模组开NG夹爪
D1160.05 BOOL  ; 下料Z模组放完NG回待机位
D1160.06 BOOL  ; 下料模组放缓存OR取缓存
D1160.07 BOOL  ; 下料X模组到放缓存位
D1160.08 BOOL  ; 下料Z模组下降放缓存
D1160.09 BOOL  ; 下料模组放缓存开夹爪or夹紧
D1160.10 BOOL  ; 下料模组缓存有料检测
D1160.11 BOOL  ; 下料Z模组到待机位
D1160.12 BOOL  ; *下料模组（取）放1OK/1NG X轴到OK下料位/旋转气缸到90度(负压)
D1160.13 BOOL  ; *下料模组（取）放1OK/1NG出料伺服Z轴放料位
D1160.14 BOOL  ; *下料模组（取）放1OK/1NG出料伺服Z轴待机&旋转气缸到0度(负压)
D1160.15 BOOL  ; *下料模组（取）放1OK/1NG流程结束
D1166 CHANNEL  ; 下料模组X/Z初始化
D1166.00 BOOL  ; 下料模组初始化准备
D1166.01 BOOL  ; 下料Z模组初始化
D1166.02 BOOL  ; 下料Z模组到待机位&旋转气缸到0度(负压)
D1166.03 BOOL  ; 下料X模组初始化
D1166.04 BOOL  ; 下料X模组到待机位
D1166.05 BOOL  ; 下料模组运行许可
D1166.06 BOOL  ; 下料模组初始化结束
D1168 CHANNEL  ; 下料模组手动跟踪联动
D1168.00 BOOL  ; 下料模组手动跟踪Z回待机位
D1168.01 BOOL  ; 下料模组手动跟踪X到对应位置
D1168.02 BOOL  ; 下料Z轴手动下降前安全判定
D1168.03 BOOL  ; 下料Z模组手动下降
D1168.04 BOOL  ; 下料X/Z模组跟踪联动需求清除
D1168.05 BOOL  ; 下料X/Z模组手动联动结束
D118 CHANNEL  ; 检漏口压力（Pa_Float_指数）
D120 CHANNEL  ; 稳定漏率（Pa.m3/s_Float）
D122 CHANNEL  ; 稳定漏率（Pa.m3/s_Float_指数）
D124 CHANNEL  ; 腔体测试设定清氦次数（次_UInt）
D126 CHANNEL  ; 腔体测试设定氦检时腔体抽气阀关延时（S_UInt）
D128 CHANNEL  ; 腔体抽真空大漏判定值(Float)
D136 CHANNEL  ; 腔体测试设定腔体预抽检测时间（S_UInt）
D138 CHANNEL  ; $?St$Bk?_#[18] / 管路清氦注氮时间（S_UInt） / $?St$Bk?_#[18]
D14 CHANNEL  ; 感应器ON延时设定值
D15 CHANNEL  ; 感应器ON延时设定值_1
D150 CHANNEL  ; 腔体自检真空到达阈值SV（Pa_Float）
D152 CHANNEL  ; 腔体自检抽真空时间上限SV（S_UInt）
D154 CHANNEL  ; 腔体自检泄漏量阈值SV（Pa_Float）
D156 CHANNEL  ; 清氦泄漏率（Pa.m3/s_Float）
D158 CHANNEL  ; 清氦泄漏率（Pa.m3/s_Float_指数）
D16 CHANNEL  ; 感应器延时时间
D160 CHANNEL  ; 电池测试设定真空阈值（Pa_Float）
D162 CHANNEL  ; 电池测试设定抽真空时间上限（S_UInt）
D168 CHANNEL  ; 电池测试设定注氦时间上限（S_UInt）
D17 CHANNEL  ; 感应器ON延时设定值_3
D170 CHANNEL  ; 电池测试设定清氦压力（Pa_Float）
D172 CHANNEL  ; 电池测试设定破真空阈值（Pa_Float）
D174 CHANNEL  ; 电池测试设定预抽检测压力（Pa_Float）
D176 CHANNEL  ; 电池测试设定#1-1注氦压力（Pa_Float）
D178 CHANNEL  ; 电池测试设定#2-1注氦压力（Pa_Float）
D18 CHANNEL  ; 自动运行条件延时时间
D188 CHANNEL  ; 漏率设定值（Pa.m3/s_Float）
D19 CHANNEL  ; 自动运行步间间隔时间
D190 CHANNEL  ; 检漏口压力设定值（Pa_Float）
D196 CHANNEL  ; 氦检仪漏率（Pa.m3/s_Float）
D198 CHANNEL  ; 氦检仪检漏口压力（Pa_Float）
D20 CHANNEL  ; 感应器ON延时设定值_6
D200 CHANNEL  ; #1-1腔体状态（0停用，1待料中，2测试中，3测试完成，4-清氦中）
D202 CHANNEL  ; #1-1腔体测试漏率（Pa.m3/s_Float）
D204 CHANNEL  ; #1-1腔体测试检漏口压力（Pa_Float）
D206 CHANNEL  ; #1-1电池充氦压力（Pa_Float）
D208 CHANNEL  ; #1-1腔体测试结果（1 OK，2腔体泄漏，3气密NG，4注氦超时，5氦检异常，6电池泄漏）
D21 CHANNEL  ; 报警长延时
D210 CHANNEL  ; $?St$Bk?_#[19] / #1-1充氦嘴压力（Pa_Float） / #1-1充氦嘴压力（Pa_Float） / #1-1充氦嘴压力（Pa_Float）$?St$Bk?_#[19]
D212 CHANNEL  ; #1-1腔体抽气时间（S_UInt）
D214 CHANNEL  ; #1-1腔体真空压力（Pa_Float）
D216 CHANNEL  ; #1-1电池抽气时间（S_UInt）
D2160 CHANNEL  ; 氦检仪状态(1.检漏；2.待机；3.定标；4.启动；5.错误；6.暂停)
D2162 CHANNEL  ; 氦检实时漏率显示
D218 CHANNEL  ; #1-1电池真空压力（Pa_Float）
D22 CHANNEL  ; 报警短延时
D23 CHANNEL  ; 氦检相关无传感器阀开关到位延时设定
D230 CHANNEL  ; #1-1腔体自检抽气时间（S_UInt）
D232 CHANNEL  ; #1-1腔体自检前保压时间（S_UInt）
D234 CHANNEL  ; #1-1腔体自检保压时间（S_UInt）
D236 CHANNEL  ; #1-1腔体自检保压前真空（Pa_Float）
D238 CHANNEL  ; #1-1腔体自检保压后真空（Pa_Float）
D24 CHANNEL  ; 伺服到位延时
D240 CHANNEL  ; #1-1腔体自检泄漏量（Pa_Float）
D242 CHANNEL  ; #1-1腔体自检结果（1-OK，2-NG）
D2500 CHANNEL  ; #1扫码阻挡气缸缩回位延时设定值
D2501 CHANNEL  ; #1扫码阻挡气缸伸出位延时设定值
D2502 CHANNEL  ; #1隔离气缸缩回位延时设定值
D2503 CHANNEL  ; 0延时设定值
D2504 CHANNEL  ; #2扫码阻挡气缸缩回位延时设定值
D2505 CHANNEL  ; #2扫码阻挡气缸伸出位延时设定值
D2506 CHANNEL  ; #2隔离气缸缩回位延时设定值
D2507 CHANNEL  ; 0延时设定值
D2508 CHANNEL  ; #1进料夹爪夹紧位延时设定值
D2509 CHANNEL  ; #1进料夹爪松开位延时设定值
D2510 CHANNEL  ; #2进料夹爪夹紧位延时设定值
D2511 CHANNEL  ; #2进料夹爪松开位延时设定值
D2512 CHANNEL  ; 进料夹爪变距气缸伸出位延时设定值
D2513 CHANNEL  ; 进料夹爪变距气缸缩回位延时设定值
D2514 CHANNEL  ; #1出料夹爪夹紧位延时设定值
D2515 CHANNEL  ; #1出料夹爪松开位延时设定值
D2516 CHANNEL  ; #2出料夹爪夹紧位延时设定值
D2517 CHANNEL  ; #2出料夹爪松开位延时设定值
D2518 CHANNEL  ; 出料夹爪变距气缸伸出位延时设定值
D2519 CHANNEL  ; 出料夹爪变距气缸缩回位延时设定值
D2520 CHANNEL  ; #1腔体平移一级气缸缩回位延时设定值
D2521 CHANNEL  ; #1腔体平移一级气缸伸出位延时设定值
D2522 CHANNEL  ; #1腔体平移二级气缸缩回位延时设定值
D2523 CHANNEL  ; #1腔体平移二级气缸伸出位延时设定值
D2524 CHANNEL  ; #1腔体顶伸气缸上升位延时设定值
D2525 CHANNEL  ; #1腔体顶伸气缸下降位延时设定值
D2526 CHANNEL  ; #1腔体氦检阀开到位延时设定值
D2527 CHANNEL  ; #1腔体氦检阀关到位延时设定值
D2528 CHANNEL  ; 0延时设定值
D2529 CHANNEL  ; 0延时设定值
D2530 CHANNEL  ; 0延时设定值
D2531 CHANNEL  ; 0延时设定值
D2532 CHANNEL  ; 0延时设定值
D2533 CHANNEL  ; #2腔体平移一级气缸缩回位延时设定值
D2534 CHANNEL  ; #2腔体平移一级气缸伸出位延时设定值
D2535 CHANNEL  ; #2腔体平移二级气缸缩回位延时设定值
D2536 CHANNEL  ; #2腔体平移二级气缸伸出位延时设定值
D2537 CHANNEL  ; #2腔体顶伸气缸上升位延时设定值
D2538 CHANNEL  ; #2腔体顶伸气缸下降位延时设定值
D2539 CHANNEL  ; #2腔体氦检阀开到位延时设定值
D2540 CHANNEL  ; #2腔体氦检阀关到位延时设定值
D2541 CHANNEL  ; 0延时设定值
D2542 CHANNEL  ; 0延时设定值
D2543 CHANNEL  ; 0延时设定值
D2544 CHANNEL  ; 0延时设定值
D2545 CHANNEL  ; 0延时设定值
D2546 CHANNEL  ; #3腔体平移一级气缸缩回位延时设定值
D2547 CHANNEL  ; #3腔体平移一级气缸伸出位延时设定值
D2548 CHANNEL  ; #3腔体平移二级气缸缩回位延时设定值
D2549 CHANNEL  ; #3腔体平移二级气缸伸出位延时设定值
D2550 CHANNEL  ; #3腔体顶伸气缸上升位延时设定值
D2551 CHANNEL  ; #3腔体顶伸气缸下降位延时设定值
D2552 CHANNEL  ; #3腔体氦检阀开到位延时设定值
D2553 CHANNEL  ; #3腔体氦检阀关到位延时设定值
D2554 CHANNEL  ; 氦检仪准备好了信号延时设定值
D2555 CHANNEL  ; 氦检仪故障信号延时设定值
D2556 CHANNEL  ; 0延时设定值
D2557 CHANNEL  ; 0延时设定值
D2558 CHANNEL  ; 0延时设定值
D2559 CHANNEL  ; 进料伺服X轴准备好了信号延时设定值
D2560 CHANNEL  ; 进料伺服X轴故障信号延时设定值
D2561 CHANNEL  ; 进料伺服Z轴准备好了信号延时设定值
D2562 CHANNEL  ; 进料伺服Z轴故障信号延时设定值
D2563 CHANNEL  ; 0延时设定值
D2564 CHANNEL  ; 出料伺服X轴准备好了信号延时设定值
D2565 CHANNEL  ; 出料伺服X轴故障信号延时设定值
D2566 CHANNEL  ; 出料伺服Z轴准备好了信号延时设定值
D2567 CHANNEL  ; 出料伺服Z轴故障信号延时设定值
D2568 CHANNEL  ; 0延时设定值
D2569 CHANNEL  ; 腔体抽真空泵运行信号延时设定值
D2570 CHANNEL  ; 腔体抽真空泵过载信号延时设定值
D2571 CHANNEL  ; 氦检前置泵运行信号延时设定值
D2572 CHANNEL  ; 氦检前置泵过载信号延时设定值
D2573 CHANNEL  ; 启动按钮延时设定值
D2574 CHANNEL  ; 停止按钮延时设定值
D2575 CHANNEL  ; 复位按钮延时设定值
D2576 CHANNEL  ; 急停按钮延时设定值
D2577 CHANNEL  ; 手自动选择延时设定值
D2578 CHANNEL  ; #1进料夹爪防下坠感应延时设定值
D2579 CHANNEL  ; #2进料夹爪防下坠感应延时设定值
D258 CHANNEL  ; #1-1清氦泄漏率（清氦）
D2580 CHANNEL  ; #1出料夹爪防下坠感应延时设定值
D2581 CHANNEL  ; #2出料夹爪防下坠感应延时设定值
D2582 CHANNEL  ; 0延时设定值
D2583 CHANNEL  ; 进料对接输入延时设定值
D2584 CHANNEL  ; 出料对接输入延时设定值
D2585 CHANNEL  ; 出料旋转气缸9O度位延时设定值
D2586 CHANNEL  ; 出料旋转气缸O度位延时设定值
D2587 CHANNEL  ; 设备总气压信号延时设定值
D2588 CHANNEL  ; #1来料位有料感应延时设定值
D2589 CHANNEL  ; #2来料位有料感应延时设定值
D2590 CHANNEL  ; #1隔离位有料感应延时设定值
D2591 CHANNEL  ; #2隔离位有料感应延时设定值
D2592 CHANNEL  ; #1扫码位有料感应延时设定值
D2593 CHANNEL  ; #2扫码位有料感应延时设定值
D2594 CHANNEL  ; #1-1进料位有料感应延时设定值
D2595 CHANNEL  ; #1-2进料位有料感应延时设定值
D2596 CHANNEL  ; #2-1进料位有料感应延时设定值
D2597 CHANNEL  ; #2-2进料位有料感应延时设定值
D2598 CHANNEL  ; 进料夹爪柔性感应延时设定值
D2599 CHANNEL  ; 出料夹爪柔性感应延时设定值
D260 CHANNEL  ; #1-1氦检时真空值（标漏）
D2600 CHANNEL  ; #1进料夹爪对应腔体有料感应延时设定值
D2601 CHANNEL  ; #2进料夹爪对应腔体有料感应延时设定值
D2602 CHANNEL  ; 扫码NG放料#1位有料感应延时设定值
D2603 CHANNEL  ; 扫码NG放料#2位有料感应延时设定值
D2604 CHANNEL  ; 扫码NG料满位有料感应延时设定值
D2605 CHANNEL  ; 进料配对位有料感应延时设定值
D2606 CHANNEL  ; 出料配对位有料感应延时设定值
D2607 CHANNEL  ; 氦检NG放料#1位有料感应延时设定值
D2608 CHANNEL  ; 氦检NG放料#2位有料感应延时设定值
D2609 CHANNEL  ; 氦检NG料满位有料感应延时设定值
D2610 CHANNEL  ; #1-1出料位有料感应延时设定值
D2611 CHANNEL  ; #1-2出料位有料感应延时设定值
D2612 CHANNEL  ; #2-1出料位有料感应延时设定值
D2613 CHANNEL  ; #2-2出料位有料感应延时设定值
D2614 CHANNEL  ; #1门磁开关延时设定值
D2615 CHANNEL  ; #2门磁开关延时设定值
D2616 CHANNEL  ; #3门磁开关延时设定值
D2617 CHANNEL  ; #4门磁开关延时设定值
D2618 CHANNEL  ; #5门磁开关延时设定值
D2619 CHANNEL  ; #6门磁开关延时设定值
D262 CHANNEL  ; #1-1氦检漏率（标漏）
D2620 CHANNEL  ; #7门磁开关延时设定值
D2621 CHANNEL  ; #8门磁开关延时设定值
D2622 CHANNEL  ; #9门磁开关延时设定值
D2623 CHANNEL  ; #10门磁开关延时设定值
D2624 CHANNEL  ; #11门磁开关延时设定值
D2625 CHANNEL  ; 设备真空压力信号延时设定值
D2626 CHANNEL  ; 设备氦气压力信号延时设定值
D2627 CHANNEL  ; 精密调压阀信号延时设定值
D2663 CHANNEL  ; $?St$Bk?_#[20] / #1隔离气缸伸出位延时设定值 / $?St$Bk?_#[20]
D2667 CHANNEL  ; $?St$Bk?_#[21] / #2隔离气缸伸出位延时设定值 / $?St$Bk?_#[21]
D270 CHANNEL  ; #1腔体抽真空需求计时
D272 CHANNEL  ; #1-1腔体管路清氦计数
D296 CHANNEL  ; 字符表示形式
D297 CHANNEL  ; 全位数
D298 CHANNEL  ; 小数位数
D3 CHANNEL  ; #2腔体设定读取时间(Float)
D30 CHANNEL  ; NG扫码重试次数设置
D300 CHANNEL  ; #2-1腔体状态（0停用，1待料中，2测试中，3测试完成，4-清氦中）
D3000 CHANNEL  ; 设备PPM测试时间设置
D3002 CHANNEL  ; 设备PPM测试时间累计
D3004 CHANNEL  ; 设备PPM测试#1出料夹爪数量累计
D3006 CHANNEL  ; 设备PPM测试#2出料夹爪数量累计
D3008 CHANNEL  ; 设备PPM测试出料夹爪总数量累计
D302 CHANNEL  ; #2-1腔体测试漏率（Pa.m3/s_Float）
D304 CHANNEL  ; #2-1腔体测试检漏口压力（Pa_Float）
D306 CHANNEL  ; #2-1电池充氦压力（Pa_Float）
D308 CHANNEL  ; #2-1腔体测试结果（1 OK，2腔体泄漏，3气密NG，4注氦超时，5氦检异常，6电池泄漏，7注氦NG，8氦嘴泄漏）
D310 CHANNEL  ; #2-1充氦嘴压力（Pa_Float）
D3102 CHANNEL  ; 腔体测试设定抽真空时间上限（S_UInt）浮点
D3110 CHANNEL  ; 腔体测试设定氦检时间（S_UInt）浮点
D312 CHANNEL  ; #2-1腔体抽气时间（S_UInt）
D3136 CHANNEL  ; 腔体测试设定腔体预抽检测时间（S_UInt）浮点
D314 CHANNEL  ; #2-1腔体真空压力（Pa_Float）
D316 CHANNEL  ; #2-1电池抽气时间（S_UInt）
D3162 CHANNEL  ; 电池测试设定抽真空时间上限（S_UInt）浮点
D318 CHANNEL  ; #2-1电池真空压力（Pa_Float）
D330 CHANNEL  ; #2-1腔体自检抽气时间（S_UInt）
D332 CHANNEL  ; #2-1腔体自检前保压时间（S_UInt）
D334 CHANNEL  ; #2-1腔体自检保压时间（S_UInt）
D336 CHANNEL  ; #2-1腔体自检保压前真空（Pa_Float）
D338 CHANNEL  ; #2-1腔体自检保压后真空（Pa_Float）
D340 CHANNEL  ; #2-1腔体自检泄漏量（Pa_Float）
D342 CHANNEL  ; #2-1腔体自检结果（1-OK，2-NG）
D358 CHANNEL  ; $?St$Bk?_#[22] / #2-1清氦泄漏率（清氦） / $?St$Bk?_#[22]
D360 CHANNEL  ; #2-1氦检时真空值（标漏）
D362 CHANNEL  ; #2-1氦检漏率（标漏）
D370 CHANNEL  ; #2腔体抽真空需求计时
D372 CHANNEL  ; #2-1腔体管路清氦计数
D40 CHANNEL  ; #1出料夹爪OK料计数（DINT）
D400 CHANNEL  ; #3-1腔体状态（0停用，1待料中，2测试中，3测试完成，4-清氦中）
D402 CHANNEL  ; #3-1腔体测试漏率（Pa.m3/s_Float）
D404 CHANNEL  ; #3-1腔体测试检漏口压力（Pa_Float）
D406 CHANNEL  ; #3-1电池充氦压力（Pa_Float）
D408 CHANNEL  ; #3-1腔体测试结果（1 OK，2腔体泄漏，3气密NG，4注氦超时，5氦检异常，6电池泄漏，7注氦NG，8氦嘴泄漏）
D410 CHANNEL  ; #3-1充氦嘴压力（Pa_Float）
D4100 CHANNEL  ; 腔体测试设定真空阈值（Pa_Float）储存
D4102 CHANNEL  ; 腔体测试设定抽真空时间上限（S_UInt）储存
D4104 CHANNEL  ; 腔体测试设定清氦压力（Pa_Float）储存
D4110 CHANNEL  ; 腔体测试设定氦检时间（S_UInt）储存
D412 CHANNEL  ; #3-1腔体抽气时间（S_UInt）
D4136 CHANNEL  ; 腔体测试设定腔体预抽检测时间（S_UInt）储存
D414 CHANNEL  ; #3-1腔体真空压力（Pa_Float）
D416 CHANNEL  ; #3-1电池抽气时间（S_UInt）
D4160 CHANNEL  ; 电池测试设定真空阈值（Pa_Float）储存
D4162 CHANNEL  ; 电池测试设定抽真空时间上限（S_UInt）储存
D4170 CHANNEL  ; 电池测试设定清氦压力（Pa_Float）储存
D4174 CHANNEL  ; 电池测试设定预抽检测压力（Pa_Float）储存
D418 CHANNEL  ; #3-1电池真空压力（Pa_Float）
D42 CHANNEL  ; #1出料夹爪NG料计数（DINT）
D430 CHANNEL  ; #3-1腔体自检抽气时间（S_UInt）
D432 CHANNEL  ; #3-1腔体自检前保压时间（S_UInt）
D434 CHANNEL  ; #3-1腔体自检保压时间（S_UInt）
D436 CHANNEL  ; #3-1腔体自检保压前真空（Pa_Float）
D438 CHANNEL  ; #3-1腔体自检保压后真空（Pa_Float）
D44 CHANNEL  ; 出料夹爪OK料总计数（DINT）
D440 CHANNEL  ; #3-1腔体自检泄漏量（Pa_Float）
D442 CHANNEL  ; #3-1腔体自检结果（1-OK，2-NG）
D458 CHANNEL  ; $?St$Bk?_#[23] / #3-1清氦泄漏率（清氦） / $?St$Bk?_#[23]
D46 CHANNEL  ; 出料夹爪总计数（DINT）
D460 CHANNEL  ; #3-1氦检时真空值（标漏）
D462 CHANNEL  ; #3-1氦检漏率（标漏）
D470 CHANNEL  ; #3腔体抽真空需求计时
D472 CHANNEL  ; #3-1腔体管路清氦计数
D48 CHANNEL  ; 出料夹爪OK料总计数（Float）
D4994 CHANNEL  ; 泄漏率设定值（Pa.m3/s_Float）储存
D4996 CHANNEL  ; 检漏口压力设定值（Pa_Float）储存
D4998 CHANNEL  ; 清氦漏率设定值（Pa_Float）储存
D5 CHANNEL  ; #3腔体设定读取时间(Float)
D50 CHANNEL  ; #2出料夹爪OK料计数（DINT）
D500 CHANNEL  ; #1-2腔体状态（0停用，1待料中，2测试中，3测试完成，4-清氦中）
D502 CHANNEL  ; #1-2腔体测试漏率（Pa.m3/s_Float）
D504 CHANNEL  ; #1-2腔体测试检漏口压力（Pa_Float）
D506 CHANNEL  ; #1-2电池充氦压力（Pa_Float）
D508 CHANNEL  ; #1-2腔体测试结果（1 OK，2腔体泄漏，3气密NG，4注氦超时，5氦检异常，6电池泄漏，7注氦NG，8氦嘴泄漏）
D510 CHANNEL  ; #1-2充氦嘴压力（Pa_Float）
D512 CHANNEL  ; #1-2腔体抽气时间（S_UInt）
D514 CHANNEL  ; #1-2腔体真空压力（Pa_Float）
D516 CHANNEL  ; #1-2电池抽气时间（S_UInt）
D518 CHANNEL  ; #1-2电池真空压力（Pa_Float）
D52 CHANNEL  ; #2出料夹爪NG料计数（DINT）
D5200 CHANNEL  ; 发送内容“T”+“0D”
D5201 CHANNEL  ; 发送内容“0A”
D5210 CHANNEL  ; 进料#1扫码数据开始字
D5240 CHANNEL  ; 进料#1扫码条码开始字
D5259 CHANNEL  ; 进料#1扫码数据结束字
D530 CHANNEL  ; #1-2腔体自检抽气时间（S_UInt）
D5300 CHANNEL  ; 进料#2扫码长度
D5301 CHANNEL  ; 进料#2扫码条码开始字
D5319 CHANNEL  ; 进料#2扫码结束字
D532 CHANNEL  ; #1-2腔体自检前保压时间（S_UInt）
D534 CHANNEL  ; #1-2腔体自检保压时间（S_UInt）
D536 CHANNEL  ; #1-2腔体自检保压前真空（Pa_Float）
D538 CHANNEL  ; #1-2腔体自检保压后真空（Pa_Float）
D54 CHANNEL  ; 出料夹爪NG料总计数（DINT）
D540 CHANNEL  ; #1-2腔体自检泄漏量（Pa_Float）
D542 CHANNEL  ; #1-2腔体自检结果（1-OK，2-NG,3-抽真空NG）
D56 CHANNEL  ; 出料夹爪总计数（Float）
D560 CHANNEL  ; #1-2氦检时真空值（标漏）
D562 CHANNEL  ; #1-2氦检漏率（标漏）
D58 CHANNEL  ; 出料夹爪OK料百分比（Float）
D60 CHANNEL  ; 接收条码数据字长度
D600 CHANNEL  ; #2-2腔体状态（0停用，1待料中，2测试中，3测试完成，4-清氦中）
D6000 CHANNEL  ; 进料伺服X轴加速比率
D6001 CHANNEL  ; 进料伺服X轴减速比率
D6002 CHANNEL  ; 进料伺服X轴目标速度
D6003 CHANNEL  ; 进料伺服X轴目标速度
D6004 CHANNEL  ; 进料伺服X轴目标位置
D6005 CHANNEL  ; 进料伺服X轴目标位置
D6006 CHANNEL  ; 进料伺服X轴启动频率
D6007 CHANNEL  ; 进料伺服X轴启动频率
D602 CHANNEL  ; #2-2腔体测试漏率（Pa.m3/s_Float）
D6020 CHANNEL  ; 进料伺服X轴JOG运行加减速
D6021 CHANNEL  ; 进料伺服X轴JOG运行速度
D6022 CHANNEL  ; 进料伺服X轴JOG运行速度
D6030 CHANNEL  ; 进料伺服X轴JOG停止加减速
D6031 CHANNEL  ; 进料伺服X轴JOG停止速度
D6032 CHANNEL  ; 进料伺服X轴JOG停止速度
D604 CHANNEL  ; #2-2腔体测试检漏口压力（Pa_Float）
D6040 CHANNEL  ; 进料伺服X轴当前位置
D6041 CHANNEL  ; 进料伺服X轴当前位置
D6042 CHANNEL  ; 进料伺服X轴当前速度
D6043 CHANNEL  ; 进料伺服X轴当前速度
D6050 CHANNEL  ; 进/出料伺服急停位置预置
D606 CHANNEL  ; #2-2电池充氦压力（Pa_Float）
D608 CHANNEL  ; #2-2腔体测试结果（1 OK，2腔体泄漏，3气密NG，4注氦超时，5氦检异常，6电池泄漏，7注氦NG，8氦嘴泄漏）
D610 CHANNEL  ; #2-2充氦嘴压力（Pa_Float）
D6100 CHANNEL  ; 进料伺服X轴加速比率SV
D6101 CHANNEL  ; 进料伺服X轴减速比率SV
D6102 CHANNEL  ; 进料伺服X轴目标速度SV
D6103 CHANNEL  ; 进料伺服X轴目标速度SV
D6106 CHANNEL  ; 进料伺服X轴启动频率SV
D6107 CHANNEL  ; 进料伺服X轴启动频率SV
D612 CHANNEL  ; #2-2腔体抽气时间（S_UInt）
D6120 CHANNEL  ; 进料伺服X轴JOG运行/停止加减速SV
D6121 CHANNEL  ; 进料伺服X轴JOG运行速度SV
D6122 CHANNEL  ; 进料伺服X轴JOG运行速度SV
D6131 CHANNEL  ; 进料伺服X轴JOG停止速度SV
D6132 CHANNEL  ; 进料伺服X轴JOG停止速度SV
D614 CHANNEL  ; #2-2腔体真空压力（Pa_Float）
D6152 CHANNEL  ; 进料伺服X轴取料位SV
D6153 CHANNEL  ; 进料伺服X轴取料位SV
D6154 CHANNEL  ; 进料伺服X轴#1腔放料位SV
D6155 CHANNEL  ; 进料伺服X轴#1腔放料位SV
D6156 CHANNEL  ; 进料伺服X轴#2腔放料位SV
D6157 CHANNEL  ; 进料伺服X轴#2腔放料位SV
D6158 CHANNEL  ; 进料伺服X轴#3腔放料位SV
D6159 CHANNEL  ; 进料伺服X轴#3腔放料位SV
D616 CHANNEL  ; #2-2电池抽气时间（S_UInt）
D6160 CHANNEL  ; 进料伺服X轴#1夹爪扫码NG放料位SV
D6161 CHANNEL  ; 进料伺服X轴#1夹爪扫码NG放料位SV
D6162 CHANNEL  ; 进料伺服X轴#2夹爪扫码NG放料位SV
D6163 CHANNEL  ; 进料伺服X轴#2夹爪扫码NG放料位SV
D6164 CHANNEL  ; 进料伺服X轴#1夹爪配对取放料位SV
D6165 CHANNEL  ; 进料伺服X轴#1夹爪配对取放料位SV
D6166 CHANNEL  ; 进料伺服X轴#2夹爪配对取放料位SV
D6167 CHANNEL  ; 进料伺服X轴#2夹爪配对取放料位SV
D6168 CHANNEL  ; 进料伺服X轴#1腔有料检测位SV
D6169 CHANNEL  ; 进料伺服X轴#1腔有料检测位SV
D6170 CHANNEL  ; 进料伺服X轴#2腔有料检测位SV
D6171 CHANNEL  ; 进料伺服X轴#2腔有料检测位SV
D6172 CHANNEL  ; 进料伺服X轴#3腔有料检测位SV
D6173 CHANNEL  ; 进料伺服X轴#3腔有料检测位SV
D618 CHANNEL  ; #2-2电池真空压力（Pa_Float）
D6200 CHANNEL  ; 进料伺服Z轴加速比率
D6201 CHANNEL  ; 进料伺服Z轴减速比率
D6202 CHANNEL  ; 进料伺服Z轴目标速度
D6203 CHANNEL  ; 进料伺服Z轴目标速度
D6204 CHANNEL  ; 进料伺服Z轴目标位置
D6205 CHANNEL  ; 进料伺服Z轴目标位置
D6206 CHANNEL  ; 进料伺服Z轴启动频率
D6207 CHANNEL  ; 进料伺服Z轴启动频率
D6220 CHANNEL  ; 进料伺服Z轴JOG运行加减速
D6221 CHANNEL  ; 进料伺服Z轴JOG运行速度
D6222 CHANNEL  ; 进料伺服Z轴JOG运行速度
D6230 CHANNEL  ; 进料伺服Z轴JOG停止加减速
D6231 CHANNEL  ; 进料伺服Z轴JOG停止速度
D6232 CHANNEL  ; 进料伺服Z轴JOG停止速度
D6240 CHANNEL  ; 进料伺服Z轴当前位置
D6241 CHANNEL  ; 进料伺服Z轴当前位置
D6242 CHANNEL  ; 进料伺服Z轴当前速度
D6243 CHANNEL  ; 进料伺服Z轴当前速度
D6254 CHANNEL  ; 进料伺服Z轴#1腔放料位SV1
D6255 CHANNEL  ; 进料伺服Z轴#1腔放料位SV1
D6256 CHANNEL  ; 进料伺服Z轴#2腔放料位SV1
D6257 CHANNEL  ; 进料伺服Z轴#2腔放料位SV1
D6258 CHANNEL  ; 进料伺服Z轴#3腔放料位SV1
D6259 CHANNEL  ; 进料伺服Z轴#3腔放料位SV1
D630 CHANNEL  ; #2-2腔体自检抽气时间（S_UInt）
D6300 CHANNEL  ; 进料伺服Z轴加速比率SV
D6301 CHANNEL  ; 进料伺服Z轴减速比率SV
D6302 CHANNEL  ; 进料伺服Z轴目标速度SV
D6303 CHANNEL  ; 进料伺服Z轴目标速度SV
D6306 CHANNEL  ; 进料伺服Z轴启动频率SV
D6307 CHANNEL  ; 进料伺服Z轴启动频率SV
D632 CHANNEL  ; #2-2腔体自检前保压时间（S_UInt）
D6320 CHANNEL  ; 进料伺服Z轴JOG运行/停止加减速SV
D6321 CHANNEL  ; 进料伺服Z轴JOG运行速度SV
D6322 CHANNEL  ; 进料伺服Z轴JOG运行速度SV
D6331 CHANNEL  ; 进料伺服Z轴JOG停止速度SV
D6332 CHANNEL  ; 进料伺服Z轴JOG停止速度SV
D634 CHANNEL  ; #2-2腔体自检保压时间（S_UInt）
D6350 CHANNEL  ; 进料伺服Z轴待料位SV
D6351 CHANNEL  ; 进料伺服Z轴待料位SV
D6352 CHANNEL  ; 进料伺服Z轴取料位SV
